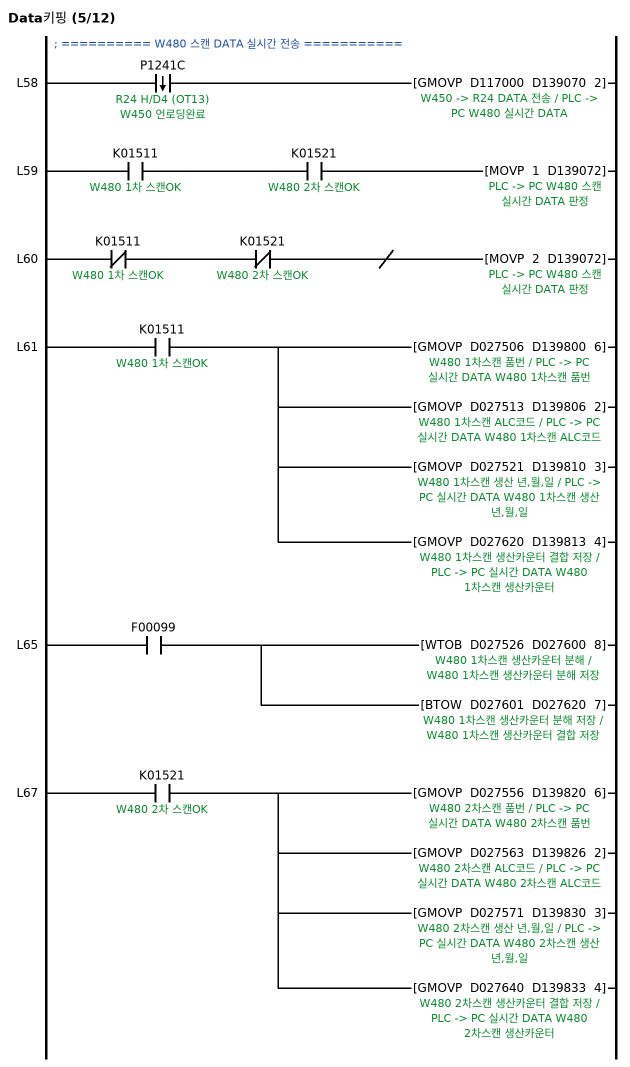
[picture p504: Data키핑 rungs L58-L67]
// ========== W480 스캔 DATA 실시간 전송 ===========
; L58
LOADN     P1241C	// R24 H/D4 (OT13) W450 언로딩완료
GMOVP     D117000 D139070 2	// W450 -> R24 DATA 전송 / PLC -> PC W480 실시간 DATA
; L59
LOAD      K01511	// W480 1차 스캔OK
AND       K01521	// W480 2차 스캔OK
MOVP      1 D139072	// PLC -> PC W480 스캔 실시간 DATA 판정
; L60
LOAD NOT  K01511	// W480 1차 스캔OK
AND NOT   K01521	// W480 2차 스캔OK
NOT
MOVP      2 D139072	// PLC -> PC W480 스캔 실시간 DATA 판정
; L61
LOAD      K01511	// W480 1차 스캔OK
GMOVP     D027506 D139800 6	// W480 1차스캔 품번 / PLC -> PC 실시간 DATA W480 1차스캔 품번
GMOVP     D027513 D139806 2	// W480 1차스캔 ALC코드 / PLC -> PC 실시간 DATA W480 1차스캔 ALC코드
GMOVP     D027521 D139810 3	// W480 1차스캔 생산 년,월,일 / PLC -> PC 실시간 DATA W480 1차스캔 생산 년,월,일
GMOVP     D027620 D139813 4	// W480 1차스캔 생산카운터 결합 저장 / PLC -> PC 실시간 DATA W480 1차스캔 생산카운터
; L65
LOAD      F00099
WTOB      D027526 D027600 8	// W480 1차스캔 생산카운터 분해 / W480 1차스캔 생산카운터 분해 저장
BTOW      D027601 D027620 7	// W480 1차스캔 생산카운터 분해 저장 / W480 1차스캔 생산카운터 결합 저장
; L67
LOAD      K01521	// W480 2차 스캔OK
GMOVP     D027556 D139820 6	// W480 2차스캔 품번 / PLC -> PC 실시간 DATA W480 2차스캔 품번
GMOVP     D027563 D139826 2	// W480 2차스캔 ALC코드 / PLC -> PC 실시간 DATA W480 2차스캔 ALC코드
GMOVP     D027571 D139830 3	// W480 2차스캔 생산 년,월,일 / PLC -> PC 실시간 DATA W480 2차스캔 생산 년,월,일
GMOVP     D027640 D139833 4	// W480 2차스캔 생산카운터 결합 저장 / PLC -> PC 실시간 DATA W480 2차스캔 생산카운터

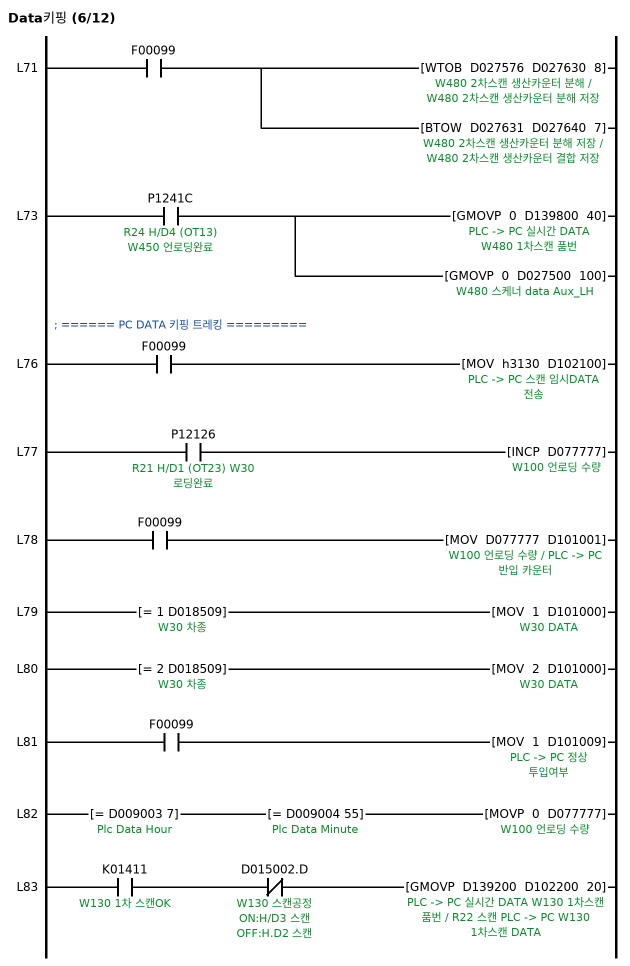
; L71
LOAD      F00099
WTOB      D027576 D027630 8	// W480 2차스캔 생산카운터 분해 / W480 2차스캔 생산카운터 분해 저장
BTOW      D027631 D027640 7	// W480 2차스캔 생산카운터 분해 저장 / W480 2차스캔 생산카운터 결합 저장
; L73
LOAD      P1241C	// R24 H/D4 (OT13) W450 언로딩완료
GMOVP     0 D139800 40	// PLC -> PC 실시간 DATA W480 1차스캔 품번
GMOVP     0 D027500 100	// W480 스케너 data Aux_LH
// ====== PC DATA 키핑 트레킹 =========
; L76
LOAD      F00099
MOV       h3130 D102100	// PLC -> PC 스캔 임시DATA 전송
; L77
LOAD      P12126	// R21 H/D1 (OT23) W30 로딩완료
INCP      D077777	// W100 언로딩 수량
; L78
LOAD      F00099
MOV       D077777 D101001	// W100 언로딩 수량 / PLC -> PC 반입 카운터
; L79
LOAD=     1 D018509	// W30 차종
MOV       1 D101000	// W30 DATA
; L80
LOAD=     2 D018509	// W30 차종
MOV       2 D101000	// W30 DATA
; L81
LOAD      F00099
MOV       1 D101009	// PLC -> PC 정상 투입여부
; L82
LOAD=     D009003 7	// Plc Data Hour
AND=      D009004 55	// Plc Data Minute
MOVP      0 D077777	// W100 언로딩 수량
; L83
LOAD      K01411	// W130 1차 스캔OK
AND NOT   D015002.D	// W130 스캔공정 ON:H/D3 스캔 OFF:H.D2 스캔
GMOVP     D139200 D102200 20	// PLC -> PC 실시간 DATA W130 1차스캔 품번 / R22 스캔 PLC -> PC W130 1차스캔 DATA

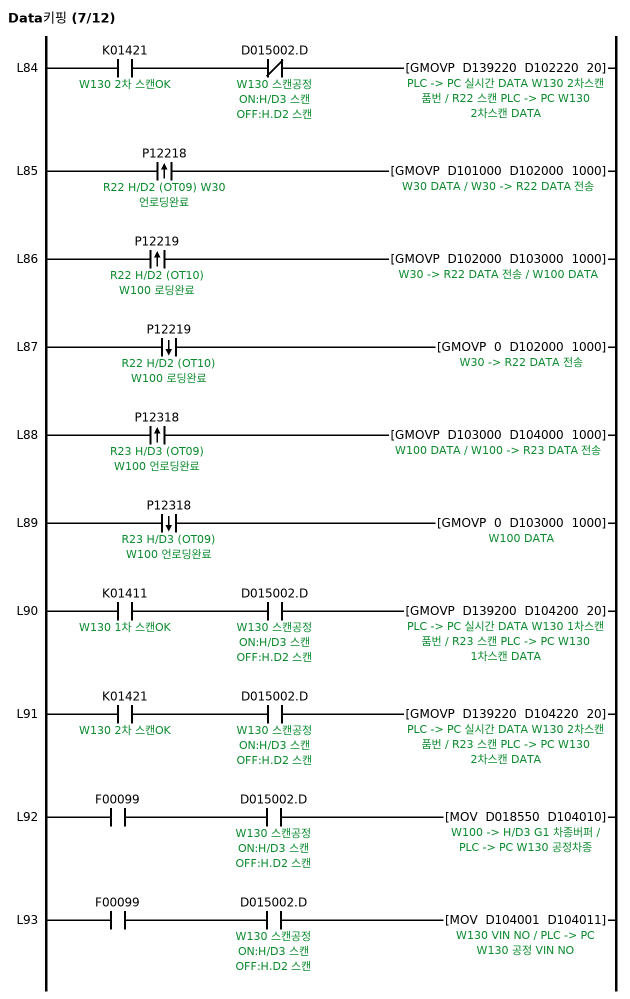
; L84
LOAD      K01421	// W130 2차 스캔OK
AND NOT   D015002.D	// W130 스캔공정 ON:H/D3 스캔 OFF:H.D2 스캔
GMOVP     D139220 D102220 20	// PLC -> PC 실시간 DATA W130 2차스캔 품번 / R22 스캔 PLC -> PC W130 2차스캔 DATA
; L85
LOADP     P12218	// R22 H/D2 (OT09) W30 언로딩완료
GMOVP     D101000 D102000 1000	// W30 DATA / W30 -> R22 DATA 전송
; L86
LOADP     P12219	// R22 H/D2 (OT10) W100 로딩완료
GMOVP     D102000 D103000 1000	// W30 -> R22 DATA 전송 / W100 DATA
; L87
LOADN     P12219	// R22 H/D2 (OT10) W100 로딩완료
GMOVP     0 D102000 1000	// W30 -> R22 DATA 전송
; L88
LOADP     P12318	// R23 H/D3 (OT09) W100 언로딩완료
GMOVP     D103000 D104000 1000	// W100 DATA / W100 -> R23 DATA 전송
; L89
LOADN     P12318	// R23 H/D3 (OT09) W100 언로딩완료
GMOVP     0 D103000 1000	// W100 DATA
; L90
LOAD      K01411	// W130 1차 스캔OK
AND       D015002.D	// W130 스캔공정 ON:H/D3 스캔 OFF:H.D2 스캔
GMOVP     D139200 D104200 20	// PLC -> PC 실시간 DATA W130 1차스캔 품번 / R23 스캔 PLC -> PC W130 1차스캔 DATA
; L91
LOAD      K01421	// W130 2차 스캔OK
AND       D015002.D	// W130 스캔공정 ON:H/D3 스캔 OFF:H.D2 스캔
GMOVP     D139220 D104220 20	// PLC -> PC 실시간 DATA W130 2차스캔 품번 / R23 스캔 PLC -> PC W130 2차스캔 DATA
; L92
LOAD      F00099
AND       D015002.D	// W130 스캔공정 ON:H/D3 스캔 OFF:H.D2 스캔
MOV       D018550 D104010	// W100 -> H/D3 G1 차종버퍼 / PLC -> PC W130 공정차종
; L93
LOAD      F00099
AND       D015002.D	// W130 스캔공정 ON:H/D3 스캔 OFF:H.D2 스캔
MOV       D104001 D104011	// W130 VIN NO / PLC -> PC W130 공정 VIN NO

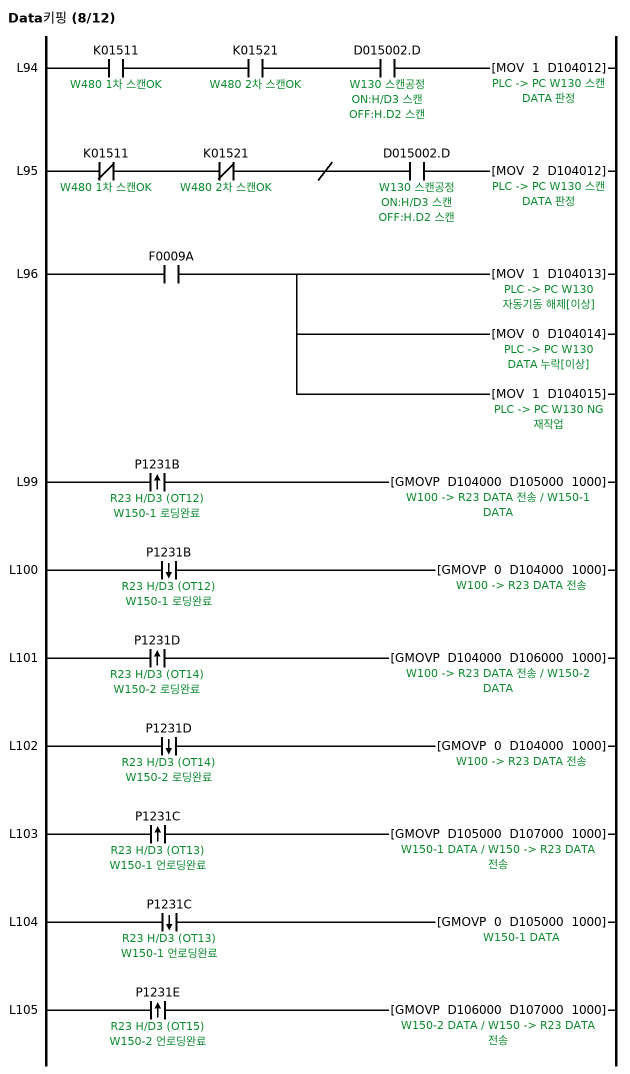
; L94
LOAD      K01511	// W480 1차 스캔OK
AND       K01521	// W480 2차 스캔OK
AND       D015002.D	// W130 스캔공정 ON:H/D3 스캔 OFF:H.D2 스캔
MOV       1 D104012	// PLC -> PC W130 스캔 DATA 판정
; L95
LOAD NOT  K01511	// W480 1차 스캔OK
AND NOT   K01521	// W480 2차 스캔OK
NOT
AND       D015002.D	// W130 스캔공정 ON:H/D3 스캔 OFF:H.D2 스캔
MOV       2 D104012	// PLC -> PC W130 스캔 DATA 판정
; L96
LOAD      F0009A
MOV       1 D104013	// PLC -> PC W130 자동기동 해제[이상]
MOV       0 D104014	// PLC -> PC W130 DATA 누락[이상]
MOV       1 D104015	// PLC -> PC W130 NG 재작업
; L99
LOADP     P1231B	// R23 H/D3 (OT12) W150-1 로딩완료
GMOVP     D104000 D105000 1000	// W100 -> R23 DATA 전송 / W150-1 DATA
; L100
LOADN     P1231B	// R23 H/D3 (OT12) W150-1 로딩완료
GMOVP     0 D104000 1000	// W100 -> R23 DATA 전송
; L101
LOADP     P1231D	// R23 H/D3 (OT14) W150-2 로딩완료
GMOVP     D104000 D106000 1000	// W100 -> R23 DATA 전송 / W150-2 DATA
; L102
LOADN     P1231D	// R23 H/D3 (OT14) W150-2 로딩완료
GMOVP     0 D104000 1000	// W100 -> R23 DATA 전송
; L103
LOADP     P1231C	// R23 H/D3 (OT13) W150-1 언로딩완료
GMOVP     D105000 D107000 1000	// W150-1 DATA / W150 -> R23 DATA 전송
; L104
LOADN     P1231C	// R23 H/D3 (OT13) W150-1 언로딩완료
GMOVP     0 D105000 1000	// W150-1 DATA
; L105
LOADP     P1231E	// R23 H/D3 (OT15) W150-2 언로딩완료
GMOVP     D106000 D107000 1000	// W150-2 DATA / W150 -> R23 DATA 전송

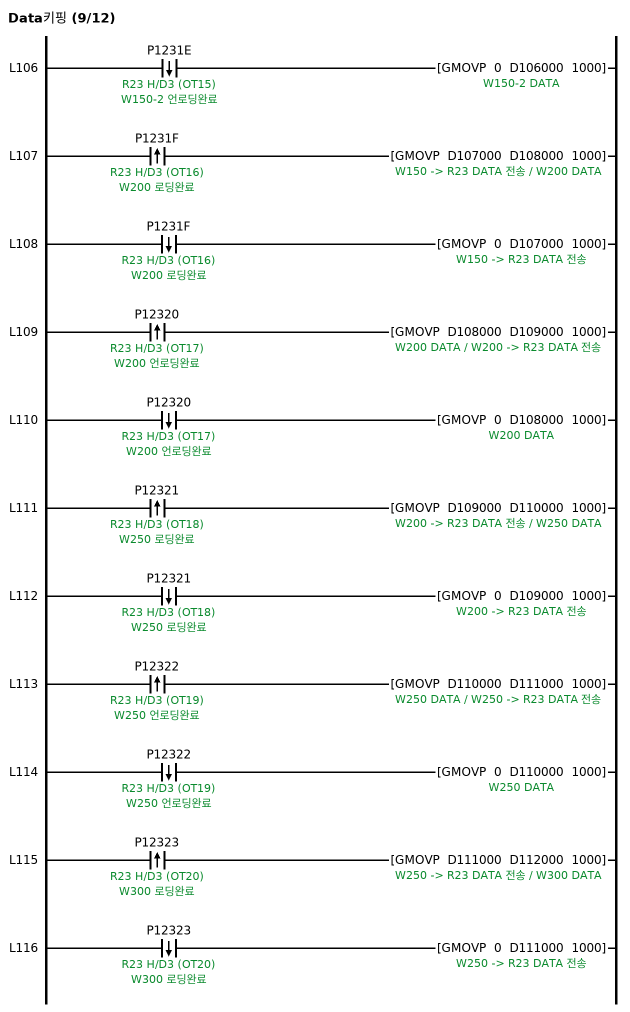
; L106
LOADN     P1231E	// R23 H/D3 (OT15) W150-2 언로딩완료
GMOVP     0 D106000 1000	// W150-2 DATA
; L107
LOADP     P1231F	// R23 H/D3 (OT16) W200 로딩완료
GMOVP     D107000 D108000 1000	// W150 -> R23 DATA 전송 / W200 DATA
; L108
LOADN     P1231F	// R23 H/D3 (OT16) W200 로딩완료
GMOVP     0 D107000 1000	// W150 -> R23 DATA 전송
; L109
LOADP     P12320	// R23 H/D3 (OT17) W200 언로딩완료
GMOVP     D108000 D109000 1000	// W200 DATA / W200 -> R23 DATA 전송
; L110
LOADN     P12320	// R23 H/D3 (OT17) W200 언로딩완료
GMOVP     0 D108000 1000	// W200 DATA
; L111
LOADP     P12321	// R23 H/D3 (OT18) W250 로딩완료
GMOVP     D109000 D110000 1000	// W200 -> R23 DATA 전송 / W250 DATA
; L112
LOADN     P12321	// R23 H/D3 (OT18) W250 로딩완료
GMOVP     0 D109000 1000	// W200 -> R23 DATA 전송
; L113
LOADP     P12322	// R23 H/D3 (OT19) W250 언로딩완료
GMOVP     D110000 D111000 1000	// W250 DATA / W250 -> R23 DATA 전송
; L114
LOADN     P12322	// R23 H/D3 (OT19) W250 언로딩완료
GMOVP     0 D110000 1000	// W250 DATA
; L115
LOADP     P12323	// R23 H/D3 (OT20) W300 로딩완료
GMOVP     D111000 D112000 1000	// W250 -> R23 DATA 전송 / W300 DATA
; L116
LOADN     P12323	// R23 H/D3 (OT20) W300 로딩완료
GMOVP     0 D111000 1000	// W250 -> R23 DATA 전송

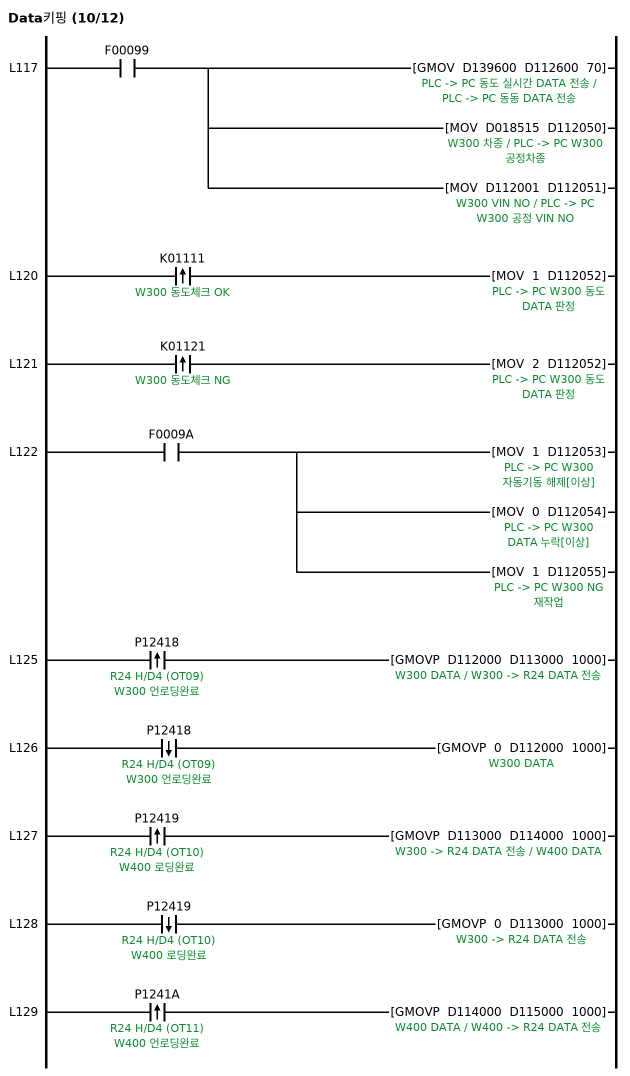
; L117
LOAD      F00099
GMOV      D139600 D112600 70	// PLC -> PC 동도 실시간 DATA 전송 / PLC -> PC 동동 DATA 전송
MOV       D018515 D112050	// W300 차종 / PLC -> PC W300 공정차종
MOV       D112001 D112051	// W300 VIN NO / PLC -> PC W300 공정 VIN NO
; L120
LOADP     K01111	// W300 동도체크 OK
MOV       1 D112052	// PLC -> PC W300 동도 DATA 판정
; L121
LOADP     K01121	// W300 동도체크 NG
MOV       2 D112052	// PLC -> PC W300 동도 DATA 판정
; L122
LOAD      F0009A
MOV       1 D112053	// PLC -> PC W300 자동기동 해제[이상]
MOV       0 D112054	// PLC -> PC W300 DATA 누락[이상]
MOV       1 D112055	// PLC -> PC W300 NG 재작업
; L125
LOADP     P12418	// R24 H/D4 (OT09) W300 언로딩완료
GMOVP     D112000 D113000 1000	// W300 DATA / W300 -> R24 DATA 전송
; L126
LOADN     P12418	// R24 H/D4 (OT09) W300 언로딩완료
GMOVP     0 D112000 1000	// W300 DATA
; L127
LOADP     P12419	// R24 H/D4 (OT10) W400 로딩완료
GMOVP     D113000 D114000 1000	// W300 -> R24 DATA 전송 / W400 DATA
; L128
LOADN     P12419	// R24 H/D4 (OT10) W400 로딩완료
GMOVP     0 D113000 1000	// W300 -> R24 DATA 전송
; L129
LOADP     P1241A	// R24 H/D4 (OT11) W400 언로딩완료
GMOVP     D114000 D115000 1000	// W400 DATA / W400 -> R24 DATA 전송

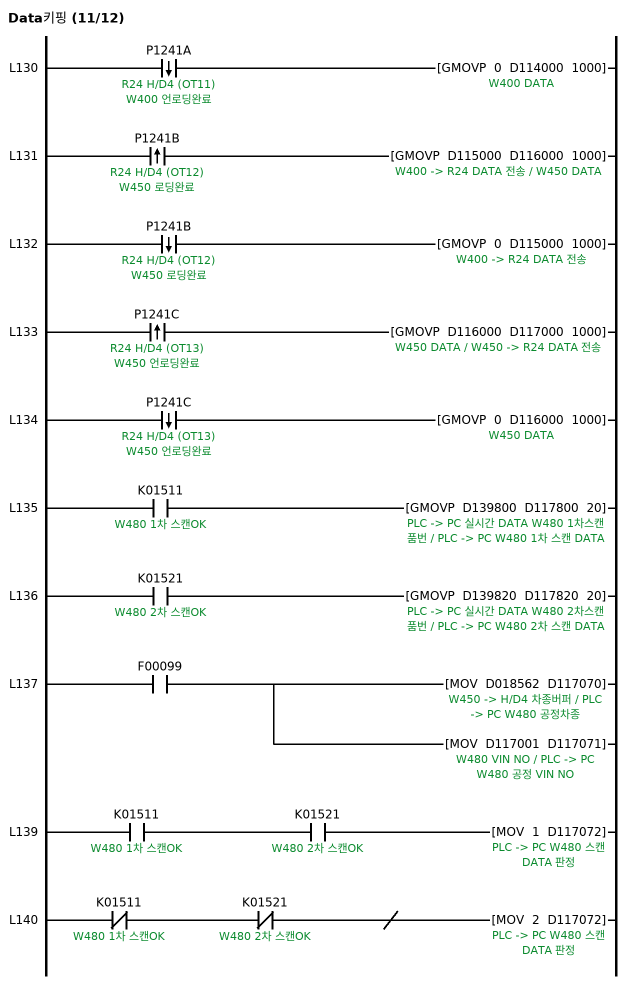
; L130
LOADN     P1241A	// R24 H/D4 (OT11) W400 언로딩완료
GMOVP     0 D114000 1000	// W400 DATA
; L131
LOADP     P1241B	// R24 H/D4 (OT12) W450 로딩완료
GMOVP     D115000 D116000 1000	// W400 -> R24 DATA 전송 / W450 DATA
; L132
LOADN     P1241B	// R24 H/D4 (OT12) W450 로딩완료
GMOVP     0 D115000 1000	// W400 -> R24 DATA 전송
; L133
LOADP     P1241C	// R24 H/D4 (OT13) W450 언로딩완료
GMOVP     D116000 D117000 1000	// W450 DATA / W450 -> R24 DATA 전송
; L134
LOADN     P1241C	// R24 H/D4 (OT13) W450 언로딩완료
GMOVP     0 D116000 1000	// W450 DATA
; L135
LOAD      K01511	// W480 1차 스캔OK
GMOVP     D139800 D117800 20	// PLC -> PC 실시간 DATA W480 1차스캔 품번 / PLC -> PC W480 1차 스캔 DATA
; L136
LOAD      K01521	// W480 2차 스캔OK
GMOVP     D139820 D117820 20	// PLC -> PC 실시간 DATA W480 2차스캔 품번 / PLC -> PC W480 2차 스캔 DATA
; L137
LOAD      F00099
MOV       D018562 D117070	// W450 -> H/D4 차종버퍼 / PLC -> PC W480 공정차종
MOV       D117001 D117071	// W480 VIN NO / PLC -> PC W480 공정 VIN NO
; L139
LOAD      K01511	// W480 1차 스캔OK
AND       K01521	// W480 2차 스캔OK
MOV       1 D117072	// PLC -> PC W480 스캔 DATA 판정
; L140
LOAD NOT  K01511	// W480 1차 스캔OK
AND NOT   K01521	// W480 2차 스캔OK
NOT
MOV       2 D117072	// PLC -> PC W480 스캔 DATA 판정

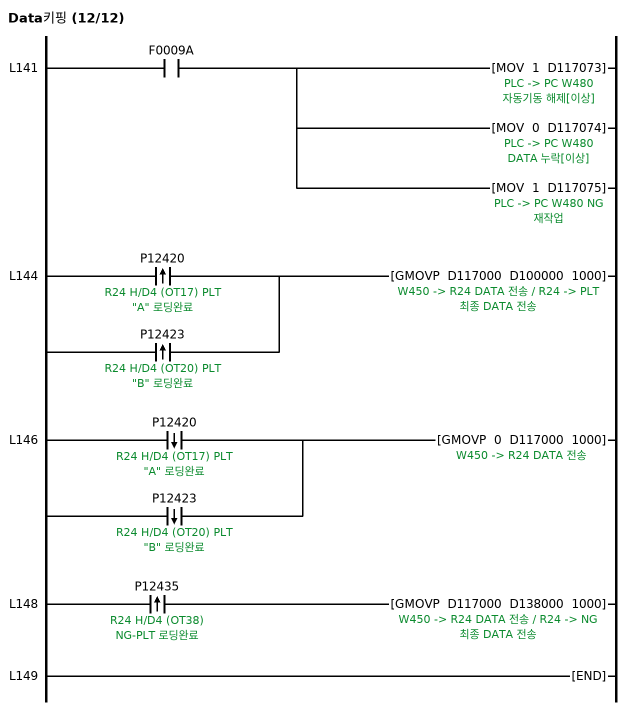
; L141
LOAD      F0009A
MOV       1 D117073	// PLC -> PC W480 자동기동 해제[이상]
MOV       0 D117074	// PLC -> PC W480 DATA 누락[이상]
MOV       1 D117075	// PLC -> PC W480 NG 재작업
; L144
LOADP     P12420	// R24 H/D4 (OT17) PLT "A" 로딩완료
ORP       P12423	// R24 H/D4 (OT20) PLT "B" 로딩완료
GMOVP     D117000 D100000 1000	// W450 -> R24 DATA 전송 / R24 -> PLT 최종 DATA 전송
; L146
LOADN     P12420	// R24 H/D4 (OT17) PLT "A" 로딩완료
ORN       P12423	// R24 H/D4 (OT20) PLT "B" 로딩완료
GMOVP     0 D117000 1000	// W450 -> R24 DATA 전송
; L148
LOADP     P12435	// R24 H/D4 (OT38) NG-PLT 로딩완료
GMOVP     D117000 D138000 1000	// W450 -> R24 DATA 전송 / R24 -> NG 최종 DATA 전송
; L149
END

PROGRAM POP (task: 스캔 프로그램)

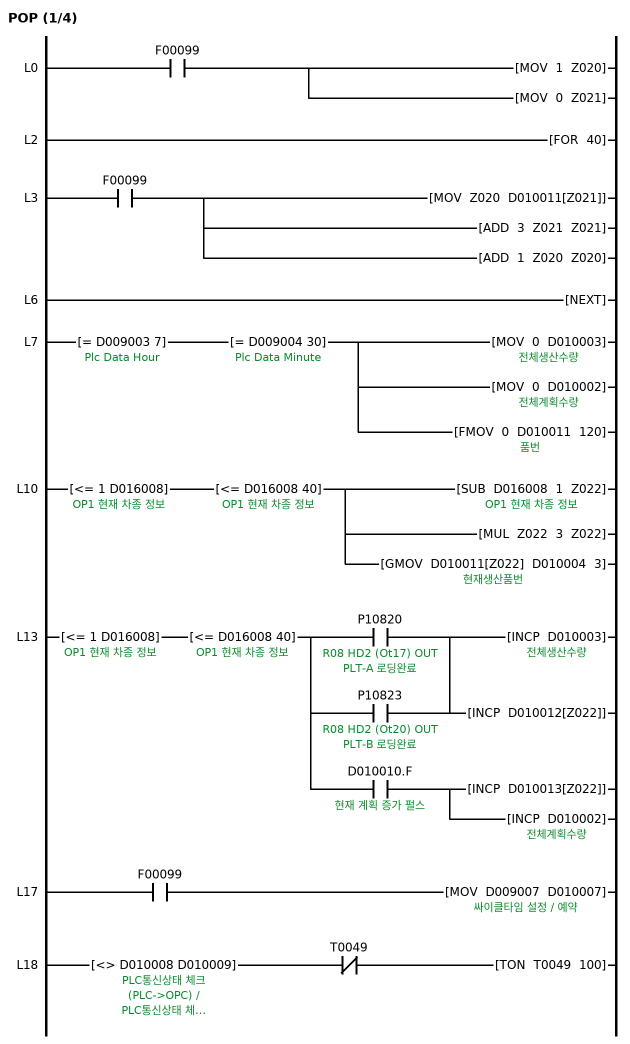
; L0
LOAD      F00099
MOV       1 Z020
MOV       0 Z021
; L2
FOR       40
; L3
LOAD      F00099
MOV       Z020 D010011[Z021]
ADD       3 Z021 Z021
ADD       1 Z020 Z020
; L6
NEXT
; L7
LOAD=     D009003 7	// Plc Data Hour
AND=      D009004 30	// Plc Data Minute
MOV       0 D010003	// 전체생산수량
MOV       0 D010002	// 전체계획수량
FMOV      0 D010011 120	// 품번
; L10
LOAD<=    1 D016008	// OP1 현재 차종 정보
AND<=     D016008 40	// OP1 현재 차종 정보
SUB       D016008 1 Z022	// OP1 현재 차종 정보
MUL       Z022 3 Z022
GMOV      D010011[Z022] D010004 3	// 현재생산품번
; L13
LOAD<=    1 D016008	// OP1 현재 차종 정보
AND<=     D016008 40	// OP1 현재 차종 정보
MPUSH
LOAD      P10820	// R08 HD2 (Ot17) OUT PLT-A 로딩완료
OR        P10823	// R08 HD2 (Ot20) OUT PLT-B 로딩완료
AND LOAD
INCP      D010003	// 전체생산수량
INCP      D010012[Z022]
MPOP
AND       D010010.F	// 현재 계획 증가 펄스
INCP      D010013[Z022]
INCP      D010002	// 전체계획수량
; L17
LOAD      F00099
MOV       D009007 D010007	// 싸이클타임 설정 / 예약
; L18
LOAD<>    D010008 D010009	// PLC통신상태 체크 (PLC->OPC) / PLC통신상태 체크 (OPC->PLC)
AND NOT   T0049
TON       T0049 100

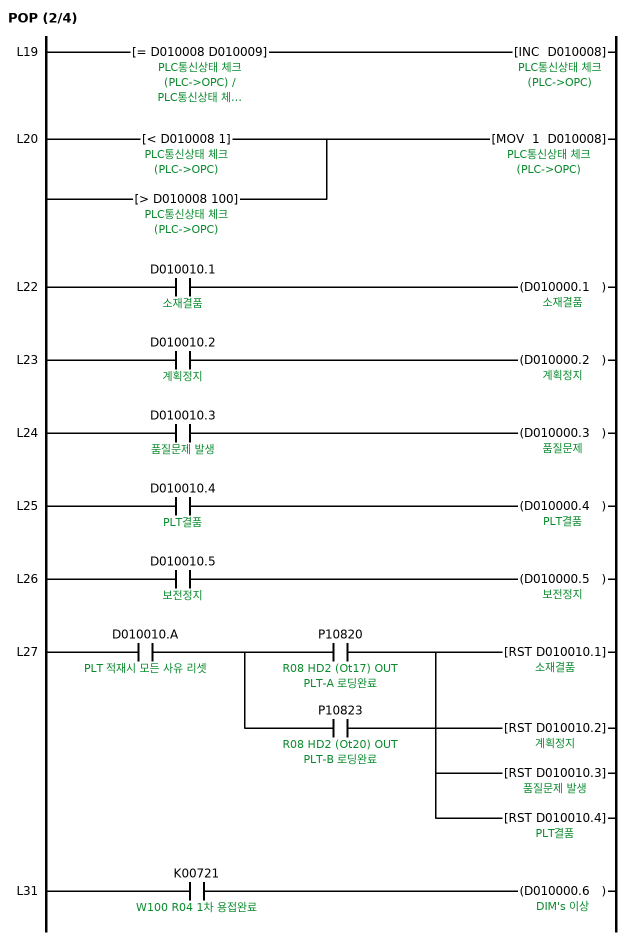
; L19
LOAD=     D010008 D010009	// PLC통신상태 체크 (PLC->OPC) / PLC통신상태 체크 (OPC->PLC)
INC       D010008	// PLC통신상태 체크 (PLC->OPC)
; L20
LOAD<     D010008 1	// PLC통신상태 체크 (PLC->OPC)
OR>       D010008 100	// PLC통신상태 체크 (PLC->OPC)
MOV       1 D010008	// PLC통신상태 체크 (PLC->OPC)
; L22
LOAD      D010010.1	// 소재결품
OUT       D010000.1	// 소재결품
; L23
LOAD      D010010.2	// 계획정지
OUT       D010000.2	// 계획정지
; L24
LOAD      D010010.3	// 품질문제 발생
OUT       D010000.3	// 품질문제
; L25
LOAD      D010010.4	// PLT결품
OUT       D010000.4	// PLT결품
; L26
LOAD      D010010.5	// 보전정지
OUT       D010000.5	// 보전정지
; L27
LOAD      D010010.A	// PLT 적재시 모든 사유 리셋
LOAD      P10820	// R08 HD2 (Ot17) OUT PLT-A 로딩완료
OR        P10823	// R08 HD2 (Ot20) OUT PLT-B 로딩완료
AND LOAD
RST       D010010.1	// 소재결품
RST       D010010.2	// 계획정지
RST       D010010.3	// 품질문제 발생
RST       D010010.4	// PLT결품
; L31
LOAD      K00721	// W100 R04 1차 용접완료
OUT       D010000.6	// DIM's 이상

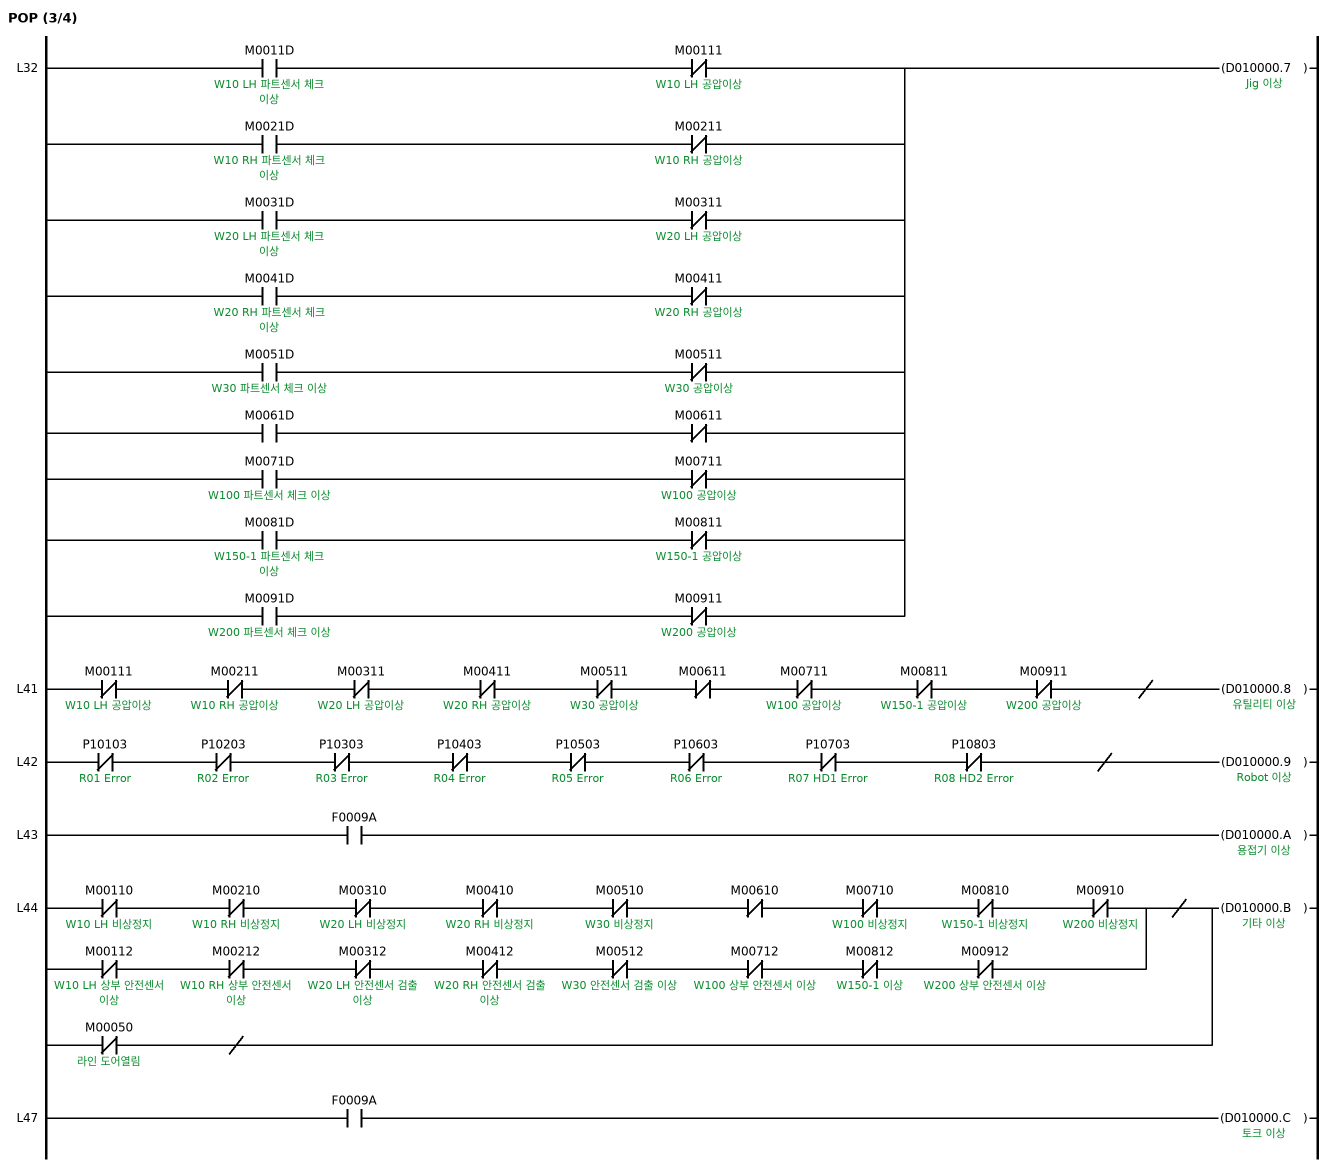
; L32
LOAD      M0011D	// W10 LH 파트센서 체크 이상
AND NOT   M00111	// W10 LH 공압이상
LOAD      M0021D	// W10 RH 파트센서 체크 이상
AND NOT   M00211	// W10 RH 공압이상
OR LOAD
LOAD      M0031D	// W20 LH 파트센서 체크 이상
AND NOT   M00311	// W20 LH 공압이상
OR LOAD
LOAD      M0041D	// W20 RH 파트센서 체크 이상
AND NOT   M00411	// W20 RH 공압이상
OR LOAD
LOAD      M0051D	// W30 파트센서 체크 이상
AND NOT   M00511	// W30 공압이상
OR LOAD
LOAD      M0061D
AND NOT   M00611
OR LOAD
LOAD      M0071D	// W100 파트센서 체크 이상
AND NOT   M00711	// W100 공압이상
OR LOAD
LOAD      M0081D	// W150-1 파트센서 체크 이상
AND NOT   M00811	// W150-1 공압이상
OR LOAD
LOAD      M0091D	// W200 파트센서 체크 이상
AND NOT   M00911	// W200 공압이상
OR LOAD
OUT       D010000.7	// Jig 이상
; L41
LOAD NOT  M00111	// W10 LH 공압이상
AND NOT   M00211	// W10 RH 공압이상
AND NOT   M00311	// W20 LH 공압이상
AND NOT   M00411	// W20 RH 공압이상
AND NOT   M00511	// W30 공압이상
AND NOT   M00611
AND NOT   M00711	// W100 공압이상
AND NOT   M00811	// W150-1 공압이상
AND NOT   M00911	// W200 공압이상
NOT
OUT       D010000.8	// 유틸리티 이상
; L42
LOAD NOT  P10103	// R01 Error
AND NOT   P10203	// R02 Error
AND NOT   P10303	// R03 Error
AND NOT   P10403	// R04 Error
AND NOT   P10503	// R05 Error
AND NOT   P10603	// R06 Error
AND NOT   P10703	// R07 HD1 Error
AND NOT   P10803	// R08 HD2 Error
NOT
OUT       D010000.9	// Robot 이상
; L43
LOAD      F0009A
OUT       D010000.A	// 용접기 이상
; L44
LOAD NOT  M00110	// W10 LH 비상정지
AND NOT   M00210	// W10 RH 비상정지
AND NOT   M00310	// W20 LH 비상정지
AND NOT   M00410	// W20 RH 비상정지
AND NOT   M00510	// W30 비상정지
AND NOT   M00610
AND NOT   M00710	// W100 비상정지
AND NOT   M00810	// W150-1 비상정지
AND NOT   M00910	// W200 비상정지
LOAD NOT  M00112	// W10 LH 상부 안전센서 이상
AND NOT   M00212	// W10 RH 상부 안전센서 이상
AND NOT   M00312	// W20 LH 안전센서 검출 이상
AND NOT   M00412	// W20 RH 안전센서 검출 이상
AND NOT   M00512	// W30 안전센서 검출 이상
AND NOT   M00712	// W100 상부 안전센서 이상
AND NOT   M00812	// W150-1 이상
AND NOT   M00912	// W200 상부 안전센서 이상
OR LOAD
NOT
LOAD NOT  M00050	// 라인 도어열림
NOT
OR LOAD
OUT       D010000.B	// 기타 이상
; L47
LOAD      F0009A
OUT       D010000.C	// 토크 이상

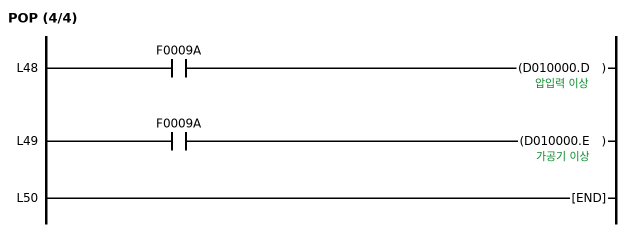
; L48
LOAD      F0009A
OUT       D010000.D	// 압입력 이상
; L49
LOAD      F0009A
OUT       D010000.E	// 가공기 이상
; L50
END

VARIABLES AND COMMENTS (devices not used above)
M02300	BIT	Servo 4  Auto Pb
M02301	BIT	Servo 4  Manual Pb
M02302	BIT	Servo 4 Jog + Pb
M02303	BIT	Servo 4 Jog - Pb
M02305	BIT	Servo 4  Home Pos. Set Pb
M02306	BIT	Servo 4  Position1 Select Pb
M02307	BIT	Servo 4  Position2 Select Pb
M02308	BIT	Servo 4  Position3 Select Pb
M02309	BIT	Servo 4  Position4 Select Pb
M0230A	BIT	Servo 4  Position5 Select Pb
M0230C	BIT	Servo 4  Position7 Select Pb
M0230D	BIT	Servo 4  Position8 Select Pb
M02310	BIT	Servo 4  Auto Lamp
M02311	BIT	Servo 4  Manual Mode Lamp
M02315	BIT	Servo 4  Home Pos Set Comple
M02316	BIT	Servo 4  Position1 Select Comple
M02317	BIT	Servo 4  Position2 Select Comple
M02318	BIT	Servo 4  Position3 Select Comple
M02319	BIT	Servo 4  Position4 Select Comple
M0231A	BIT	Servo 4  Position5 Select Comple
M02321	BIT	Servo 4 POS 1 (Home)
M02322	BIT	Servo 4 Pos 2 (Worker)
M02331	BIT	Servo 4  Position 1 Select'g
M02332	BIT	Servo 4  Position2 Select'g
M02333	BIT	Servo 4  Position3 Select'g
M02334	BIT	Servo 4  Position4 Select'g
M02335	BIT	Servo 4  Position5 Select'g
M02341	BIT	Servo 4  Pos 1 Move
M02342	BIT	Servo 4  Pos2 Move
M02343	BIT	Servo 4  Pos3 Move
M02344	BIT	Servo 4  Pos4 Move
M02345	BIT	Servo 4  Pos5 Move
M02350	BIT	Servo 4  Auto Location Possible
M02354	BIT	Servo 4 Power ON Check
M02361	BIT	Servo 4  Position 1 (Home) Move Commend
M02362	BIT	Servo 4  Position2 (Worker) Move Commend
M02363	BIT	Servo 4  Position3 (1st Weld) Move Commend
M02364	BIT	Servo 4  Position4 (2nd Weld) Move Commend
M02365	BIT	Servo 4  Position5 (3rd Weld) Move Commend
D02600	WORD	서보 4 현재 위치 데이타 Low
D02614	WORD	서보 4 Table 1 위치 데이타 Low
D02636	WORD	서보 4 이상 코드 Low
D02638	WORD	서보 4 통신 하트 비트 리턴 Low
D02640	WORD	서보 4 Mode (0=자동, 1=수동)
D02641	WORD	서보 4 통신 체크용 스캔 카운터
D02650	WORD	서보 4 등록 포지션 1번 Low
D02652	WORD	서보 4 등록 포지션 2번 Low
D02654	WORD	서보 4 등록 포지션 3번 Low
D02656	WORD	서보 4 등록 포지션 4번 Low
D02658	WORD	서보 4 등록 포지션 5번 Low
D02670	WORD	서보 4 등록 포지션 1번 Low Band Low
D02672	WORD	서보 4 등록 포지션 2번 Low Band Low
D02674	WORD	서보 4 등록 포지션 3번 Low Band Low
D02676	WORD	서보 4 등록 포지션 4번 Low Band Low
D02678	WORD	서보 4 등록 포지션 5번 Low Band Low
D02680	WORD	서보 4 등록 포지션 1번 High Band Low
D02682	WORD	서보 4 등록 포지션 2번 High Band Low
D02684	WORD	서보 4 등록 포지션 3번 High Band Low
D02686	WORD	서보 4 등록 포지션 4번 High Band Low
D02688	WORD	서보 4 등록 포지션 5번 High Band Low
D02702	WORD	서보 4 Table 1 위치 데이타 Low
D02704	WORD	서보 4 Table 1 위치 결정 속도 Low
D02738	WORD	서보 4 통신 하트 비트 Low
D02608.6	BIT	서보 4 리셋 (RES) 리턴
D02609.1	BIT	서보 4 자동/수동 선택 (MD0) 리턴
D02609.3	BIT	서보 4 포인트 테이블 No. 선택1 (DI0) 리턴
D02609.4	BIT	서보 4 포인트 테이블 No. 선택2 (DI1) 리턴
D02609.5	BIT	서보 4 포인트 테이블 No. 선택3 (DI2) 리턴
D02609.6	BIT	서보 4 포인트 테이블 No. 선택4 (DI3) 리턴
D02609.D	BIT	서보 4 포인트 테이블 No. 선택5 (DI4) 리턴
D02610.0	BIT	서보 4 준비완료 (RD)
D02610.8	BIT	서보 4 고장 (ALM)
D02611.1	BIT	서보 4 원점복귀완료 (ZP)
D02611.C	BIT	서보 4 이동완료 (MEND)
D02700.0	BIT	서보 4 서보 ON (SON)
D02700.1	BIT	서보 4 정전스트로크엔드 (LSP)
D02700.2	BIT	서보 4 역전스트로크엔드 (LSN)
D02700.6	BIT	서보 4 리셋 (RES)
D02700.B	BIT	서보 4 정전 시동 (ST1)
D02700.C	BIT	서보 4 역전 시동 (ST2)
D02701.1	BIT	서보 4 자동/수동 선택 (MD0)
D02701.3	BIT	서보 4 포인트 테이블 No. 선택1 (DI0)
D02701.4	BIT	서보 4 포인트 테이블 No. 선택2 (DI1)
D02701.5	BIT	서보 4 포인트 테이블 No. 선택3 (DI2)
D02701.6	BIT	서보 4 포인트 테이블 No. 선택4 (DI3)
D02701.D	BIT	서보 4 포인트 테이블 No. 선택5 (DI4)
D03411.1	BIT	서보 7 원점복귀완료 (ZP)
D03500.0	BIT	서보 7 서보 ON (SON)
D03500.1	BIT	서보 7 정전스트로크엔드 (LSP)
D03500.2	BIT	서보 7 역전스트로크엔드 (LSN)
D03500.6	BIT	서보 7 리셋 (RES)
D03500.B	BIT	서보 7 정전 시동 (ST1)
D03500.C	BIT	서보 7 역전 시동 (ST2)
D03501.3	BIT	서보 7 포인트 테이블 No. 선택1 (DI0)
D03501.4	BIT	서보 7 포인트 테이블 No. 선택2 (DI1)
D03501.5	BIT	서보 7 포인트 테이블 No. 선택3 (DI2)
D03501.6	BIT	서보 7 포인트 테이블 No. 선택4 (DI3)
D03501.D	BIT	서보 7 포인트 테이블 No. 선택5 (DI4)
M1022F	BIT	R02 (IN32)
M1022E	BIT	R02 (IN31)
M1032F	BIT	R03 (IN32)
M1032E	BIT	R03 (IN31)
M1012E	BIT	R01 (IN31)
M1012F	BIT	R01 (IN32)
M1042E	BIT	R04 (IN31)
M1042F	BIT	R04 (IN32)
M1052E	BIT	R05 (IN31)
M1052F	BIT	R05 (IN32)
M0230B	BIT	Servo 4  Position6 Select Pb
M0231B	BIT	Servo 4  Position6 Select Comple
M0231C	BIT	Servo 4  Position7 Select Comple
M0231D	BIT	Servo 4  Position8 Select Comple
M02326	BIT	Servo 4 POS 6 ()
M0232C	BIT	Servo 4  Move Pb
M0232D	BIT	Servo 4 Copy From CV
M0232E	BIT	Servo 4 Copy from PV
M02336	BIT	Servo 4  Position6 Select'g
M02337	BIT	Servo 4  Position7 Select'g
M02338	BIT	Servo 4  Position8 Select'g
M02346	BIT	Servo 4  Pos6 Move
M02347	BIT	Servo 4  Pos7 Move
M02348	BIT	Servo 4  Pos8 Move
M02366	BIT	Servo 4  Position6()Move Commend
M02367	BIT	Servo 4  Position7 (Load'g) Move Commend
M02368	BIT	Servo 4  Position8 (Unload'g) Move Commend
D03410.8	BIT	서보 7 고장 (ALM)
D03408.6	BIT	서보 7 리셋 (RES) 리턴
D03411.C	BIT	서보 7 이동완료 (MEND)
D15001.8	BIT	OP1 STN08 Select Pb
D15001.9	BIT	OP1 STN09 IDLE Select Pb
D15001.A	BIT	OP1 STN10 Select Pb
D15001.B	BIT	OP1 STN11 Select Pb
D15001.C	BIT	OP1 STN12 Select Pb
K07211	BIT	R02+W100 서보1 간섭 이상
K07212	BIT	R--+W100 서보1 간섭 이상
K07221	BIT	R03+W700-2 서보2 간섭 이상
K07222	BIT	R--+W700-2 서보2 간섭 이상
K07231	BIT	R04+W40 서보3 간섭 이상
K07232	BIT	R--+W40 서보3 간섭 이상
K07240	BIT	W400 서보4 로봇 간섭이상
K07241	BIT	R05+W400 서보4 간섭 이상
K07242	BIT	R06+W400 서보4 간섭 이상
K07243	BIT	R--+W400 서보4 간섭 이상
K07252	BIT	R07+W70 서보5 간섭 이상
K07261	BIT	R07+W80 서보6 간섭 이상
M0030B	BIT	W20 LH 상부 안전센서 정상
M00332	BIT	W20 LH 기동 Pulse
M00342	BIT	W20-3 LH 로보트 간섭무
M00343	BIT	W20 LH Work 로보트 간섭무
M00370	BIT	W20 LH 기동준비
M00371	BIT	W20 LH 1차 기동
M00372	BIT	W20 LH 2차 기동
M00373	BIT	W20 LH 3차 기동
M00506	BIT	W30 서보 동작가능
M0050B	BIT	W30 상부 안전센서 정상
M0050C	BIT	W30 하부 안전세서 정상
M0050D	BIT	W30 안전매트 정상
M00560	BIT	W30 원위치복귀 Pb (XP)
M00574	BIT	W30 4차 기동
M00584	BIT	W30 4차 기동완료
M00070	BIT	OP1 Robot Error
M00073	BIT	OP2 Robot Error
D00005	WORD	OP2 Touch Display Change 비밀번호
M02323	BIT	Servo 4 Pos 3 (1st Weld'g)
M02324	BIT	Servo 4 POS 4 (2nd Weld'g)
M02325	BIT	Servo 4 POS 5 (3rd Weld'g)
M02328	BIT	Servo 4 POS 8 (Unload'g)
M02327	BIT	Servo 4 POS 7 (Load'g)
K07210	BIT	W100 서보1 로봇 간섭이상
K07250	BIT	W70 서보5 로봇 간섭이상
K07260	BIT	W80 서보6 로봇 간섭이상
K07251	BIT	R--+W70 서보5 간섭 이상
K07270	BIT	OP1 Total 서보 로봇 간섭이상
D18002	WORD	R01 표준시간 최소 용접시간
D18012	WORD	R02 표준시간 최소 용접시간
D18022	WORD	R03 표준시간 최소 용접시간
D18032	WORD	R04 표준시간 최소 용접시간
P10529	BIT	R05 (OT26)
M1062F	BIT	R06 (IN32)
M10027	BIT	R-- 원점 요구 Pb
M10037	BIT	R-- 원점 확인 요구
D18066.1	BIT	W200 R05 용접구간 카운터
M16285	BIT	OP1 R05 Seleted
M16286	BIT	OP1 R06 Seleted
M16265	BIT	OP1 R05 Select Pb
M16266	BIT	OP1 R06 Select Pb
D18076.1	BIT	W200 R06 용접구간 카운터
M00035	BIT	OP3 Emergency Stop
P0030F	BIT	W10 LH 1차 클램프 풀림2
M16328	BIT	OP2 R-- Seleted
M16308	BIT	OP2 R-- Select Pb
M16580	BIT	OP1 R16 Power On Lamp
M03780	BIT	R-- 주간 초품 원점 체크 지령
M03781	BIT	R-- 주간 중품 원점 체크 지령
M03782	BIT	R-- 야간 초품 원점 체크 지령
M03783	BIT	R-- 야간 중품 원점 체크 지령
M03788	BIT	R-- 전체 카운터 클리어 Pb
M03789	BIT	R-- OK 카운터 클리어 Pb
M0378A	BIT	R-- NG 카운터 클리어 Pb
D04880	WORD	R-- 원점 주간 초품 OK/NG 정보
D04881	WORD	R-- 원점 주간 중품 OK/NG 정보
D04882	WORD	R-- 원점 야간 초품 OK/NG 정보
D04883	WORD	R-- 원점 야간 중품 OK/NG 정보
D04884	WORD	R-- 원점 확인 전체 카운터
D04885	WORD	R-- 원점 OK 카운터
D04886	WORD	R-- 원점 NG 카운터
D04911	WORD	R-- 원점 주간 중품 OK/NG 정보
D04921	WORD	R-- 원점 주간 중품 OK/NG 정보
K07271	BIT	OP2 Total 서보 로봇 간섭이상
D18086.1	BIT	W300 R05 용접구간 카운터
D18096.1	BIT	W300 R06 용접구간 카운터
D18106.1	BIT	W600 R-- 용접구간 카운터
D18116.1	BIT	W600 R-- 용접구간 카운터
D18126.1	BIT	W700 R-- 용접구간 카운터
D18136.1	BIT	W700 R07 용접구간 카운터
M00091	BIT	OP2 토탈 공정 선택
M00060	BIT	OP2 Robot Emergency Stop
M16500	BIT	Line 강제배출 Mode On Pb
M16501	BIT	Line 강제배출 Mode Off Pb
T0018	BIT/WORD	Line 강제배출 Mode Off Delay Tmr
T0008	BIT/WORD	Line 강제배출 Mode On Delay Tmr
D00023	WORD	OP2 Touch Display Change 비밀번호
T0116	BIT/WORD	W10 LH 파트이상 (누락)지연
P0050F	BIT	W10 RH 1차 클램프 풀림2
D00117	WORD	W50 파트램프 상태7
M00306	BIT	W20 LH 서보 동작가능
M0030C	BIT	W20 LH 하부 안전세서 정상
M0030D	BIT	W20 LH 안전매트 정상
M00374	BIT	W20 LH 4차 기동
M00381	BIT	W20 LH 1차 기동완료
M00382	BIT	W20 LH 2차 기동완료
M00383	BIT	W20 LH 3차 기동완료
M00384	BIT	W20 LH 4차 기동완료
M00406	BIT	W20 RH 서보 동작가능
M0040C	BIT	W20 RH 하부 안전세서 정상
M0040B	BIT	W20 RH 상부 안전센서 정상
M0040D	BIT	W20 RH 안전매트 정상
M00432	BIT	W20 RH 기동 Pulse
M00472	BIT	W20 RH 2차 기동
M00473	BIT	W20 RH 3차 기동
M00441	BIT	W20-2 RH 로보트 간섭무
M00442	BIT	W20-3 RH 로보트 간섭무
M00443	BIT	W20 RH Work 로보트 간섭무
M00470	BIT	W20 RH 기동준비
M00471	BIT	W20 RH 1차 기동
M00474	BIT	W20 RH 4차 기동
M00481	BIT	W20 RH 1차 기동완료
M00482	BIT	W20 RH 2차 기동완료
M00483	BIT	W20 RH 3차 기동완료
M00484	BIT	W20 RH 4차 기동완료
T0403	BIT/WORD	W20 RH Air Blow On TMR
M02351	BIT	Servo 4 수동선택
M02352	BIT	Servo 4 자동선택
M02353	BIT	Servo 4 이상해제
M02340	BIT	Servo 4 원점복귀 명령
D02660	WORD	서보 4 사용자 입력 위치 데이타1 Low
D02662	WORD	서보 4 사용자 입력 위치 데이타2 Low
D02664	WORD	서보 4 사용자 입력 위치 데이타3 Low
D02706	WORD	서보 4 예약
D02708	WORD	서보 4 예약
D03409.1	BIT	서보 7 자동/수동 선택 (MD0) 리턴
D03501.1	BIT	서보 7 자동/수동 선택 (MD0)
D03409.3	BIT	서보 7 포인트 테이블 No. 선택1 (DI0) 리턴
D03409.4	BIT	서보 7 포인트 테이블 No. 선택2 (DI1) 리턴
D03409.5	BIT	서보 7 포인트 테이블 No. 선택3 (DI2) 리턴
D03409.6	BIT	서보 7 포인트 테이블 No. 선택4 (DI3) 리턴
D03409.D	BIT	서보 7 포인트 테이블 No. 선택5 (DI4) 리턴
D00006	WORD	OP3 Touch Display Change 비밀번호
P0030D	BIT	W10 LH 1차 클램프 풀림1
P0030C	BIT	W10 LH 1차 클램프 잠김1
D04701.0	BIT	OP2 로보트 용접 카운트 전체 리셋PB
M10028	BIT	R-- 원점 요구 Pb
M10038	BIT	R-- 원점 확인 요구
M03790	BIT	R-- 주간 초품 원점 체크 지령
M03791	BIT	R-- 주간 중품 원점 체크 지령
M03792	BIT	R-- 야간 초품 원점 체크 지령
M03793	BIT	R-- 야간 중품 원점 체크 지령
M10039	BIT	R-- 원점 확인 요구
M03798	BIT	R-- 전체 카운터 클리어 Pb
M03799	BIT	R-- OK 카운터 클리어 Pb
M0379A	BIT	R-- NG 카운터 클리어 Pb
M03820	BIT	R-- 주간 초품 원점 체크 지령
M03821	BIT	R-- 주간 중품 원점 체크 지령
M03822	BIT	R-- 야간 초품 원점 체크 지령
M03823	BIT	R-- 야간 중품 원점 체크 지령
M03828	BIT	R-- 전체 카운터 클리어 Pb
M03829	BIT	R-- OK 카운터 클리어 Pb
M0382A	BIT	R-- NG 카운터 클리어 Pb
M03830	BIT	R-- 주간 초품 원점 체크 지령
M03831	BIT	R-- 주간 중품 원점 체크 지령
M03832	BIT	R-- 야간 초품 원점 체크 지령
M03833	BIT	R-- 야간 중품 원점 체크 지령
M03838	BIT	R-- 전체 카운터 클리어 Pb
M03839	BIT	R-- OK 카운터 클리어 Pb
M0383A	BIT	R-- NG 카운터 클리어 Pb
M03840	BIT	R-- 주간 초품 원점 체크 지령
M03841	BIT	R-- 주간 중품 원점 체크 지령
M03842	BIT	R-- 야간 초품 원점 체크 지령
M03843	BIT	R-- 야간 중품 원점 체크 지령
M03848	BIT	R-- 전체 카운터 클리어 Pb
M03849	BIT	R-- OK 카운터 클리어 Pb
M0384A	BIT	R-- NG 카운터 클리어 Pb
M03850	BIT	R12 주간 초품 원점 체크 지령
M03851	BIT	R12 주간 중품 원점 체크 지령
M03852	BIT	R12 야간 초품 원점 체크 지령
M03853	BIT	R12 야간 중품 원점 체크 지령
M03858	BIT	R12 전체 카운터 클리어 Pb
M03859	BIT	R12 OK 카운터 클리어 Pb
M0385A	BIT	R12 NG 카운터 클리어 Pb
M03860	BIT	R13 주간 초품 원점 체크 지령
M03861	BIT	R13 주간 중품 원점 체크 지령
M03862	BIT	R13 야간 초품 원점 체크 지령
M03863	BIT	R13 야간 중품 원점 체크 지령
M03868	BIT	R13 전체 카운터 클리어 Pb
M03869	BIT	R13 OK 카운터 클리어 Pb
M0386A	BIT	R13 NG 카운터 클리어 Pb
M03870	BIT	R14 주간 초품 원점 체크 지령
M03871	BIT	R14 주간 중품 원점 체크 지령
M03872	BIT	R14 야간 초품 원점 체크 지령
M03873	BIT	R14 야간 중품 원점 체크 지령
M03878	BIT	R14 전체 카운터 클리어 Pb
M03879	BIT	R14 OK 카운터 클리어 Pb
M0387A	BIT	R14 NG 카운터 클리어 Pb
M10029	BIT	R-- 원점 요구 Pb
D04890	WORD	R-- 원점 주간 초품 OK/NG 정보
D04900	WORD	R-- 원점 주간 초품 OK/NG 정보
D04920	WORD	R-- 원점 주간 초품 OK/NG 정보
D04891	WORD	R-- 원점 주간 중품 OK/NG 정보
D04892	WORD	R-- 원점 야간 초품 OK/NG 정보
D04893	WORD	R-- 원점 야간 중품 OK/NG 정보
D04894	WORD	R-- 원점 확인 전체 카운터
D04895	WORD	R-- 원점 OK 카운터
D04896	WORD	R-- 원점 NG 카운터
D04901	WORD	R-- 원점 주간 중품 OK/NG 정보
D04902	WORD	R-- 원점 야간 초품 OK/NG 정보
D04903	WORD	R-- 원점 야간 중품 OK/NG 정보
D04904	WORD	R-- 원점 확인 전체 카운터
D04905	WORD	R-- 원점 OK 카운터
D04906	WORD	R-- 원점 NG 카운터
D04912	WORD	R-- 원점 야간 초품 OK/NG 정보
D04913	WORD	R-- 원점 야간 중품 OK/NG 정보
D04914	WORD	R-- 원점 확인 전체 카운터
D04915	WORD	R-- 원점 OK 카운터
D04916	WORD	R-- 원점 NG 카운터
D04922	WORD	R-- 원점 야간 초품 OK/NG 정보
D04923	WORD	R-- 원점 야간 중품 OK/NG 정보
D04924	WORD	R-- 원점 확인 전체 카운터
D04925	WORD	R-- 원점 OK 카운터
D04926	WORD	R-- 원점 NG 카운터
T0303	BIT/WORD	W20 LH Air Blow On TMR
D00001.1	BIT	Main 62405-S1000 2WD-가솔린 LHD 비방청
D00001.2	BIT	Main 62405-S1250 2WD-가솔린 LHD 방청
D00001.3	BIT	Main 62405-S1100 2WD-디젤 LHD 비방청
D00001.4	BIT	Main 62405-S1350 2WD-디젤 LHD 방청
D00001.5	BIT	Main 62405-S1400 4WD-가솔린 LHD 비방청
D00001.6	BIT	Main 62405-S1650 4WD-가솔린 LHD 방청
D00001.7	BIT	Main 62405-S1500 4WD-디젤 LHD 비방청
D00001.8	BIT	Main 62405-S1750 4WD-디젤 LHD 방청
D00001.9	BIT	Main 62405-S1850 2WD-디젤 LHD 방청
D00001.A	BIT	Main 62405-S1950 4WD-디젤 LHD 방청
D00001.B	BIT	Main 62405-S1010 2WD-가솔린 RHD 비방청
D00001.C	BIT	Main 62405-S1110 2WD-디젤 RHD 비방청
D00001.D	BIT	Main 62405-S1410 4WD-가솔린 RHD 비방청
D00001.E	BIT	Main 62405-S1660 4WD-가솔린 RHD 방청
D00002.0	BIT	Main 62405-S1860 2WD-디젤 RHD 방청
D00002.1	BIT	Main 62405-S1960 4WD-디젤 RHD 방청
P0050D	BIT	W10 RH 1차 클램프 풀림1
D08810.0	BIT	OP2 노즐청소 카운터 전체리셋  PB
T0117	BIT/WORD	W10 LH 사양감지 체크완료 지연
D00014.0	BIT	Line JIG All No Part[Main]
D00014.1	BIT	Robot All No Part/ All Home[main]
D00011.3	BIT	All Jig No Work Completed MAIN
D00014.3	BIT	All Jig No Work Completed MAIN
D00010	WORD	Exhaust Mode 1:Running 0:Cancel
D00013	WORD	Exhaust Mode[op3_라인2] 1:Running 0:Cancel
M10041	BIT	OP2 원점체크 NG 리셋PB
P10240	BIT	R02 (OT49)
P10340	BIT	R03 (OT49)
P10440	BIT	R04 (OT49)
P10540	BIT	R05 (OT49)
P10640	BIT	R06 (OT49)
M10067	BIT	R-- 원점체크 요구 On
M10068	BIT	R-- 원점체크 요구 On
M10069	BIT	R-- 원점체크 요구 On
T2517	BIT/WORD	R-- 원점체크 요구/완료 해제지연
T2518	BIT/WORD	R-- 원점체크 요구/완료 해제지연
T2519	BIT/WORD	R-- 원점체크 요구/완료 해제지연
D07000.7	BIT	SR01 용접팁교환 요구 PB
D07000.8	BIT	SR02 용접팁교환 요구 PB
D07002.7	BIT	SR01 용접팁교환 완료 PB
D07002.8	BIT	SR02 용접팁교환 완료 PB
D07003.1	BIT	R-- 용접팁교환 요구 PB
D07003.2	BIT	R-- 용접팁교환 요구 PB
D07003.3	BIT	R-- 용접팁교환 요구 PB
D07003.4	BIT	R07 용접팁교환 요구 PB
D07003.5	BIT	R08 용접팁교환 요구 PB
D07003.6	BIT	R12 용접팁교환 요구 PB
D20000	WORD	스캐너 Data
D17539.0	BIT	W100/W50-1 지그사용 마킹기 데이터
D17539.1	BIT	W150/W50-1 지그사용 마킹기 데이터
T0503	BIT/WORD	W30 Air Blow On TMR
R00700	WORD	R-- 원점체크 최종점검 일자 년
R00800	WORD	R-- 원점체크 최종점검 일자 년
R00900	WORD	R-- 원점체크 최종점검 일자 년
R01000	WORD	R07 원점체크 최종점검 일자 년
R01100	WORD	R08 원점체크 최종점검 일자 년
R01200	WORD	R12 원점체크 최종점검 일자 년
R01300	WORD	R13 원점체크 최종점검 일자 년
R01400	WORD	R14 원점체크 최종점검 일자 년
D18204	WORD	W50 R01 용접구간 카운터
R10001	WORD	Arc_R01 용접구간 저장 시작워드
P1023F	BIT	R02 (OT48)
R10101	WORD	Arc_R02 용접구간 저장 시작워드
P1033F	BIT	R03 (OT48)
D18224	WORD	W100 R03 용접구간 카운터
R10201	WORD	Arc_R03 용접구간 저장 시작워드
P1043F	BIT	R04 (OT48)
R10301	WORD	Arc_R04 용접구간 저장 시작워드
P1053F	BIT	R05 (OT48)
P1063F	BIT	R06 (OT48)
R10501	WORD	Arc_R04 용접구간 저장 시작워드
T2106	BIT/WORD	W200 R05 용접시간 현재값
R10600	WORD	W700-3 R05 용접시간 저장 시작워드
R10601	WORD	Arc_R05 용접구간 저장 시작워드
T2107	BIT/WORD	W200 R06 용접시간 현재값
R10700	WORD	W200 R06 용접시간 저장 시작워드
R10701	WORD	Arc_R06 용접구간 저장 시작워드
T2108	BIT/WORD	W300 R05 용접시간 현재값
D15014.1	BIT	R-- Weld Count By_Pass On
R10800	WORD	W300 R05 용접시간 저장 시작워드
R10801	WORD	Arc_R05 용접구간 저장 시작워드
T2109	BIT/WORD	W300 R06 용접시간 현재값
D15014.2	BIT	R-- Weld Count By_Pass On
R10900	WORD	W300 R06 용접시간 저장 시작워드
R10901	WORD	Arc_R06 용접구간 저장 시작워드
T2110	BIT/WORD	W600 R-- 용접시간 현재값
D15014.3	BIT	R-- Weld Count By_Pass On
R11001	WORD	Arc_R-- 용접구간 저장 시작워드
T2111	BIT/WORD	W600 R-- 용접시간 현재값
D15014.4	BIT	R07 Weld Count By_Pass On
R11100	WORD	W600 R-- 용접시간 저장 시작워드
R11101	WORD	Arc_R-- 용접구간 저장 시작워드
T2112	BIT/WORD	W700 R-- 용접시간 현재값
D15014.5	BIT	R08 Weld Count By_Pass On
R11200	WORD	W700 R-- 용접시간 저장 시작워드
R11201	WORD	Arc_R079 용접구간 저장 시작워드
T2113	BIT/WORD	W700 R-- 용접시간 현재값
R11300	WORD	W700 R07 용접시간 저장 시작워드
R11301	WORD	Arc_R07 용접구간 저장 시작워드
D15014.6	BIT	R12 Weld Count By_Pass On
D15016.6	BIT	스캐너 By_Pass On
D15016.5	BIT	타각정보 수동입력
M00055	BIT	메인라인 도어열림
D00032	WORD	라인1 누설가스 설정시간
T2201	BIT/WORD	R01 누설가스 검출이상
M03901	BIT	R01 누설가스 검출이상
M03903	BIT	R02 누설가스 검출이상
M03905	BIT	R03 누설가스 검출이상
M03907	BIT	R04 누설가스 검출이상
M03909	BIT	R05 누설가스 검출이상
T2203	BIT/WORD	R02 누설가스 검출이상
T2205	BIT/WORD	R03 누설가스 검출이상
T2207	BIT/WORD	R04 누설가스 검출이상
T2209	BIT/WORD	R05 누설가스 검출이상
D00040	WORD	라인2 가스체크 설정시간
D00042	WORD	라인2 누설가스 설정시간
D00021	WORD	OP1 Touch Display Change 비밀번호
D25000	WORD	NG 버퍼
D25002	WORD	NG 슈트 버퍼
D18003	WORD	R01 표준시간 최대 용접시간
D18013	WORD	R02 표준시간 최대 용접시간
D18023	WORD	R03 표준시간 최대 용접시간
D18024	WORD	W100 R03 용접구간 카운터설정
D18033	WORD	R04 표준시간 최대 용접시간
D18004	WORD	W50 R01 용접구간 카운터설정
D15021.3	BIT	OP3 W70 Select Pb
D17541.0	BIT	W70 타각기 차종
D15016.1	BIT	W45 브러쉬 시프트 바이 패스
T0032	BIT/WORD	라인3 배기팬 Off Delay Tmr
D00092	WORD	라인3 배기팬 전원 상태
T2240	BIT/WORD	R01 Gas On 검출이상
T2241	BIT/WORD	R02 Gas On 검출이상
T2242	BIT/WORD	R03 Gas On 검출이상
T2243	BIT/WORD	R04 Gas On 검출이상
T2244	BIT/WORD	R05 Gas On 검출이상
T2245	BIT/WORD	R06 Gas On 검출이상
T2246	BIT/WORD	R-- Gas On 검출이상
T2247	BIT/WORD	R-- Gas On 검출이상
T2248	BIT/WORD	R-- Gas On 검출이상
D07001.7	BIT	SR01 용접팁교환 요구 LAMP
D07001.8	BIT	SR02 용접팁교환 요구 LAMP
D07004.1	BIT	R-- 용접팁교환 요구 LAMP
D07004.2	BIT	R-- 용접팁교환 요구 LAMP
D07004.3	BIT	R-- 용접팁교환 요구 LAMP
D07004.4	BIT	R07 용접팁교환 요구 LAMP
D07004.5	BIT	R08 용접팁교환 요구 LAMP
D07004.6	BIT	R12 용접팁교환 요구 LAMP
D06060	WORD	W200 R05 용접누락 판정결과
D06070	WORD	W200 R06 용접누락 판정결과
D06080	WORD	W300 R05 용접누락 판정결과
D06090	WORD	W300 R06 용접누락 판정결과
D06100	WORD	W600 R-- 용접누락 판정결과
D06110	WORD	W600 R-- 용접누락 판정결과
D06120	WORD	W700 R-- 용접누락 판정결과
D06130	WORD	W700 R-- 용접누락 판정결과
D01871	WORD	W500 G1 측정 1:OK 2:NG (W600)
D01872	WORD	W500 G2 측정 1:OK 2:NG (W600)
D01873	WORD	W500 G3 측정 1:OK 2:NG (W600)
D15007.D	BIT	로보트서보 Off lamp
M00036	BIT	Line Emergency Stop
D00001.F	BIT	Main 62405-S1510 4WD-디젤 RHD 비방청
M09970	BIT	R01 원점 확인 NG
M09960	BIT	R01 원점 확인 OK
M09961	BIT	R02 원점 확인 OK
M09971	BIT	R02 원점 확인 NG
M09962	BIT	R03 원점 확인 OK
M09972	BIT	R03 원점 확인 NG
M09963	BIT	R04 원점 확인 OK
M09973	BIT	R04 원점 확인 NG
M09964	BIT	R05 원점 확인 OK
M09974	BIT	R05 원점 확인 NG
M09965	BIT	R06 원점 확인 OK
M09975	BIT	R06 원점 확인 NG
M09966	BIT	R-- 원점 확인 OK
M09976	BIT	R-- 원점 확인 NG
M09967	BIT	R-- 원점 확인 OK
M09977	BIT	R-- 원점 확인 NG
D05706	WORD	R-- 전압 진행상태
D05716	WORD	R-- 전류 진행상태
D00070	WORD	NG 마스타 파트램프 상태1
D00071	WORD	NG 마스타 파트램프 상태2
D00072	WORD	NG 마스타 파트램프 상태3
D00073	WORD	NG 마스타 파트램프 상태4
D00074	WORD	NG 마스타 파트램프 상태5
D00075	WORD	NG 마스타 파트램프 상태6
D00076	WORD	NG 마스타 파트램프 상태7
D00077	WORD	NG 마스타 파트램프 상태8
D00078	WORD	NG 마스타 파트램프 상태9
D00079	WORD	NG 마스타 파트램프 상태10
D00080	WORD	NG 마스타 파트램프 상태11
D00081	WORD	NG 마스타 파트램프 상태12
D00082	WORD	NG 마스타 파트램프 상태13
R01900.2	BIT	R01 용접시간 NG
R01900.3	BIT	R01 용접구간 NG
R01900.4	BIT	R01 용접 시간/구간 NG
R01901.2	BIT	R02 용접시간 NG
R01901.3	BIT	R02 용접구간 NG
R01901.4	BIT	R02 용접 시간/구간 NG
R01902.2	BIT	R03 용접시간 NG
R01902.3	BIT	R03 용접구간 NG
R01902.4	BIT	R03 용접 시간/구간 NG
R01903.2	BIT	R04 용접시간 NG
R01903.3	BIT	R04 용접구간 NG
R01903.4	BIT	R04 용접 시간/구간 NG
R01904.2	BIT	R05 용접시간 NG
R01904.3	BIT	R05 용접구간 NG
R01904.4	BIT	R05 용접 시간/구간 NG
R01905.2	BIT	R06 용접시간 NG
R01905.3	BIT	R06 용접구간 NG
R01905.4	BIT	R06 용접 시간/구간 NG
R01906.2	BIT	R-- 용접시간 NG
R01906.3	BIT	R-- 용접구간 NG
R01906.4	BIT	R-- 용접 시간/구간 NG
R01907.2	BIT	R-- 용접시간 NG
R01907.3	BIT	R-- 용접구간 NG
R01907.4	BIT	R-- 용접 시간/구간 NG
R01908.2	BIT	R-- 용접시간 NG
R01908.3	BIT	R-- 용접구간 NG
R01908.4	BIT	R-- 용접 시간/구간 NG
R01909.2	BIT	R07 용접시간 NG
R01909.3	BIT	R07 용접구간 NG
R01909.4	BIT	R07 용접 시간/구간 NG
R01910.2	BIT	R08 용접시간 NG
R01910.3	BIT	R08 용접구간 NG
R01910.4	BIT	R08 용접 시간/구간 NG
R01911.2	BIT	R12 용접시간 NG
R01911.3	BIT	R12 용접구간 NG
R01911.4	BIT	R12 용접 시간/구간 NG
R01912.2	BIT	R13 용접시간 NG
R01912.3	BIT	R13 용접구간 NG
R01912.4	BIT	R13 용접 시간/구간 NG
R01913.2	BIT	R14 용접시간 NG
R01913.3	BIT	R14 용접구간 NG
R01913.4	BIT	R14 용접 시간/구간 NG
D15016.8	BIT	라인1 안전문 안전매트 By_Pass On
M0005F	BIT	라인 안전문 안전매트 이상
T0059	BIT/WORD	라인1 안전문3 안전매트 횟수RST 지연
T0041	BIT/WORD	라인1 안전문2 안전매트 검출유지 RST지연
D08500	WORD	R-- 표준시간 최소 용접시간 설정
D08540	WORD	R-- 표준시간 최소 용접시간 설정
D08580	WORD	R-- 표준시간 최소 용접시간 설정
D08620	WORD	R13 표준시간 최소 용접시간 설정
D08660	WORD	R15 표준시간 최소 용접시간 설정
D03410.0	BIT	서보 7 준비완료 (RD)
D00095	WORD	라인1 안전매트1 터치횟수
D00097	WORD	라인1 안전매트2 터치횟수
D00099	WORD	라인1 안전매트3 터치횟수
D00002.4	BIT	LX 프로젝트 차종 LHD 방청
D00002.2	BIT	TMC-S1000 2WD LHD 비방청
D00002.3	BIT	TMC-S1400 4WD LHD 비방청
M10076	BIT	R-- 노즐체크 NG
M10077	BIT	R-- 노즐체크 NG
M10078	BIT	R-- 노즐체크 NG
D00118	WORD	W50 파트램프 상태8
D00119	WORD	W50 파트램프 상태9
D00120	WORD	W50 파트램프 상태10
D00121	WORD	W50 파트램프 상태11
D00417	WORD	W200 파트램프 상태7
D00418	WORD	W200 파트램프 상태8
D00419	WORD	W200 파트램프 상태9
D15017.6	BIT	R06 원점체크 By_Pass On
D15017.7	BIT	SR01 원점체크 By_Pass On
D15017.8	BIT	SR02 원점체크 By_Pass On
D15018.1	BIT	R-- 원점체크 By_Pass On
D15018.2	BIT	R-- 원점체크 By_Pass On
D15018.3	BIT	R-- 원점체크 By_Pass On
D15018.4	BIT	R07 원점체크 By_Pass On
D15018.5	BIT	R08 원점체크 By_Pass On
D15018.6	BIT	R12 원점체크 By_Pass On
M1013C	BIT	R01 (IN45)
M1023C	BIT	R02 (IN45)
M1033C	BIT	R03 (IN45)
M1043C	BIT	R04 (IN45)
M1053C	BIT	R05 (IN45)
M1063C	BIT	R06 (IN45)
M0397A	BIT	NG마스타 주간 초품 체크 지령
M0397B	BIT	NG마스타 주간 중품 체크 지령
M0397C	BIT	NG마스타 야간 초품 체크 지령
M0397D	BIT	NG마스타 야간 중품 체크 지령
D15016.B	BIT	댐퍼미사용 By_Pass On
D18538	WORD	W700-> 파렛트적재 R-- HD2 버퍼
D18543	WORD	NG슈트 차종
D18566	WORD	W150-1  JIG변경 차종
D18567	WORD	W150-2  JIG변경 차종
D18501.0	BIT	W50 차종
D18503.0	BIT	W100 차종
D18505.0	BIT	W700-2 차종
D18513.0	BIT	W40 차종
D18521.0	BIT	W500 차종
D18523.0	BIT	W200 차종
D18527.0	BIT	W300 차종
D18529.0	BIT	W400 차종
M0501E	BIT	5라인 Display 표시창
M0501F	BIT	6라인 Display 표시창
D19740	WORD	5라인 잔여수량 Display 표시 
D19750	WORD	6라인 잔여수량 Display 표시 
K00115	BIT	W50 LWR 사양감지 체크완료
D00171	WORD	W50 LWR CHK Data.2 1:OK 2:NG
D00172	WORD	W50 UPR CHK Data.1 1:OK 2:NG
D00173	WORD	W50 UPR CHK Data.1 1:OK 2:NG
M05020	BIT	W50공정 작업수량 도달 차종교환 메세지
M10140	BIT	R01 (IN49)
M10240	BIT	R02 (IN49) 
M10340	BIT	R03 (IN49) 
M10440	BIT	R04 (IN49) 
M10540	BIT	R05 (IN49) 
M10640	BIT	R06 (IN49) 
D15016.2	BIT	W95 브러쉬 시프트 바이 패스
D15016.3	BIT	W250 브러쉬 시프트 바이 패스
D00122	WORD	W50 파트램프 상태12
M1636D	BIT	OP1 R13 Power ON Pb
M1636E	BIT	OP1 R14 Power ON Pb
M1657D	BIT	OP1 R13 Power On Lamp
M1657E	BIT	OP1 R14 Power On Lamp
M1657F	BIT	OP1 R15 Power On Lamp
M16581	BIT	OP1 R17 Power On Lamp
M16582	BIT	OP1 R18 Power On Lamp
M16583	BIT	OP1 R19 Power On Lamp
M16584	BIT	OP1 R20 Power On Lamp
M16585	BIT	OP1 R17 HD1 Power On Lamp
M16586	BIT	OP1 R18 HD2 Power On Lamp
M16587	BIT	OP1 R19 HD3 Power On Lamp
M16588	BIT	OP1 R20 HD4 Power On Lamp
M16589	BIT	OP1 R25 Power On Lamp
M1658E	BIT	OP1 R30 Power On Lamp
M16769	BIT	OP1 R-- 용접기 Power On Pb
M1676A	BIT	OP1 R07 용접기 Power On Pb
M1676B	BIT	OP1 R08 용접기 Power On Pb
M1676C	BIT	OP1 R12 용접기 Power On Pb
M1676D	BIT	OP1 R13 용접기 Power On Pb
M1676E	BIT	OP1 R14 용접기 Power On Pb
M16771	BIT	OP1 R20 HD4 용접기 Power On Pb
M16772	BIT	OP1 R18 용접기 Power On Pb
M16773	BIT	OP1 R19 용접기 Power On Pb
M16775	BIT	OP1 R17 HD1 용접기 Power On Pb
M16776	BIT	OP1 R18 HD2 용접기 Power On Pb
M16777	BIT	OP1 R19 HD3 용접기 Power On Pb
M16778	BIT	OP1 R20 HD4 용접기 Power On Pb
M16779	BIT	OP1 R25 용접기 Power On Pb
M1677A	BIT	OP1 R26 용접기 Power On Pb
M1677B	BIT	OP1 R27 용접기 Power On Pb
M1677C	BIT	OP1 R28 용접기 Power On Pb
M1677D	BIT	OP1 R29 용접기 Power On Pb
M1677E	BIT	OP1 R30 용접기 Power On Pb
M16979	BIT	OP1 R-- 용접기 Power On Lamp
M1697A	BIT	OP1 R07 용접기 Power On Lamp
M1697B	BIT	OP1 R08 용접기 Power On Lamp
M1697C	BIT	OP1 R12 용접기 Power On Lamp
M1697D	BIT	OP1 R13 용접기 Power On Lamp
M1697E	BIT	OP1 R14 용접기 Power On Lamp
M16981	BIT	OP1 R20 HD4 용접기 Power On Lamp
M16982	BIT	OP1 R18 용접기 Power On Lamp
M16983	BIT	OP1 R19 용접기 Power On Lamp
M16986	BIT	OP1 R18 HD2 용접기 Power On Lamp
M16987	BIT	OP1 R19 HD3 용접기 Power On Lamp
M16988	BIT	OP1 R20 HD4 용접기 Power On Lamp
M16989	BIT	OP1 R25 용접기 Power On Lamp
M1698A	BIT	OP1 R26 용접기 Power On Lamp
M1698B	BIT	OP1 R27 용접기 Power On Lamp
M1698C	BIT	OP1 R28 용접기 Power On Lamp
M1698D	BIT	OP1 R29 용접기 Power On Lamp
M1698E	BIT	OP1 R30 용접기 Power On Lamp
M1646D	BIT	OP1 R13 Power OFF Pb
M1646E	BIT	OP1 R14 Power OFF Pb
M16472	BIT	OP1 R18 Power OFF Pb
M16473	BIT	OP1 R19 Power OFF Pb
M16474	BIT	OP1 R20 Power OFF Pb
M16475	BIT	OP1 R17 HD1 Power OFF Pb
M16476	BIT	OP1 R18 HD2 Power OFF Pb
M16477	BIT	OP1 R19 HD3 Power OFF Pb
M16478	BIT	OP1 R20 HD4 Power OFF Pb
M16479	BIT	OP1 R25 Power OFF Pb
M1647E	BIT	OP1 R30 Power OFF Pb
M16869	BIT	OP1 R-- 용접기 Power OFF Pb
M1686A	BIT	OP1 R07 용접기 Power OFF Pb
M1686B	BIT	OP1 R08 용접기 Power OFF Pb
M1686C	BIT	OP1 R12 용접기 Power OFF Pb
M1686D	BIT	OP1 R13 용접기 Power OFF Pb
M1686E	BIT	OP1 R14 용접기 Power OFF Pb
M16871	BIT	OP1 R20 HD4 용접기 Power OFF Pb
M16872	BIT	OP1 R18 용접기 Power OFF Pb
M16873	BIT	OP1 R19 용접기 Power OFF Pb
M16875	BIT	OP1 R17 HD1 용접기 Power OFF Pb
M16876	BIT	OP1 R18 HD2 용접기 Power OFF Pb
M16877	BIT	OP1 R19 HD3 용접기 Power OFF Pb
M16878	BIT	OP1 R20 HD4 용접기 Power OFF Pb
M16879	BIT	OP1 R25 용접기 Power OFF Pb
M1687A	BIT	OP1 R26 용접기 Power OFF Pb
M1687B	BIT	OP1 R27 용접기 Power OFF Pb
M1687C	BIT	OP1 R28 용접기 Power OFF Pb
M1687D	BIT	OP1 R29 용접기 Power OFF Pb
M1687E	BIT	OP1 R30 용접기 Power OFF Pb
M03000	BIT	Servo 5  Auto Pb
M03001	BIT	Servo 5  Manual Pb
M03002	BIT	Servo 5 Jog + Pb
M03003	BIT	Servo 5 Jog - Pb
M03005	BIT	Servo 5  Home Pos. Set Pb
M03006	BIT	Servo 5  Position1 Select Pb
M03007	BIT	Servo 5  Position2 Select Pb
M03008	BIT	Servo 5  Position3 Select Pb
M03009	BIT	Servo 5  Position4 Select Pb
M0300A	BIT	Servo 5  Position5 Select Pb
M0300B	BIT	Servo 5  Position6 Select Pb
M0300C	BIT	Servo 5  Position7 Select Pb
M0300D	BIT	Servo 5  Position8 Select Pb
M03010	BIT	Servo 5  Auto Lamp
M03011	BIT	Servo 5  Manual Mode Lamp
M03015	BIT	Servo 5  Home Pos Set Comple
M03016	BIT	Servo 5  Position1 Select Comple
M03017	BIT	Servo 5  Position2 Select Comple
M03018	BIT	Servo 5  Position3 Select Comple
M03019	BIT	Servo 5  Position4 Select Comple
M0301A	BIT	Servo 5  Position5 Select Comple
M0301B	BIT	Servo 5  Position6 Select Comple
M0301C	BIT	Servo 5  Position7 Select Comple
M0301D	BIT	Servo 5  Position8 Select Comple
M03021	BIT	Servo 5 POS 1 (Home)
M03022	BIT	Servo 5 Pos 2 (Worker)
M03023	BIT	Servo 5 Pos 3 (1st Weld)
M03024	BIT	Servo 5 POS 4 (2nd Weld)
M03025	BIT	Servo 5 POS 5 (3rd Weld) 
M03026	BIT	Servo 5 POS 6 ()
M03027	BIT	Servo 5 POS 7 (Load'g)
M03028	BIT	Servo 5 POS 8 (Unload'g)
M0302C	BIT	Servo 5  Move Pb
M0302D	BIT	Servo 5 Copy From CV
M0302E	BIT	Servo 5 Copy from PV
M03031	BIT	Servo 5  Position 1 Select'g
M03032	BIT	Servo 5  Position2 Select'g
M03033	BIT	Servo 5  Position3 Select'g
M03034	BIT	Servo 5  Position4 Select'g
M03035	BIT	Servo 5  Position5 Select'g
M03036	BIT	Servo 5  Position6 Select'g
M03037	BIT	Servo 5  Position7 Select'g
M03038	BIT	Servo 5  Position8 Select'g
M03040	BIT	Servo 5 원점복귀 명령
M03041	BIT	Servo 5  Pos 1 Move
M03042	BIT	Servo 5  Pos2 Move
M03043	BIT	Servo 5  Pos3 Move
M03044	BIT	Servo 5  Pos4 Move
M03045	BIT	Servo 5  Pos5 Move
M03046	BIT	Servo 5  Pos6 Move
M03047	BIT	Servo 5  Pos7 Move
M03048	BIT	Servo 5  Pos8 Move
M03050	BIT	Servo 5  Auto Location Possible
M03051	BIT	Servo 5 수동선택
M03052	BIT	Servo 5 자동선택
M03053	BIT	Servo 5 이상해제
M03054	BIT	Servo 5 Power ON Check
M03061	BIT	Servo 5  Position 1 (Home) Move Commend
M03062	BIT	Servo 5  Position2 (Worker) Move Commend
M03063	BIT	Servo 5  Position3 (1st Weld) Move Commend
M03064	BIT	Servo 5  Position4 (2nd Weld) Move Commend
M03065	BIT	Servo 5  Position5 (3rd Weld) Move Commend
M03066	BIT	Servo 5  Position6()Move Commend
M03067	BIT	Servo 5  Position7 (Load'g) Move Commend
M03068	BIT	Servo 5  Position8 (Unload'g) Move Commend
M03100	BIT	Servo 6  Auto Pb
M03101	BIT	Servo 6  Manual Pb
M03102	BIT	Servo 6 Jog + Pb
M03103	BIT	Servo 6 Jog - Pb
M03105	BIT	Servo 6  Home Pos. Set Pb
M03106	BIT	Servo 6  Position1 Select Pb
M03107	BIT	Servo 6  Position2 Select Pb
M03108	BIT	Servo 6  Position3 Select Pb
M03109	BIT	Servo 6  Position4 Select Pb
M0310A	BIT	Servo 6  Position5 Select Pb
M0310B	BIT	Servo 6  Position6 Select Pb
M0310C	BIT	Servo 6  Position7 Select Pb
M0310D	BIT	Servo 6  Position8 Select Pb
M03110	BIT	Servo 6  Auto Lamp
M03111	BIT	Servo 6  Manual Mode Lamp
M03115	BIT	Servo 6  Home Pos Set Comple
M03116	BIT	Servo 6  Position1 Select Comple
M03117	BIT	Servo 6  Position2 Select Comple
M03118	BIT	Servo 6  Position3 Select Comple
M03119	BIT	Servo 6  Position4 Select Comple
M0311A	BIT	Servo 6  Position5 Select Comple
M0311B	BIT	Servo 6  Position6 Select Comple
M0311C	BIT	Servo 6  Position7 Select Comple
M0311D	BIT	Servo 6  Position8 Select Comple
M03121	BIT	Servo 6 POS 1 (Home)
M03122	BIT	Servo 6 Pos 2 (Worker)
M03123	BIT	Servo 6 Pos 3 (1st Weld'g)
M03124	BIT	Servo 6 POS 4 (2nd Weld'g) 
M03125	BIT	Servo 6 POS 5 (3rd Weld'g)
M03126	BIT	Servo 6 POS 6 ()
M03127	BIT	Servo 6 POS 7 (Load'g)
M03128	BIT	Servo 6 POS 8 (Unload'g)
M0312C	BIT	Servo 6  Move Pb
M0312D	BIT	Servo 6 Copy From CV
M0312E	BIT	Servo 6 Copy from PV
M03131	BIT	Servo 6  Position 1 Select'g
M03132	BIT	Servo 6  Position2 Select'g
M03133	BIT	Servo 6  Position3 Select'g
M03134	BIT	Servo 6  Position4 Select'g
M03135	BIT	Servo 6  Position5 Select'g
M03136	BIT	Servo 6  Position6 Select'g
M03137	BIT	Servo 6  Position7 Select'g
M03138	BIT	Servo 6  Position8 Select'g
M03140	BIT	Servo 6 원점복귀 명령
M03141	BIT	Servo 6  Pos 1 Move
M03142	BIT	Servo 6  Pos2 Move
M03143	BIT	Servo 6  Pos3 Move
M03144	BIT	Servo 6  Pos4 Move
M03145	BIT	Servo 6  Pos5 Move
M03146	BIT	Servo 6  Pos6 Move
M03147	BIT	Servo 6  Pos7 Move
M03148	BIT	Servo 6  Pos8 Move
M03150	BIT	Servo 6  Auto Location Possible
M03151	BIT	Servo 6 수동선택
M03152	BIT	Servo 6 자동선택
M03153	BIT	Servo 6 이상해제
M03154	BIT	Servo 6 Power ON Check
M03161	BIT	Servo 6  Position 1 (Home) Move Commend
M03162	BIT	Servo 6  Position2 (Worer) Move Commend
M03163	BIT	Servo 6  Position3 (1st Weld) Move Commend
M03164	BIT	Servo 6  Position4 (2nd Weld) Move Commend
M03165	BIT	Servo 6  Position5 (3rd Weld) Move Commend
M03166	BIT	Servo 6  Position6()Move Commend
M03167	BIT	Servo 6  Position7 (Load'g) Move Commend
M03168	BIT	Servo 6  Position8 (Unload) Move Commend
M03200	BIT	Servo 7  Auto Pb
M03201	BIT	Servo 7  Manual Pb
M03202	BIT	Servo 7 Jog + Pb
M03203	BIT	Servo 7 Jog - Pb
M03205	BIT	Servo 7  Home Pos. Set Pb
M03206	BIT	Servo 7  Position1 Select Pb
M03207	BIT	Servo 7  Position2 Select Pb
M03208	BIT	Servo 7  Position3 Select Pb
M03209	BIT	Servo 7  Position4 Select Pb
M0320A	BIT	Servo 7  Position5 Select Pb
M0320B	BIT	Servo 7  Position6 Select Pb
M0320C	BIT	Servo 7  Position7 Select Pb
M0320D	BIT	Servo 7  Position8 Select Pb
M03210	BIT	Servo 7  Auto Lamp
M03211	BIT	Servo 7  Manual Mode Lamp
M03215	BIT	Servo 7  Home Pos Set Comple
M03216	BIT	Servo 7  Position1 Select Comple
M03217	BIT	Servo 7  Position2 Select Comple
M03218	BIT	Servo 7  Position3 Select Comple
M03219	BIT	Servo 7  Position4 Select Comple
M0321A	BIT	Servo 7  Position5 Select Comple
M0321B	BIT	Servo 7  Position6 Select Comple
M0321C	BIT	Servo 7  Position7 Select Comple
M0321D	BIT	Servo 7  Position8 Select Comple
M03221	BIT	Servo 7 POS 1 (Home)
M03222	BIT	Servo 7 Pos 2 (Worker)
M03223	BIT	Servo 7 Pos 3 (1st Weld)
M03224	BIT	Servo 7 POS 4 (2nd Weld)
M03225	BIT	Servo 7 POS 5 (3rd Weld)
M03226	BIT	Servo 7 POS 6 ()
M03227	BIT	Servo 7 POS 7 (Load'g)
M03228	BIT	Servo 7 POS 8 (Unload'g)
M0322C	BIT	Servo 7  Move Pb
M0322D	BIT	Servo 7 Copy From CV
M0322E	BIT	Servo 7 Copy from PV
M03231	BIT	Servo 7  Position 1 Select'g
M03232	BIT	Servo 7  Position2 Select'g
M03233	BIT	Servo 7  Position3 Select'g
M03234	BIT	Servo 7  Position4 Select'g
M03235	BIT	Servo 7  Position5 Select'g
M03236	BIT	Servo 7  Position6 Select'g
M03237	BIT	Servo 7  Position7 Select'g
M03238	BIT	Servo 7  Position8 Select'g
M03240	BIT	Servo 7 원점복귀 명령
M03241	BIT	Servo 7  Pos 1 Move
M03242	BIT	Servo 7  Pos2 Move
M03243	BIT	Servo 7  Pos3 Move
M03244	BIT	Servo 7  Pos4 Move
M03245	BIT	Servo 7  Pos5 Move
M03246	BIT	Servo 7  Pos6 Move
M03247	BIT	Servo 7  Pos7 Move
M03248	BIT	Servo 7  Pos8 Move
M03250	BIT	Servo 7  Auto Location Possible
M03251	BIT	Servo 7 수동선택
M03252	BIT	Servo 7 자동선택
M03253	BIT	Servo 7 이상해제
M03254	BIT	Servo 7 Power ON Check
M03261	BIT	Servo 7  Position 1 (Home) Move Commend
M03262	BIT	Servo 7  Position2 (Worker) Move Commend
M03263	BIT	Servo 7  Position3 (1st Weld) Move Commend
M03264	BIT	Servo 7  Position4 (2nd Weld) Move Commend
M03265	BIT	Servo 7  Position5 (3rd Weld) Move Commend
M03266	BIT	Servo 7  Position6()Move Commend
M03267	BIT	Servo 7  Position7 (Load'g) Move Commend
M03268	BIT	Servo 7  Position8 (Unload'g) Move Commend
D03000	WORD	서보 5 현재 위치 데이타 Low
D03014	WORD	서보 5 Table 1 위치 데이타 Low
D03036	WORD	서보 5 이상 코드 Low
D03038	WORD	서보 5 통신 하트 비트 리턴 Low
D03040	WORD	서보 5 Mode (0=자동, 1=수동)
D03041	WORD	서보 5 통신 체크용 스캔 카운터
D03050	WORD	서보 5 등록 포지션 1번 Low
D03052	WORD	서보 5 등록 포지션 2번 Low
D03054	WORD	서보 5 등록 포지션 3번 Low
D03056	WORD	서보 5 등록 포지션 4번 Low
D03058	WORD	서보 5 등록 포지션 5번 Low
D03060	WORD	서보 5 사용자 입력 위치 데이타1 Low
D03062	WORD	서보 5 사용자 입력 위치 데이타2 Low
D03064	WORD	서보 5 사용자 입력 위치 데이타3 Low
D03070	WORD	서보 5 등록 포지션 1번 Low Band Low
D03072	WORD	서보 5 등록 포지션 2번 Low Band Low
D03074	WORD	서보 5 등록 포지션 3번 Low Band Low
D03076	WORD	서보 5 등록 포지션 4번 Low Band Low
D03078	WORD	서보 5 등록 포지션 5번 Low Band Low
D03080	WORD	서보 5 등록 포지션 1번 High Band Low
D03082	WORD	서보 5 등록 포지션 2번 High Band Low
D03084	WORD	서보 5 등록 포지션 3번 High Band Low
D03086	WORD	서보 5 등록 포지션 4번 High Band Low
D03088	WORD	서보 5 등록 포지션 5번 High Band Low
D03102	WORD	서보 5 Table 1 위치 데이타 Low
D03104	WORD	서보 5 Table 1 위치 결정 속도 Low
D03106	WORD	서보 5 예약
D03108	WORD	서보 5 예약
D03138	WORD	서보 5 통신 하트 비트 Low
D03200	WORD	서보 6 현재 위치 데이타 Low
D03214	WORD	서보 6 Table 1 위치 데이타 Low
D03236	WORD	서보 6 이상 코드 Low
D03238	WORD	서보 6 통신 하트 비트 리턴 Low
D03240	WORD	서보 6 Mode (0=자동, 1=수동)
D03241	WORD	서보 6 통신 체크용 스캔 카운터
D03250	WORD	서보 6 등록 포지션 1번 Low
D03252	WORD	서보 6 등록 포지션 2번 Low
D03254	WORD	서보 6 등록 포지션 3번 Low
D03256	WORD	서보 6 등록 포지션 4번 Low
D03258	WORD	서보 6 등록 포지션 5번 Low
D03260	WORD	서보 6 사용자 입력 위치 데이타 Low
D03262	WORD	서보 6 등록 포지션 7번 Low
D03264	WORD	서보 6 등록 포지션 8번 Low
D03270	WORD	서보 6 등록 포지션 1번 Low Band Low
D03272	WORD	서보 6 등록 포지션 2번 Low Band Low
D03274	WORD	서보 6 등록 포지션 3번 Low Band Low
D03276	WORD	서보 6 등록 포지션 4번 Low Band Low
D03278	WORD	서보 6 등록 포지션 5번 Low Band Low
D03280	WORD	서보 6 등록 포지션 1번 High Band Low
D03282	WORD	서보 6 등록 포지션 2번 High Band Low
D03284	WORD	서보 6 등록 포지션 3번 High Band Low
D03286	WORD	서보 6 등록 포지션 4번 High Band Low
D03288	WORD	서보 6 등록 포지션 5번 High Band Low
D03302	WORD	서보 6 Table 1 위치 데이타 Low
D03304	WORD	서보 6 Table 1 위치 결정 속도 Low
D03306	WORD	서보 6 예약
D03308	WORD	서보 6 예약
D03008.6	BIT	서보 5 리셋 (RES) 리턴
D03009.1	BIT	서보 5 자동/수동 선택 (MD0) 리턴
D03009.3	BIT	서보 5 포인트 테이블 No. 선택1 (DI0) 리턴
D03009.4	BIT	서보 5 포인트 테이블 No. 선택2 (DI1) 리턴
D03009.5	BIT	서보 5 포인트 테이블 No. 선택3 (DI2) 리턴
D03009.6	BIT	서보 5 포인트 테이블 No. 선택4 (DI3) 리턴
D03009.D	BIT	서보 5 포인트 테이블 No. 선택5 (DI4) 리턴
D03010.0	BIT	서보 5 준비완료 (RD)
D03010.8	BIT	서보 5 고장 (ALM)
D03011.1	BIT	서보 5 원점복귀완료 (ZP)
D03011.C	BIT	서보 5 이동완료 (MEND)
D03100.0	BIT	서보 5 서보 ON (SON)
D03100.1	BIT	서보 5 정전스트로크엔드 (LSP)
D03100.2	BIT	서보 5 역전스트로크엔드 (LSN)
D03100.6	BIT	서보 5 리셋 (RES)
D03100.B	BIT	서보 5 정전 시동 (ST1)
D03100.C	BIT	서보 5 역전 시동 (ST2)
D03101.1	BIT	서보 5 자동/수동 선택 (MD0)
D03101.3	BIT	서보 5 포인트 테이블 No. 선택1 (DI0)
D03101.4	BIT	서보 5 포인트 테이블 No. 선택2 (DI1)
D03101.5	BIT	서보 5 포인트 테이블 No. 선택3 (DI2)
D03101.6	BIT	서보 5 포인트 테이블 No. 선택4 (DI3)
D03101.D	BIT	서보 5 포인트 테이블 No. 선택5 (DI4)
D03208.6	BIT	서보 6 리셋 (RES) 리턴
D03209.1	BIT	서보 6 자동/수동 선택 (MD0) 리턴
D03209.3	BIT	서보 6 포인트 테이블 No. 선택1 (DI0) 리턴
D03209.4	BIT	서보 6 포인트 테이블 No. 선택2 (DI1) 리턴
D03209.5	BIT	서보 6 포인트 테이블 No. 선택3 (DI2) 리턴
D03209.6	BIT	서보 6 포인트 테이블 No. 선택4 (DI3) 리턴
D03209.D	BIT	서보 6 포인트 테이블 No. 선택5 (DI4) 리턴
D03210.0	BIT	서보 6 준비완료 (RD)
D03210.8	BIT	서보 6 고장 (ALM)
D03211.1	BIT	서보 6 원점복귀완료 (ZP)
D03211.C	BIT	서보 6 이동완료 (MEND)
D03300.0	BIT	서보 6 서보 ON (SON)
D03300.1	BIT	서보 6 정전스트로크엔드 (LSP)
D03300.2	BIT	서보 6 역전스트로크엔드 (LSN)
D03300.6	BIT	서보 6 리셋 (RES)
D03300.B	BIT	서보 6 정전 시동 (ST1)
D03300.C	BIT	서보 6 역전 시동 (ST2)
D03301.1	BIT	서보 6 자동/수동 선택 (MD0)
D03301.3	BIT	서보 6 포인트 테이블 No. 선택1 (DI0)
D03301.4	BIT	서보 6 포인트 테이블 No. 선택2 (DI1)
D03301.5	BIT	서보 6 포인트 테이블 No. 선택3 (DI2)
D03301.6	BIT	서보 6 포인트 테이블 No. 선택4 (DI3)
D03301.D	BIT	서보 6 포인트 테이블 No. 선택5 (DI4)
D04020	WORD	T1500 라벨보관함 파트램프
D04021	WORD	S1250 라벨보관함 파트램프
D04022	WORD	S1100 라벨보관함 파트램프
D04023	WORD	S1350 라벨보관함 파트램프
D04024	WORD	S1400 라벨보관함 파트램프
D04025	WORD	S1650 라벨보관함 파트램프
D04026	WORD	S1500 라벨보관함 파트램프
D04027	WORD	S1750 라벨보관함 파트램프
D04028	WORD	S1850 라벨보관함 파트램프
D04029	WORD	S1950 라벨보관함 파트램프
D04030	WORD	S1010 라벨보관함 파트램프
D04031	WORD	S1110 라벨보관함 파트램프
D04032	WORD	S1360 라벨보관함 파트램프
D04033	WORD	S1410 라벨보관함 파트램프
D04034	WORD	S1660 라벨보관함 파트램프
D04035	WORD	S1510 라벨보관함 파트램프
D04036	WORD	S1760 라벨보관함 파트램프
D04037	WORD	S1860 라벨보관함 파트램프
D04038	WORD	S1960 라벨보관함 파트램프
T0601	BIT/WORD	W400 수동 Mode Tmr
T0602	BIT/WORD	W400 자동 Mode Tmr
T0611	BIT/WORD	W400 공압이상 지연 타이머
T0612	BIT/WORD	W400 로보트 간섭무지연
T0622	BIT/WORD	W400 MBR 2번 파트없음 지연
T0623	BIT/WORD	W400 MBR 2번 파트 OK지연
T0624	BIT/WORD	W400 MBR 3번 파트없음 지연
T0625	BIT/WORD	W400 MBR 3번 파트 OK지연
T0631	BIT/WORD	W400-1 냉각동작 시간
T0632	BIT/WORD	W400-2 냉각동작 시간
T0633	BIT/WORD	W400-3 냉각동작 시간
D00600	WORD	W400 공정표시
D00611	WORD	W400 파트램프 상태1
D00612	WORD	W400 파트램프 상태2
D00613	WORD	W400 파트램프 상태3
D00614	WORD	W400 파트램프 상태4
D00615	WORD	W400 파트램프 상태5
D00616	WORD	W400 파트램프 상태6
P03001	BIT	OP1 수동 선택
P03005	BIT	OP1 부저 정지
P03009	BIT	OP1 CAM S/W 선택 BIT2
P0300A	BIT	OP1 CAM S/W 선택 BIT4
P0300B	BIT	OP1 CAM S/W 선택 BIT8
P03021	BIT	OP2 수동 선택
P03025	BIT	OP2 부저 정지
P03029	BIT	OP2 CAM S/W 선택 BIT2
P0302A	BIT	OP2 CAM S/W 선택 BIT4
P0302B	BIT	OP2 CAM S/W 선택 BIT8
P0030E	BIT	W10 LH 1차 클램프 잠김2
P00317	BIT	W10 LH 3차 클램프 풀림1
P00318	BIT	W10 LH 3차 클램프 잠김2
P00319	BIT	W10 LH 3차 클램프 풀림2
P02300	BIT	W65 클램프 전진1
P02301	BIT	W65 클램프 후진1
P02302	BIT	W65 클램프 전진2
P02303	BIT	W65 클램프 후진2
P02304	BIT	W65 제품확인1 UPR
P02307	BIT	W65 공기압력
P0230A	BIT	W60 브러쉬1 BLDC - 이상
P0230B	BIT	W60 브러쉬2 BLDC - 이상
P02320	BIT	W65 클램프 전진 Sol
P02321	BIT	W65 클램프 후진 Sol
P02326	BIT	W60 브러쉬1 BLDC - 역회전
P0232A	BIT	W60 브러쉬2 BLDC - 역회전
P0232D	BIT	W65 에어 분사 Sol
P0232F	BIT	W65 잔압배기 Sol
P0240E	BIT	타각기 작업완료
P0240F	BIT	타각기 이상
P02416	BIT	W70 제품확인7 PIPE
P0242D	BIT	타각기 이상해제
P02500	BIT	W80-1 클램프 전진1
P02501	BIT	W80-1 클램프 후진1
P02509	BIT	W80-1 제품확인1 SIDE MBR
P02510	BIT	W80-1 턴포인트 1
P02511	BIT	W80-1 턴포인트 2
P02512	BIT	W80-1 턴포인트 3
P02513	BIT	W80-1 턴포인트 4
P02517	BIT	W80-1 공기압력
P02518	BIT	W80-1 발판스위치 Jog+
P02519	BIT	W80-1 발판스위치 Jog-
P0251A	BIT	W80-1 광 안전장치1
P0251B	BIT	W80-1 광 안전장치2
P0251C	BIT	W80-1 기동-L
P0251D	BIT	W80-1 기동-R
P0251E	BIT	W80-1 원점복귀
P0251F	BIT	W80-1 비상정지
P02520	BIT	W80-1 클램프 전진 Sol
P02521	BIT	W80-1 클램프 후진 Sol
P0252D	BIT	W80-1 에어 분사 Sol
P0252F	BIT	W80-1 잔압배기 Sol
P02600	BIT	W80-2 클램프 전진1
P02601	BIT	W80-2 클램프 후진1
P02609	BIT	W80-2 제품확인1 SIDE MBR
P02610	BIT	W80-2 턴포인트 1
P02611	BIT	W80-2 턴포인트 2
P02612	BIT	W80-2 턴포인트 3
P02613	BIT	W80-2 턴포인트 4
P02617	BIT	W80-2 공기압력
P02618	BIT	W80-2 발판스위치 Jog+
P02619	BIT	W80-2 발판스위치 Jog-
P0261A	BIT	W80-2 광 안전장치1
P0261B	BIT	W80-2 광 안전장치2
P0261C	BIT	W80-2 기동-L
P0261D	BIT	W80-2 기동-R
P0261E	BIT	W80-2 원점복귀
P0261F	BIT	W80-2 비상정지
P02620	BIT	W80-2 클램프 전진 Sol
P02621	BIT	W80-2 클램프 후진 Sol
P0262D	BIT	W80-2 에어 분사 Sol
P0262F	BIT	W80-2 잔압배기 Sol
P02700	BIT	파렛트-A 클램프 잠김
P02701	BIT	파렛트-A 클램프 풀림
P02702	BIT	파렛트-A 배출 전진
P02703	BIT	파렛트-A 배출 후진
P02704	BIT	파렛트-A 배출 전진
P02705	BIT	파렛트-A 배출 후진
P02706	BIT	파렛트-A 안전 플러그
P02707	BIT	파렛트-A 광 안전장치
P02708	BIT	파렛트-A 배출 기동
P02709	BIT	파렛트-A 파렛트 감지_1
P0270A	BIT	파렛트-A 파렛트 감지_2
P0270B	BIT	파렛트-A 자동/수동
P0270C	BIT	파렛트-A 기동
P0270D	BIT	파렛트-A 클램프 잠김
P0270E	BIT	파렛트-A 클램프 풀림
P0270F	BIT	파렛트-A 비상정지
P02710	BIT	파렛트-B 클램프 잠김
P02711	BIT	파렛트-B 클램프 풀림
P02712	BIT	파렛트-B 배출 전진
P02713	BIT	파렛트-B 배출 후진
P02714	BIT	파렛트-B 배출 전진
P02715	BIT	파렛트-B 배출 후진
P02716	BIT	파렛트-B 안전 플러그
P02717	BIT	파렛트-B 광 안전장치
P02718	BIT	파렛트-B 배출 기동
P02719	BIT	파렛트-B 파렛트 감지_1
P0271A	BIT	파렛트-B 파렛트 감지_2
P0271B	BIT	파렛트-B 자동/수동
P0271C	BIT	파렛트-B 기동
P0271D	BIT	파렛트-B 클램프 잠김
P0271E	BIT	파렛트-B 클램프 풀림
P0271F	BIT	파렛트-B 비상정지
P02720	BIT	불량DIE 클램프 잠김
P02721	BIT	불량DIE 클램프 풀림
P0272C	BIT	불량DIE 기동
P02740	BIT	파렛트-A 클램프 잠김 Sol
P02741	BIT	파렛트-A 클램프 풀림 Sol
P02742	BIT	파렛트-A 배출 전진 Sol
P02743	BIT	파렛트-A 배출 후진 Sol
P02748	BIT	파렛트-A 기동
P02749	BIT	파렛트-A Tower Lamp_R
P0274A	BIT	파렛트-A Tower Lamp_Y
P0274B	BIT	파렛트-A Tower Lamp_G
P0274C	BIT	파렛트-A Tower Lamp_B
P0274E	BIT	불량DIE 클램프 잠김 Sol
P0274F	BIT	불량DIE 클램프 풀림 Sol
P02760	BIT	파렛트-B 클램프 잠김 Sol
P02761	BIT	파렛트-B 클램프 풀림 Sol
P02762	BIT	파렛트-B 배출 전진 Sol
P02763	BIT	파렛트-B 배출 후진 Sol
P02768	BIT	파렛트-B 기동
P02769	BIT	파렛트-B Tower Lamp_R
P0276A	BIT	파렛트-B Tower Lamp_Y
P0276B	BIT	파렛트-B Tower Lamp_G
P0276C	BIT	파렛트-B Tower Lamp_B
P1012F	BIT	R01 (OT32)
P1032F	BIT	R03 (OT32)
P1042F	BIT	R04 (OT32)
P1052F	BIT	R05 (OT32)
P1062F	BIT	R06 (OT32)
M1697F	BIT	OP1 R15 용접기 Power On Lamp
M16980	BIT	OP1 R16 용접기 Power On Lamp
D15001.6	BIT	OP1 STN06 Select Pb
D15001.7	BIT	OP1 STN07 Select Pb
T0354	BIT/WORD	W20 LH 에어블로우 ON
T0374	BIT/WORD	W20 LH 에어블로우 OFF
T0454	BIT/WORD	W20 RH 에어블로우 ON
T0474	BIT/WORD	W20 RH 에어블로우 OFF
M0027A	BIT	W10 RH 2차 작업준비
P1031C	BIT	R03 (OT13)
P1031D	BIT	R03 (OT14)
P1041D	BIT	R04 (OT14)
T0634	BIT/WORD	W400-4 냉각동작 시간
T0626	BIT/WORD	W400 MBR 4번 파트없음 지연
T0627	BIT/WORD	W400 MBR 4번 파트 OK지연
T0716	BIT/WORD	W100 파트이상 (누락)지연
T0717	BIT/WORD	W100 사양감지 체크완료 지연
M0017A	BIT	W10 LH 2차 작업준비
M00826	BIT	W150-1 파트체크 정상
M00827	BIT	W150-1 차종감지 파트정상
M00832	BIT	W150-1 기동 Pulse
M00842	BIT	W150-1 언로딩 로보트 간섭무
M00843	BIT	W150-1 Work Robot 간섭무
M00870	BIT	W150-1 기동준비
M00871	BIT	W150-1 1차 기동
M00872	BIT	W150-1 2차 기동
M00873	BIT	W150-1 3차 기동
M00874	BIT	W150-1 4차 기동
M00879	BIT	W150-1 1차 작업준비
M0087A	BIT	W150-1 2차 작업준비
M00881	BIT	W150-1 1차 기동 End
M00882	BIT	W150-1 2차 기동 End
M00883	BIT	W150-1 3차 기동 End
T0803	BIT/WORD	W150-1 Air Blow On TMR
T0812	BIT/WORD	W150-1 로보트 간섭무지연
T0816	BIT/WORD	W150-1 파트이상 (누락)지연
T0830	BIT/WORD	W150-1 양수기동 이상지연
M00830	BIT	W150-1 양수기동 이상
M00831	BIT	W150-1 Anti-Repeat
M0082F	BIT	W150-1 차광막 하강/상승
M00927	BIT	W200 차종감지 파트정상
M0092F	BIT	W200 차광막 하강/상승
M00930	BIT	W200 양수기동 이상
M00931	BIT	W200 Anti-Repeat
M00974	BIT	W200 4차 기동
K00915	BIT	W700 LWR 사양감지 체크완료
K00916	BIT	W700 UPR 사양감지 체크완료
T0916	BIT/WORD	W200 파트이상 (누락)지연
T0917	BIT/WORD	W200 사양감지 체크완료 지연
T0930	BIT/WORD	W200 양수기동 이상지연
D15021.1	BIT	OP3 W60 Select Pb
M03159	BIT	Foot S/W 사용함
M03156	BIT	Servo 6 Foot S/W + Aux
M03157	BIT	Servo 6 Foot S/W - Aux
M03259	BIT	Foot S/W 사용함
M03258	BIT	Servo 7 Foot S/W Control Mode
M03158	BIT	Servo 6 Foot S/W Control Mode
M03256	BIT	Servo 7 Foot S/W + Aux
M03257	BIT	Servo 7 Foot S/W - Aux
M1646F	BIT	OP1 R15 Power OFF Pb
M16470	BIT	OP1 R16 Power OFF Pb
M1636F	BIT	OP1 R15 Power ON Pb
M16471	BIT	OP1 R17 Power OFF Pb
M1686F	BIT	OP1 R15 용접기 Power OFF Pb
M1676F	BIT	OP1 R15 용접기 Power On Pb
M16770	BIT	OP1 R16 용접기 Power On Pb
M16870	BIT	OP1 R16 용접기 Power OFF Pb
M1626A	BIT	OP1 R07 Select Pb
M1626B	BIT	OP1 R08 Select Pb
M1626C	BIT	OP1 R12 Select Pb
M1626D	BIT	OP1 R13 Select Pb
M1626E	BIT	OP1 R14 Select Pb
M1626F	BIT	OP1 R15 Select Pb
M1628A	BIT	OP1 R07 Seleted
M1628B	BIT	OP1 R08 Seleted
M1628C	BIT	OP1 R12 Seleted
M1628D	BIT	OP1 R13 Seleted
M1628E	BIT	OP1 R14 Seleted
M1628F	BIT	OP1 R15 Seleted
M16309	BIT	OP2 R-- Select Pb
M1630A	BIT	OP2 R-- Select Pb
M1630B	BIT	OP2 R-- Select Pb
M1630C	BIT	OP2 R-- Select Pb
M16329	BIT	OP2 R-- Seleted
M1632A	BIT	OP2 R-- Seleted
M1632B	BIT	OP2 R-- Seleted
M1632C	BIT	OP2 R-- Seleted
M16344	BIT	OP3 R04 Select Pb
M16345	BIT	OP3 R05 Select Pb
M16346	BIT	OP3 R06 Select Pb
M16347	BIT	OP3 R-- Select Pb
M16348	BIT	OP3 R-- Select Pb
M16349	BIT	OP3 R-- Select Pb
M1634A	BIT	OP3 R07 Select Pb
M1634B	BIT	OP3 R08 Select Pb
M1634C	BIT	OP3 R12 Select Pb
M1634D	BIT	OP3 R13 Select Pb
M1634E	BIT	OP3 R14 Select Pb
M1634F	BIT	OP3 R15 Select Pb
P10429	BIT	R04 (OT26)
M0057A	BIT	W30 2차 작업준비
P10629	BIT	R06 (OT26)
M16040	BIT	OP3 Robot SERVO_ON PB/XP
M16041	BIT	OP3 Robot REMOTE PB/XP
M16042	BIT	OP3 Robot PLAY PB/XP
M16043	BIT	OP3 Robot RUN /XP
M16044	BIT	OP3 Robot WELD PB/XP
M16045	BIT	OP3 Robot ERROR RESET PB/XP
M16046	BIT	OP3 Robot LOCAL PB/XP
M16047	BIT	OP3 Robot TEACH PB/XP
M16048	BIT	OP3 Robot PAUSE PB/XP
M16049	BIT	OP3 Robot Power On PB/XP
P10330	BIT	R03 (OT33)
P1052A	BIT	R05 (OT27)
P1062A	BIT	R06 (OT27)
P0276D	BIT	불량DIE Tower Lamp_R
P0276E	BIT	불량DIE Tower Lamp_G
K04295	BIT	NG 슈트 로딩 완료
K04296	BIT	NG 슈트 로딩완료 해제
P0276F	BIT	불량DIE Tower Lamp_B
P0272D	BIT	불량DIE 클램프 잠김 SPB
P0272E	BIT	불량DIE 클램프 풀림 SPB
P02725	BIT	불량DIE 확인    1
P02726	BIT	불량DIE 확인    2
P02724	BIT	불량DIE 제품 안착확인 1
T4249	BIT/WORD	NG 슈트 락킹 잠김완료
T4269	BIT/WORD	NG 슈트 락킹 풀림 완료
D15016.4	BIT	타각기 By_Pass On
D00198	WORD	메인3 안전문 안전매트 터치 횟수
T0062	BIT/WORD	라인1 안전문3 안전매트 이상지연
T0063	BIT/WORD	라인1 안전문3 안전매트 횟수RST 지연
D15021.4	BIT	OP3 80-1 Select Pb
D15021.5	BIT	OP3 80-2 Select Pb
D15021.6	BIT	OP3 STN6 Select Pb
D15021.7	BIT	OP3 Pallet Select Pb
M04727	BIT	-
P02418	BIT	W70 제품확인09 PIPE (LH ONLY)
P02419	BIT	W70 제품확인 MAIN LS
M16985	BIT	OP1 수동 용접기2 Power On Lamp
M02356	BIT	Servo 4 Foot S/W + Aux
M02357	BIT	Servo 4 Foot S/W - Aux
M02358	BIT	Servo 4 Foot S/W Control Mode
M02359	BIT	Foot S/W 사용함
D15016.9	BIT	라인 안전문2 안전매트 By_Pass On
D15016.A	BIT	라인 안전문3 안전매트 By_Pass On
T0050	BIT/WORD	라인 안전문1 안전매트 이상지연 (W50)
T0052	BIT/WORD	라인 안전문3 안전매트 이상지연
D00096	WORD	라인1 안전문2 안전매트 터치 횟수
M0003B	BIT	라인1 안전문2 안전매트 검출
M0003E	BIT	라인1 안전문2 안전매트 검출유지
M0003A	BIT	라인1 안전문1 안전매트 검출
M0003D	BIT	라인1 안전문1 안전매트 검출유지
T0040	BIT/WORD	라인1 안전문1 안전매트 검출유지 RST지연
D00094	WORD	라인1 안전문1 안전매트 터치 횟수
P0260C	BIT	라인2 안전문2 안전매트
D00098	WORD	라인1 안전문3 안전매트 터치 횟수
M0003C	BIT	라인1 안전문3 안전매트 검출
M0003F	BIT	라인1 안전문3 안전매트 검출유지
T0042	BIT/WORD	라인1 안전문3 안전매트 검출유지 RST지연
P0260D	BIT	안전문2. 플러그 1 외부
P0260E	BIT	안전문2. 플러그 2 개방
P0260F	BIT	안전문2. 플러그 내부
T0057	BIT/WORD	라인2 메인에어 압력 이상
T0058	BIT/WORD	라인2 메인가스 압력저하 이상
D08810.3	BIT	R-- 노즐청소 카운터 리셋PB
D08810.4	BIT	R07 노즐청소 카운터 리셋PB
D08810.5	BIT	R08 노즐청소 카운터 리셋PB
D08810.6	BIT	R12 노즐청소 카운터 리셋PB
D08810.7	BIT	R13 노즐청소 카운터 리셋PB
D08810.8	BIT	R14 노즐청소 카운터 리셋PB
D08810.1	BIT	R-- 노즐청소 카운터 리셋PB
D08810.2	BIT	R-- 노즐청소 카운터 리셋PB
D08810.9	BIT	R15 노즐청소 카운터 리셋PB
D08810.A	BIT	R16 노즐청소 카운터 리셋PB
D08830	WORD	R-- 노즐청소 설정
D08810.F	BIT	OP2 노즐청소 카운터 전체리셋  PB
D07003.7	BIT	R13 용접팁교환 요구 PB
D07003.8	BIT	R14 용접팁교환 요구 PB
D07003.9	BIT	R15 용접팁교환 요구 PB
D07003.A	BIT	R16 용접팁교환 요구 PB
D07004.7	BIT	R13 용접팁교환 요구 LAMP
D07004.8	BIT	R14 용접팁교환 요구 LAMP
D07004.9	BIT	R15 용접팁교환 요구 LAMP
D07004.A	BIT	R16 용접팁교환 요구 LAMP
D08822	WORD	R-- 노즐청소 설정
D08824	WORD	R-- 노즐청소 설정
M08807	BIT	R-- 노즐청소 진입중
M08808	BIT	R-- 노즐청소 진입중
M08817	BIT	R-- 노즐청소 요구
M08818	BIT	R-- 노즐청소 요구
D08800.7	BIT	SR01 노즐청소 카운터 리셋PB
D08800.8	BIT	SR02 노즐청소 카운터 리셋PB
R01500	WORD	R15 원점체크 최종점검 일자 년
R01600	WORD	R16 원점체크 최종점검 일자 년
R01700	WORD	SR01 원점체크 최종점검 일자 년
R01800	WORD	SR02 원점체크 최종점검 일자 년
M03880	BIT	R15 주간 초품 원점 체크 지령
M03881	BIT	R15 주간 중품 원점 체크 지령
M03882	BIT	R15 야간 초품 원점 체크 지령
M03883	BIT	R15 야간 중품 원점 체크 지령
M03888	BIT	R15 전체 카운터 클리어 Pb
M03889	BIT	R15 OK 카운터 클리어 Pb
M0388A	BIT	R15 NG 카운터 클리어 Pb
M03890	BIT	R16 주간 초품 원점 체크 지령
M03891	BIT	R16 주간 중품 원점 체크 지령
M03892	BIT	R16 야간 초품 원점 체크 지령
M03893	BIT	R16 야간 중품 원점 체크 지령
M03898	BIT	R16 전체 카운터 클리어 Pb
M03899	BIT	R16 OK 카운터 클리어 Pb
M0389A	BIT	R16 NG 카운터 클리어 Pb
M03680	BIT	SR01 주간 초품 원점 체크 지령
M03681	BIT	SR01 주간 중품 원점 체크 지령
M03682	BIT	SR01 야간 초품 원점 체크 지령
M03683	BIT	SR01 야간 중품 원점 체크 지령
M03688	BIT	SR01전체 카운터 클리어 Pb
M03689	BIT	SR01 OK 카운터 클리어 Pb
M0368A	BIT	SR01 NG 카운터 클리어 Pb
M03690	BIT	SR02 주간 초품 원점 체크 지령
M03691	BIT	SR02 주간 중품 원점 체크 지령
M03692	BIT	SR02 야간 초품 원점 체크 지령
M03693	BIT	SR02 야간 중품 원점 체크 지령
M03698	BIT	SR02전체 카운터 클리어 Pb
M03699	BIT	SR02 OK 카운터 클리어 Pb
M0369A	BIT	SR02 NG 카운터 클리어 Pb
D15018.7	BIT	R13 원점체크 By_Pass On
D15018.8	BIT	R14 원점체크 By_Pass On
D15018.9	BIT	R15 원점체크 By_Pass On
D15018.A	BIT	R16 원점체크 By_Pass On
D18146.1	BIT	W40 R08 용접구간 카운터
D18156.1	BIT	W40 R12 용접구간 카운터
D07003.0	BIT	OP2 전체 용접팁교환 요구 PB
D07007.0	BIT	OP2 전체 용접팁교환 완료 PB
D07007.1	BIT	R-- 용접팁교환 완료 PB
D07007.2	BIT	R-- 용접팁교환 완료 PB
D07007.3	BIT	R-- 용접팁교환 완료 PB
D07007.4	BIT	R07 용접팁교환 완료 PB
D07007.5	BIT	R08 용접팁교환 완료 PB
D07007.6	BIT	R12 용접팁교환 완료 PB
D07007.7	BIT	R13 용접팁교환 완료 PB
D07007.8	BIT	R14 용접팁교환 완료 PB
D07007.9	BIT	R15 용접팁교환 완료 PB
D07007.A	BIT	R16 용접팁교환 완료 PB
D12010	WORD	R01 용접 가스 유량
D12014	WORD	R01 가스 하한
D12016	WORD	R01 용접중 가스 유량
D12018	WORD	R01 가스 상한
D12020	WORD	R02 용접 가스 유량
D12024	WORD	R02 가스 하한
D12026	WORD	R02 용접중 가스 유량
D12028	WORD	R02 가스 상한
D12030	WORD	R03 용접 가스 유량
D12034	WORD	R03 가스 하한
D12036	WORD	R03 용접중 가스 유량
D12038	WORD	R03 가스 상한
D12040	WORD	R04 용접 가스 유량
D12044	WORD	R04 가스 하한
D12046	WORD	R04 용접중 가스 유량
D12048	WORD	R04 가스 상한
D12050	WORD	R05 용접 가스 유량
D12054	WORD	R05 가스 하한
D12056	WORD	R05 용접중 가스 유량
D12058	WORD	R05 가스 상한
D12000	WORD	라인1 공기 압력 
D12002	WORD	라인1 공기 압력 
D12004	WORD	라인1 용접 가스 유량
D12006	WORD	라인1 용접 가스 유량
D12110	WORD	R-- 용접 가스 유량
D12114	WORD	R-- 가스 하한
D12116	WORD	R-- 용접중 가스 유량
D12118	WORD	R-- 가스 상한
D15015.3	BIT	R-- GAS Check By_Pass On
D15015.4	BIT	R07 GAS Check By_Pass On
D15015.5	BIT	R08 GAS Check By_Pass On
D15015.6	BIT	R12 GAS Check By_Pass On
D15015.7	BIT	R13 GAS Check By_Pass On
D15015.8	BIT	R14 GAS Check By_Pass On
D15015.9	BIT	R15 GAS Check By_Pass On
D15015.A	BIT	R16 GAS Check By_Pass On
D15014.7	BIT	R13 Weld Count By_Pass On
D15014.8	BIT	R14 Weld Count By_Pass On
R01914.2	BIT	R15 용접시간 NG
R01914.3	BIT	R15 용접구간 NG
R01914.4	BIT	R15 용접 시간/구간 NG
R01915.2	BIT	R16 용접시간 NG
R01915.3	BIT	R16 용접구간 NG
R01915.4	BIT	R16 용접 시간/구간 NG
K04261	BIT	Main 62410-T1500
K04262	BIT	Main 62410-SP2
K04263	BIT	Main 62410-SP3
K04264	BIT	Main 62410-SP4
K04265	BIT	Main 62410-SP5
K04266	BIT	Main 62410-SP6
K04267	BIT	Main 62410-SP7
K04268	BIT	Main 62410-SP8
K04269	BIT	Main 62410-SP9
K0426A	BIT	Main 62410-SP10
K0426B	BIT	Main 62410-SP11
K0426C	BIT	Main 62410-SP12
K0426D	BIT	Main 62410-SP13
K0426E	BIT	Main 62410-SP14
K0426F	BIT	Main 62410-SP15
K04270	BIT	Main 62410-SP16
K04271	BIT	Main 62410-SP17
K04272	BIT	Main 62410-SP18
K04273	BIT	Main 62410-SP19
K04274	BIT	Main 62410-SP20
D19082	WORD	R18 HD2 G1 Spare3 라인내 잔여수량 카운터
D19083	WORD	R18 HD2 G2 Spare3 라인내 잔여수량 카운터
D19084	WORD	R19 HD3 G1 Spare3 라인내 잔여수량 카운터
D19085	WORD	R19 HD3 G2 Spare3 라인내 잔여수량 카운터
D19086	WORD	R20 HD4 G1 Spare3 라인내 잔여수량 카운터
D19087	WORD	R20 HD4 G2 Spare3 라인내 잔여수량 카운터
D19112	WORD	R18 HD2 G1 Spare4 라인내 잔여수량 카운터
D19113	WORD	R18 HD2 G2 Spare4 라인내 잔여수량 카운터
D19114	WORD	R19 HD3 G1 Spare4 라인내 잔여수량 카운터
D19115	WORD	R19 HD3 G2 Spare4 라인내 잔여수량 카운터
D19116	WORD	R20 HD4 G1 Spare4 라인내 잔여수량 카운터
D19117	WORD	R20 HD4 G2 Spare4 라인내 잔여수량 카운터
D19142	WORD	R18 HD2 G1 Spare5 라인내 잔여수량 카운터
D19143	WORD	R18 HD2 G2 Spare5 라인내 잔여수량 카운터
D19144	WORD	R19 HD3 G1 Spare5 라인내 잔여수량 카운터
D19145	WORD	R19 HD3 G2 Spare5 라인내 잔여수량 카운터
D19146	WORD	R20 HD4 G1 Spare5 라인내 잔여수량 카운터
D19147	WORD	R20 HD4 G2 Spare5 라인내 잔여수량 카운터
D19172	WORD	R18 HD2 G1 Spare6 라인내 잔여수량 카운터
D19173	WORD	R18 HD2 G2 Spare6 라인내 잔여수량 카운터
D19174	WORD	R19 HD3 G1 Spare6 라인내 잔여수량 카운터
D19175	WORD	R19 HD3 G2 Spare6 라인내 잔여수량 카운터
D19176	WORD	R20 HD4 G1 Spare6 라인내 잔여수량 카운터
D19177	WORD	R20 HD4 G2 Spare6 라인내 잔여수량 카운터
D19202	WORD	R18 HD2 G1 Spare7 라인내 잔여수량 카운터
D19203	WORD	R18 HD2 G2 Spare7 라인내 잔여수량 카운터
D19204	WORD	R19 HD3 G1 Spare7 라인내 잔여수량 카운터
D19205	WORD	R19 HD3 G2 Spare7 라인내 잔여수량 카운터
D19206	WORD	R20 HD4 G1 Spare7 라인내 잔여수량 카운터
D19207	WORD	R20 HD4 G2 Spare7 라인내 잔여수량 카운터
D19232	WORD	R18 HD2 G1 Spare8 라인내 잔여수량 카운터
D19233	WORD	R18 HD2 G2 Spare8 라인내 잔여수량 카운터
D19234	WORD	R19 HD3 G1 Spare8 라인내 잔여수량 카운터
D19235	WORD	R19 HD3 G2 Spare8 라인내 잔여수량 카운터
D19236	WORD	R20 HD4 G1 Spare8 라인내 잔여수량 카운터
D19237	WORD	R20 HD4 G2 Spare8 라인내 잔여수량 카운터
M00037	BIT	라인1 안전문4 안전매트 검출
M00038	BIT	라인1 안전문4 안전매트 검출유지
D00088	WORD	라인1 안전문4 안전매트 터치 횟수
D00089	WORD	라인1 안전매트4 터치횟수
D15016.C	BIT	라인 안전문4 안전매트 By_Pass On
D18186.1	BIT	W50-2 R15 용접구간 카운터
D18196.1	BIT	W50-2 R16 용접구간 카운터
D18206.1	BIT	S01 SR01 용접구간 카운터
D18216.1	BIT	S01 SR02 용접구간 카운터
R10699	WORD	W200 R05 용접시간 저장 시작워드
R10799	WORD	W200 R06 용접시간 저장 시작워드
R10899	WORD	W300 R05 용접시간 저장 시작워드
R10999	WORD	W300 R06 용접시간 저장 시작워드
R11199	WORD	W600 R-- 용접시간 저장 시작워드
R11299	WORD	W700 R-- 용접시간 저장 시작워드
R11399	WORD	W700 R07 용접시간 저장 시작워드
R11400	WORD	W40 R08 용접시간 저장 시작워드
R11401	WORD	Arc_R08 용접구간 저장 시작워드
R11499	WORD	W40 R08 용접시간 저장 시작워드
R11500	WORD	W40 R12 용접시간 저장 시작워드
R11501	WORD	Arc_R12 용접구간 저장 시작워드
R11599	WORD	W40 R12 용접시간 저장 시작워드
R11600	WORD	W50-1 R13 용접시간 저장 시작워드
R11601	WORD	Arc_R13 용접구간 저장 시작워드
R11699	WORD	W50-1 R13 용접시간 저장 시작워드
R11700	WORD	W50-1 R14 용접시간 저장 시작워드
R11701	WORD	Arc_R14 용접구간 저장 시작워드
R11799	WORD	W50-1 R14 용접시간 저장 시작워드
R11800	WORD	W50-2 R15 용접시간 저장 시작워드
R11801	WORD	Arc_R15 용접구간 저장 시작워드
R11899	WORD	W50-2 R15 용접시간 저장 시작워드
R11900	WORD	W50-2 R16 용접시간 저장 시작워드
R11901	WORD	Arc_R16 용접구간 저장 시작워드
R11999	WORD	W50-2 R16 용접시간 저장 시작워드
D08420	WORD	R05 표준시간 최소 용접시간 설정
D08440	WORD	R06 표준시간 최소 용접시간 설정
D08460	WORD	R05 표준시간 최소 용접시간 설정
D08480	WORD	R06 표준시간 최소 용접시간 설정
D08520	WORD	R-- 표준시간 최소 용접시간 설정
D08560	WORD	R-- 표준시간 최소 용접시간 설정
D08600	WORD	R12 표준시간 최소 용접시간 설정
D08640	WORD	R14 표준시간 최소 용접시간 설정
D08680	WORD	R16 표준시간 최소 용접시간 설정
D15014.A	BIT	R16 Weld Count By_Pass On
D15012.7	BIT	SR01 Weld Count By_Pass On
D15013.7	BIT	SR01 GAS Check By_Pass On
D15013.8	BIT	SR02 GAS Check By_Pass On
D17539.2	BIT	W200/W50-1 지그사용 마킹기 데이터
D17539.3	BIT	W300/W50-1 지그사용 마킹기 데이터
D17539.4	BIT	W100/W50-2 지그사용 마킹기 데이터
D17539.5	BIT	W150/W50-2 지그사용 마킹기 데이터
D17539.6	BIT	W200/W50-2 지그사용 마킹기 데이터
D17539.7	BIT	W300/W50-2 지그사용 마킹기 데이터
M16353	BIT	OP3 R03 Seleted
M16354	BIT	OP3 R04 Seleted
M16355	BIT	OP3 R05 Seleted
M16356	BIT	OP3 R06 Seleted
M16357	BIT	OP3 R-- Seleted
M16358	BIT	OP3 R-- Seleted
M16359	BIT	OP3 R-- Seleted
M1635A	BIT	OP3 R07 Seleted
M1635B	BIT	OP3 R08 Seleted
M1635C	BIT	OP3 R12 Seleted
M1635D	BIT	OP3 R13 Seleted
M1635E	BIT	OP3 R14 Seleted
M1635F	BIT	OP3 R15 Seleted
M16370	BIT	OP1 R16 Power ON Pb
M16371	BIT	OP1 R17 Power ON Pb
M16372	BIT	OP1 R18 Power ON Pb
M16373	BIT	OP1 R19 Power ON Pb
M16374	BIT	OP1 R20 Power ON Pb
M16375	BIT	OP1 R17 HD1 Power ON Pb
M16376	BIT	OP1 R18 HD2 Power ON Pb
M16377	BIT	OP1 R19 HD3 Power ON Pb
M16378	BIT	OP1 R20 HD4 Power ON Pb
M16379	BIT	OP1 R25 Power ON Pb
M1637E	BIT	OP1 R30 Power ON Pb
P0252C	BIT	W80-1 제품확인(PL)
P0262C	BIT	W80-2 제품확인(PL)
P0260A	BIT	W80-2 작업자 NG 취출기동 SW
P0262A	BIT	W80-2 제품 NG Lamp [부져차단]
P02629	BIT	W80-2 제품 NG Lamp [녹색]
P02628	BIT	W80-2 제품 NG Lamp [적색]
P02727	BIT	마스터 DIE 제품 안착확인 LS
D00508	WORD	W300 Air Blow Setting Time
D00408	WORD	W200 Air Blow Set'g Time
D15006.C	BIT	라인 전체 배기팬 전원 ON Pb
D15007.C	BIT	라인 전체 배기팬 전원 ON LAMP
D24998	WORD	W600 NG 버퍼
P0250A	BIT	W80-1 작업자 NG 취출기동 SW
P02528	BIT	W80-1 제품 NG Lamp [적색]
P02529	BIT	W80-1 제품 NG Lamp [녹색]
P0252A	BIT	W80-1 제품 NG Lamp [부져차단]
D15021.8	BIT	OP3 STN8 Select Pb
P02415	BIT	W70 제품확인6 PIPE ON:이상 OFF;정상
K00250	BIT	W100.2 선두 신호
K00251	BIT	W200.4 선두 신호
P1052B	BIT	R05 (OT28)
P1062B	BIT	R06 (OT28)
M0012E	BIT	W10 LH 작업수량 도달 차종교환 메세지
M05103	BIT	R03 지그 작업중
M05104	BIT	R04 지그 작업중
M05105	BIT	R05 지그 작업중
M05107	BIT	R-- 지그 작업중
M05108	BIT	R-- 지그 작업중
M05109	BIT	R-- 지그 작업중
M05110	BIT	R07 HD1 지그 작업중
M05111	BIT	R08 HD2 지그 작업중
M05201	BIT	R01 로보트 팬던트 감지 이상
M05202	BIT	R02 로보트 팬던트 감지 이상
M05203	BIT	R03 로보트 팬던트 감지 이상
M05204	BIT	R04 로보트 팬던트 감지 이상
M05205	BIT	R05 로보트 팬던트 감지 이상
M05206	BIT	R06 로보트 팬던트 감지 이상
M05207	BIT	R-- 로보트 팬던트 감지 이상
M05208	BIT	R-- 로보트 팬던트 감지 이상
M05209	BIT	R-- 로보트 팬던트 감지 이상
M05210	BIT	R07 HD1 로보트 팬던트 감지 이상
M05211	BIT	R08 HD2 로보트 팬던트 감지 이상
T5210	BIT/WORD	R07 로보트 팬던트 감지 이상
T5211	BIT/WORD	R08 로보트 팬던트 감지 이상
T5212	BIT/WORD	R12 로보트 팬던트 감지 이상
T5213	BIT/WORD	R13 로보트 팬던트 감지 이상
T5214	BIT/WORD	R14 로보트 팬던트 감지 이상
T5215	BIT/WORD	R15 로보트 팬던트 감지 이상
T5216	BIT/WORD	R16 로보트 팬던트 감지 이상
T5217	BIT/WORD	R17(H/D-1) 로보트 팬던트 감지 이상
T5218	BIT/WORD	R18(H/D-2) 로보트 팬던트 감지 이상
T5219	BIT/WORD	R19(H/D-3) 로보트 팬던트 감지 이상
T5201	BIT/WORD	R01 로보트 팬던트 감지 이상
T5202	BIT/WORD	R02 로보트 팬던트 감지 이상
T5203	BIT/WORD	R03 로보트 팬던트 감지 이상
T5204	BIT/WORD	R04 로보트 팬던트 감지 이상
T5205	BIT/WORD	R05 로보트 팬던트 감지 이상
T5206	BIT/WORD	R06 로보트 팬던트 감지 이상
T5207	BIT/WORD	R-- 로보트 팬던트 감지 이상
T5208	BIT/WORD	R-- 로보트 팬던트 감지 이상
T5209	BIT/WORD	R-- 로보트 팬던트 감지 이상
T5220	BIT/WORD	R20(H/D-4) 로보트 팬던트 감지 이상
T0124	BIT/WORD	W10 LH 차종감지 이상 지연
T0681	BIT/WORD	W400 클램프 이상
T0685	BIT/WORD	W400 베이스 슬라이드 이상
M03978	BIT	W600 체크 OK LAMP _ W600
P0005B	BIT	라인1 조명등 전원 ON
P0005C	BIT	라인2 조명등 전원 ON
P0005D	BIT	라인1 배기팬 전원 ON
M16577	BIT	OP1 R-- Power On Lamp
M16578	BIT	OP1 R-- Power On Lamp
M16467	BIT	OP1 R-- Power OFF Pb
M16468	BIT	OP1 R-- Power OFF Pb
M16367	BIT	OP1 R-- Power ON Pb
M16368	BIT	OP1 R-- Power ON Pb
M16978	BIT	OP1 R-- 용접기 Power On Lamp
M16867	BIT	OP1 R-- 용접기 Power OFF Pb
M16868	BIT	OP1 R-- 용접기 Power OFF Pb
M16768	BIT	OP1 R-- 용접기 Power On Pb
M16767	BIT	OP1 R-- 용접기 Power On Pb
M0390A	BIT	R-- Gas On 검출이상
M0390B	BIT	R-- 누설가스 검출이상
M0390C	BIT	R-- Gas On 검출이상
M0390E	BIT	R-- Gas On 검출이상
M0390D	BIT	R-- 누설가스 검출이상
M0390F	BIT	R-- 누설가스 검출이상
M04717	BIT	R-- 팁 교환요구
M04718	BIT	R-- 팁 교환요구
K07220	BIT	W200 서보2 로봇 간섭이상
K07230	BIT	W300 서보3 로봇 간섭이상
D00401	WORD	W200 상부 안전센서 상태
D00402	WORD	W200 하부 안전센서 상태
D00501	WORD	W300 상부 안전센서 상태
D00502	WORD	W300 하부 안전센서 상태
M0020F	BIT	W10 RH 지그동작 서보위치
P10311	BIT	R03 (OT02)
K0011A	BIT	W50 너트감지 OK
K0011B	BIT	W50 너트감지 NG
D00170	WORD	W50 너트감지 Data.1 1:OK 2:NG
D00123	WORD	W50 파트램프 상태13
D00124	WORD	W50 파트램프 상태14
D00125	WORD	W50 파트램프 상태15
M10248	BIT	R02 (IN57)
P10348	BIT	R03 (OT57)
P10248	BIT	R02 (OT57)
M10348	BIT	R03 (IN57)
P1032A	BIT	R03 (OT27)
M10448	BIT	R04 (IN57)
P10548	BIT	R05 (OT57)
P10411	BIT	R04 (OT02)
P1042B	BIT	R04 (OT28)
M10548	BIT	R05 (IN57)
P10448	BIT	R04 (OT57)
P1052C	BIT	R05 (OT29)
P1062D	BIT	R06 (OT30)
M16288	BIT	OP1 R08 HD2 Seleted
T0620	BIT/WORD	W400 파트없음 지연
T0621	BIT/WORD	W400 파트 OK지연
M00341	BIT	W20-2 LH 로보트 간섭무
T0313	BIT/WORD	W20-2 LH 로보트 간섭무지연
T0666	BIT/WORD	W400 베이스 록킹 후진완료
T0646	BIT/WORD	W400 베이스 록킹 전진완료
K00221	BIT	W100 R03 1차 용접완료
K00222	BIT	W100 R03 2차 용접완료
T0665	BIT/WORD	W400 베이스 슬라이드 후진완료
T0645	BIT/WORD	W400 베이스 슬라이드 전진완료
T0641	BIT/WORD	W400 클램프 잠김완료
T0518	BIT/WORD	W30 서보 위치이상 지연
T0519	BIT/WORD	W30 서보 근접센서 위치이상 Tmr
T0686	BIT/WORD	W400 베이스 록킹 이상
D15016.7	BIT	W500 파트체크 By_Pass On
D00760	WORD	W500 동도 측정 1:OK 2:NG
D00771	WORD	W500 G1 측정 1:OK 2:NG
D00767	WORD	W500 RH 홀 체크 결과
D00768	WORD	W500 LH 홀 체크 결과
D00772	WORD	W500 G2 측정 1:OK 2:NG
D00773	WORD	W500 G3 측정 1:OK 2:NG
D00774	WORD	W500 G4 측정 1:OK 2:NG
D00775	WORD	W500 G5 측정 1:OK 2:NG
D00776	WORD	W500 G6 측정 1:OK 2:NG
D00777	WORD	W500 G7 측정 1:OK 2:NG
D24012	WORD	W500 Unload'g G1:P1-P2 REAL Data
D24014	WORD	W600 Load'g G1:P1-P2 REAL Data
D24022	WORD	W500 Unload'g G2:P3-P4 REAL Data
D24024	WORD	W600 Load'g G2:P3-P4 REAL Data
D24032	WORD	W500 Unload'g G3:(Avg) REAL Data
D24034	WORD	W600 Load'g G3:(Avg) REAL Data
D24042	WORD	W500 Unload'g G4:P5-P6 REAL Data
D24044	WORD	W600 Load'g G4:P5-P6 REAL Data
D24052	WORD	W500 Unload'g G5:P7-P8 REAL Data
D24054	WORD	W600 Load'g G5:P7-P8 REAL Data
D24062	WORD	W500 Unload'g G6:(Avg) REAL Data
D24064	WORD	W600 Load'g G6:(Avg) REAL Data
D24072	WORD	W500 Unload'g G7:G3+G6 REAL Data
D24074	WORD	W600 Load'g G7:G3+G6 REAL Data
D03912	WORD	OK_NG Master 파트램프 상태2
M03979	BIT	W600 체크 NG LAMP - W500
P1041C	BIT	R04 (OT13)
D08823	WORD	R-- Arc Weld Count
D08825	WORD	R-- Arc Weld Count
D08831	WORD	R-- Arc Weld Count
D08826	WORD	R-- 노즐청소 설정
D08827	WORD	R-- Arc Weld Count
D08828	WORD	R-- 노즐청소 설정
D08829	WORD	R-- Arc Weld Count
M04719	BIT	R-- 팁 교환요구
D04700.7	BIT	R-- 로보트 용접 카운트 리셋PB
D04700.8	BIT	R-- 로보트 용접 카운트 리셋PB
D04701.1	BIT	R-- 로보트 용접 카운트 리셋PB
T2007	BIT/WORD	R-- 노즐청소 요구지연
T2008	BIT/WORD	R-- 노즐청소 요구지연
T2010	BIT/WORD	R-- 노즐청소 요구지연
M08809	BIT	R-- 노즐청소 진입중
M08819	BIT	R-- 노즐청소 요구
M09968	BIT	R-- 원점 확인 OK
M09978	BIT	R-- 원점 확인 NG
D18214	WORD	W100 R02 용접구간 카운터
D18014	WORD	W100 R02 용접구간 카운터설정
D18234	WORD	W200 R04 용접구간 카운터
D18034	WORD	W200 R04 용접구간 카운터설정
D18244	WORD	W200 R05 용접구간 카운터
D18042	WORD	R05 표준시간 최소 용접시간
D18043	WORD	R05 표준시간 최대 용접시간
D18044	WORD	W200 R05 용접구간 카운터설정
R10401	WORD	Arc_R05 용접구간 저장 시작워드
T0054	BIT/WORD	라인1 안전문1 안전매트 횟수RST 지연(W300)
T0053	BIT/WORD	라인1 안전문1 안전매트 횟수RST 지연(W50)
M0004B	BIT	OP2 R08 HD2 Emergency Stop
T2216	BIT/WORD	R-- Gas On 검출이상
T2217	BIT/WORD	R-- 누설가스 검출이상
T0661	BIT/WORD	W400 클램프 풀림완료
D12060	WORD	R-- 용접 가스 유량
D12070	WORD	R-- 용접 가스 유량
D12076	WORD	R-- 용접중 가스 유량
D12080	WORD	R-- 용접 가스 유량
D12086	WORD	R-- 용접중 가스 유량
D15015.1	BIT	R-- GAS Check By_Pass On
T2212	BIT/WORD	R-- Gas On 검출이상
D12074	WORD	R-- 가스 하한
D12078	WORD	R-- 가스 상한
T2213	BIT/WORD	R-- 누설가스 검출이상
T2214	BIT/WORD	R-- Gas On 검출이상
D15015.2	BIT	R-- GAS Check By_Pass On
D12084	WORD	R-- 가스 하한
D12088	WORD	R-- 가스 상한
T2215	BIT/WORD	R-- 누설가스 검출이상
D00778	WORD	W500 G8 측정 1:OK 2:NG
D00779	WORD	W500 G9 측정 1:OK 2:NG
D00780	WORD	W500 G10 측정 1:OK 2:NG
D00781	WORD	W500 G11 측정 1:OK 2:NG
D00782	WORD	W500 G12 측정 1:OK 2:NG
D00783	WORD	W500 G13 측정 1:OK 2:NG
M16287	BIT	OP1 R07 HD1 Seleted
D00570	WORD	W300 3D 비젼 측정 1:OK 2:NG
D00571	WORD	W300 3D비젼 P1 측정 1:OK 2:NG
D00572	WORD	W300 3D비젼 P2 측정 1:OK 2:NG
D00573	WORD	W300 3D비젼 P3 측정 1:OK 2:NG
D00574	WORD	W300 3D비젼 P4 측정 1:OK 2:NG
D00575	WORD	W300 3D비젼 P5 측정 1:OK 2:NG
D00576	WORD	W300 3D비젼 P6 측정 1:OK 2:NG
D00577	WORD	W300 3D비젼 P7 측정 1:OK 2:NG
D00578	WORD	W300 3D비젼 P8 측정 1:OK 2:NG
D00579	WORD	W300 3D비젼 P9 측정 1:OK 2:NG
D00580	WORD	W300 3D비젼 P10 측정 1:OK 2:NG
D00581	WORD	W300 3D비젼 P11 측정 1:OK 2:NG
D00582	WORD	W300 3D비젼 P12 측정 1:OK 2:NG
D00583	WORD	W300 3D비젼 P13 측정 1:OK 2:NG
D00584	WORD	W300 3D비젼 P14 측정 1:OK 2:NG
D00585	WORD	W300 3D비젼 P15 측정 1:OK 2:NG
D15002.2	BIT	W300 3D비젼체크 바이패스 ON
M03977	BIT	W600 3D비젼 체크 NG LAMP_W300
M03976	BIT	W600 3D비젼 체크 OK LAMP_W300
D24999	WORD	W600 3D비젼 NG 버퍼
D00586	WORD	W300 3D비젼 P16 측정 1:OK 2:NG
D00571.0	BIT	W300 3D비젼 P1 측정 OK
D00572.0	BIT	W300 3D비젼 P2 측정 OK
D00573.0	BIT	W300 3D비젼 P3 측정 OK
D00574.0	BIT	W300 3D비젼 P4 측정 OK
D00575.0	BIT	W300 3D비젼 P5 측정 OK
D00576.0	BIT	W300 3D비젼 P6 측정 OK
D00577.0	BIT	W300 3D비젼 P7 측정 OK
D00578.0	BIT	W300 3D비젼 P8 측정 OK
D00579.0	BIT	W300 3D비젼 P9 측정 OK
D00580.0	BIT	W300 3D비젼 P10 측정 OK
D00581.0	BIT	W300 3D비젼 P11 측정 OK
D00582.0	BIT	W300 3D비젼 P12 측정 OK
D00583.0	BIT	W300 3D비젼 P13 측정 OK
D00584.0	BIT	W300 3D비젼 P14 측정 OK
D00585.0	BIT	W300 3D비젼 P15 측정 OK
D00586.0	BIT	W300 3D비젼 P16 측정 OK
D00571.1	BIT	W300 3D비젼 P1 측정 NG
D00572.1	BIT	W300 3D비젼 P2 측정 NG
D00573.1	BIT	W300 3D비젼 P3 측정 NG
D00574.1	BIT	W300 3D비젼 P4 측정 NG
D00575.1	BIT	W300 3D비젼 P5 측정 NG
D00576.1	BIT	W300 3D비젼 P6 측정 NG
D00577.1	BIT	W300 3D비젼 P7 측정 NG
D00578.1	BIT	W300 3D비젼 P8 측정 NG
D00579.1	BIT	W300 3D비젼 P9 측정 NG
D00580.1	BIT	W300 3D비젼 P10 측정 NG
D00581.1	BIT	W300 3D비젼 P11 측정 NG
D00582.1	BIT	W300 3D비젼 P12 측정 NG
D00583.1	BIT	W300 3D비젼 P13 측정 NG
D00584.1	BIT	W300 3D비젼 P14 측정 NG
D00585.1	BIT	W300 3D비젼 P15 측정 NG
D00586.1	BIT	W300 3D비젼 P16 측정 NG
T4026	BIT/WORD	W600 작업자 NG 취출기동 
D01874	WORD	W500 G4 측정 1:OK 2:NG (W600)
D01875	WORD	W500 G5 측정 1:OK 2:NG (W600)
D01876	WORD	W500 G6 측정 1:OK 2:NG (W600)
D01877	WORD	W500 G7 측정 1:OK 2:NG (W600)
D01878	WORD	W500 G8 측정 1:OK 2:NG (W600)
D01879	WORD	W500 G9 측정 1:OK 2:NG (W600)
D01880	WORD	W500 G10 측정 1:OK 2:NG (W600)
D01881	WORD	W500 G11 측정 1:OK 2:NG (W600)
D01882	WORD	W500 G12 측정 1:OK 2:NG (W600)
D01883	WORD	W500 G13 측정 1:OK 2:NG (W600)
M16268	BIT	OP1 R08 HD2 Select Pb
M16267	BIT	OP1 R07 HD1 Select Pb
P0031A	BIT	W10 LH 3차 클램프 잠김3
M10560	BIT	R05 (ln81) Wire 커터진진
M10561	BIT	R05 (ln82) Wire 커터후진
M10562	BIT	R05 (ln83) Wire Home
M10563	BIT	R05 (ln84) 노즐확인
M10565	BIT	R05 (ln86) Wire Cut
M10566	BIT	R05 (ln87) Motor On
M17000	BIT	R07 HD1 In Line Part Empty
M17001	BIT	R08 HD2 In Line Part Empty
D21012	WORD	G3:FRT LH "L" ASCII Data
D21017	WORD	G4:FRT LH "H" ASCII Data
D21021	WORD	G5:FRT RH "T" ASCII Data
D21026	WORD	G6:FRT RH "L" ASCII Data
D21030	WORD	G7:FRT RH "H" ASCII Data
D21035	WORD	G8:RR LH "T" ASCII Data
D21039	WORD	G9:RR LH "L" ASCII Data
D21044	WORD	G10:RR LH "H" ASCII Data
D21057	WORD	G13:RR RH "H" ASCII Data
T0074	BIT/WORD	서보모타4 전원 OFF 지연
D14100.0	BIT	PC Ready
D14102.0	BIT	PLC Ready
D14102.1	BIT	Car Type-1
D14102.2	BIT	Car Type-2
D14102.3	BIT	Car Type-4
D14102.4	BIT	Car Type-8
D14100.8	BIT	W500 Check OK
D14100.9	BIT	W500 Check NG
D14102.8	BIT	W500 Check Req
D14102.F	BIT	Master Check Mode
D14103.0	BIT	W500 Check Bypass
D14103.8	BIT	W300 Loading
D15100.A	BIT	PC Data Keeping Bypass ON
D14103.A	BIT	W600 Loading
D14200	WORD	PC W500 동도 측정 Data
D24410	WORD	W600 G1:CTR "L" REAL Data
D24420	WORD	W600 G2:FRT LH "T" REAL Data
D24430	WORD	W600 G3:FRT LH "L" REAL Data
D24440	WORD	W600 G4:FRT LH "H" REAL Data
D24450	WORD	W600 G5:FRT RH "T" REAL Data
D24460	WORD	W600 G6:FRT RH "L" REAL Data
D24470	WORD	W600 G7:FRT RH "H" REAL Data
D24480	WORD	W600 G8:RR LH "T" REAL Data
D24490	WORD	W600 G9:RR LH "L" REAL Data
D24510	WORD	W600 G11:RR RH "T" REAL Data
D24520	WORD	W600 G12:RR RH "L" REAL Data
D24530	WORD	W600 G13:RR RH "H" REAL Data
D26250	WORD	W600 G1:CTR "L" REAL Data 차이 <RG3>
D26255	WORD	W600 G2:FRT LH "T" REAL Data 차이 <RG3>
D26260	WORD	W600 G3:FRT LH "L" REAL Data 차이 <RG3>
D26265	WORD	W600 G4:FRT LH "H" REAL Data 차이 <RG3>
D26270	WORD	W600 G5:FRT RH "T" REAL Data 차이 <RG3>
D26275	WORD	W600 G6:FRT RH "L" REAL Data 차이 <RG3>
D26280	WORD	W600 G7:FRT RH "H" REAL Data 차이 <RG3>
D26285	WORD	W600 G8:RR LH "T" REAL Data 차이 <RG3>
D26290	WORD	W600 G9:RR LH "L" REAL Data 차이 <RG3>
D26295	WORD	W600 G10:RR LH "H" REAL Data 차이 <RG3>
D26300	WORD	W600 G11:RR RH "T" REAL Data 차이 <RG3>
D26305	WORD	W600 G12:RR RH "L" REAL Data 차이 <RG3>
D26310	WORD	W600 G13:RR RH "H" REAL Data 차이 <RG3>
D26152	WORD	OK/NG마스타 G1:CTR "L" REAL Data 차이 <RG3>
D26157	WORD	OK/NG마스타 G2:FRT LH "T" REAL Data 차이 <RG3>
D26162	WORD	OK/NG마스타 G3:FRT LH "L" REAL Data 차이 <RG3>
D26167	WORD	OK/NG마스타 G4:FRT LH "H" REAL Data 차이 <RG3>
D26172	WORD	OK/NG마스타 G5:FRT RH "T" REAL Data 차이 <RG3>
D26177	WORD	OK/NG마스타 G6:FRT RH "L" REAL Data 차이 <RG3>
D26182	WORD	OK/NG마스타 G7:FRT RH "H" REAL Data 차이 <RG3>
D26187	WORD	OK/NG마스타 G8:RR LH "T" REAL Data 차이 <RG3>
D26192	WORD	OK/NG마스타 G9:RR LH "L" REAL Data 차이 <RG3>
D26197	WORD	OK/NG마스타 G10:RR LH "H" REAL Data 차이 <RG3>
D26202	WORD	OK/NG마스타 G11:RR RH "T" REAL Data 차이 <RG3>
D26207	WORD	OK/NG마스타 G12:RR RH "L" REAL Data 차이 <RG3>
D26212	WORD	OK/NG마스타 G13:RR RH "H" REAL Data 차이 <RG3>
D14110	WORD	VIN AUX
D14111	WORD	VIN AUX W300
D14112	WORD	VIN AUX H/D.1
D14113	WORD	VIN AUX W400
D14114	WORD	VIN AUX H/D.2
D14115	WORD	VIN AUX W500
D14116	WORD	VIN AUX H/D.2
D14117	WORD	VIN AUX W600
D31000	WORD	PLC->PC 3D비젼 체크 Data
D31050	WORD	PLC->PC W600 스케너 Data_LH
D31100	WORD	PLC->PC W600 스케너 Data_RH
D31200	WORD	PLC->PC W600 동도 측정 Data
D14118	WORD	VIN AUX W700
D14103.1	BIT	W600 NG
D14103.9	BIT	W500 Loading
D14103.C	BIT	W700 Loading
D14103.B	BIT	W600 Unloading
D14102.E	BIT	W300 Scan RH Check Req
D14102.D	BIT	W300 Scan LH Check Req
D14100.D	BIT	W300 Scan LH Check'd
D14100.E	BIT	W300 Scan RH Check'd
D14101.C	BIT	W700 Loading Check
D00761	WORD	W500 F/PROOF 파트램프 상태1
D00762	WORD	W500 F/PROOF 파트램프 상태2
D00763	WORD	W500 F/PROOF 파트램프 상태3
D00764	WORD	W500 F/PROOF 파트램프 상태4
D15002.4	BIT	W350 스케너 체크 바이패스
P00316	BIT	W10 LH 3차 클램프 잠김1
P1051B	BIT	R05 (OT12)
P1041B	BIT	R04 (OT12)
R01800.2	BIT	R01 용접시간 NG
R01800.3	BIT	R01 용접구간 NG
R01800.4	BIT	R01 용접 시간/구간 NG
R01801.2	BIT	R02 용접시간 NG
R01801.3	BIT	R02 용접구간 NG
R01801.4	BIT	R02 용접 시간/구간 NG
R01802.2	BIT	R03 용접시간 NG W02-1
R01802.3	BIT	R03 용접구간 NG W02-1
R01802.4	BIT	R03 용접 시간/구간 NG W02-1
R01803.2	BIT	R04 용접시간 NG W02-1
R01803.3	BIT	R04 용접구간 NG W02-1
R01803.4	BIT	R04 용접 시간/구간 NG W02-1
R01804.2	BIT	R05 용접시간 NG
R01804.3	BIT	R05 용접구간 NG
R01804.4	BIT	R05 용접 시간/구간 NG
R01805.2	BIT	R06 용접시간 NG
R01805.3	BIT	R06 용접구간 NG
R01805.4	BIT	R06 용접 시간/구간 NG
D28152	WORD	G1: CTR "L" 3차원 측정값
D28157	WORD	G2:FRT LH "T" 3차원 측정값
D28162	WORD	G3:FRT LH "L" 3차원 측정값
D28167	WORD	G4:FRT LH "H" 3차원 측정값
D28172	WORD	G5:FRT RH "T" 3차원 측정값
D28177	WORD	G6:FRT RH "L" 3차원 측정값
D28182	WORD	G7:FRT RH "H" 3차원 측정값
D28187	WORD	G8:RR LH "T" 3차원 측정값
D28192	WORD	G9:RR LH "L" 3차원 측정값
D28197	WORD	G10:RR LH "H" 3차원 측정값
D28202	WORD	G11:RR RH "T" 3차원 측정값
D28207	WORD	G12:RR RH "L" 3차원 측정값
D28212	WORD	G13:RR RH "H" 3차원 측정값
M00076	BIT	OP2 Robot08 Gripper-2 Error
M00077	BIT	OP2 Robot08 Gripper Part Error
M00033	BIT	OP3 Emergency Stop
M10700	BIT	R07 HD1 External RUN
M10701	BIT	R07 HD1 Servo_ON
M10703	BIT	R07 HD1 Error Reset
M10705	BIT	R07 HD1 REMInE Selet
M10706	BIT	R07 HD1 PLAY Select
M10707	BIT	R07 HD1 TEACH Select
M1070A	BIT	OP1 RobIn WELD ON
M1071C	BIT	R07 HD1 (In13) W150-2 로딩가능 _RG3
M1071D	BIT	R07 HD1 (In14) W150-2 언로딩가능 _RG3
M1071E	BIT	R07 HD1 (In15) W200 로딩가능 _RG3
M1071F	BIT	R07 HD1 (In16) W200 언로딩가능 _RG3
M10720	BIT	R07 HD1 (In17) W300 로딩가능 _RG3
M10721	BIT	R07 HD1 (In18) W300 언로딩가능 _RG3
M10722	BIT	R07 HD1 (In19) W400 로딩가능 _RG3
M10723	BIT	R07 HD1 (In20) W150 파트 FULL
M10724	BIT	R07 HD1 (In21)
M1072E	BIT	R07 HD1 (In31) 외부 비상정지
M1072F	BIT	R07 HD1 (In32) 외부 일시정지
M1071B	BIT	R07 HD1 (In12) W150-1 언로딩가능 _RG3
M1071A	BIT	R07 HD1 (In11) W150-1 로딩 가능 _RG3
M10738	BIT	R07 HD1 (In41) 그리퍼1 파트감지
M10737	BIT	R07 HD1 (In40)
M10736	BIT	R07 HD1 (In39)
M1073C	BIT	R07 HD1 (In45) 그리퍼1 핀 후진
M10740	BIT	R07 HD1 (In49) 그리퍼2 핀 전진
M10718	BIT	R07 HD1 (In09) W100 언로딩 가능 _RG3
M10719	BIT	R07 HD1 (In10)
M10729	BIT	R07 HD1 (In26) R07 HD1<-R2 인터록
M10730	BIT	R07 HD1 (In33) W100 핀 다운 완료
M10731	BIT	R07 HD1 (In34) W150-1 핀 다운 완료
M10732	BIT	R07 HD1 (In35) W150-2 핀 다운 완료
M10733	BIT	R07 HD1 (In36) W200 핀 다운 완료
M10734	BIT	R07 HD1 (In37) W300 핀 다운 완료
M10739	BIT	R07 HD1 (In42) 그리퍼1 클램프 잠김
M1073A	BIT	R07 HD1 (In43) 그리퍼1 클램프 풀림
M1073B	BIT	R07 HD1 (In44) 그리퍼1 핀 전진
M1073E	BIT	R07 HD1 (In47) 그리퍼2 클램프 잠김
M1073F	BIT	R07 HD1 (In48) 그리퍼2 클램프 풀림
M10741	BIT	R07 HD1 (In50) 그리퍼2 핀 후진
M10770	BIT	R07 HD1 그리퍼2 핀 전진 SOL
M10771	BIT	R07 HD1 그리퍼2 핀 후진 SOL
M10772	BIT	R07 HD1 그리퍼2 클램프 잠김 SOL
M10773	BIT	R07 HD1 그리퍼2 클램프 풀림 SOL
M10774	BIT	R07 HD1 그리퍼1 핀 전진 Sol
M10775	BIT	R07 HD1 그리퍼1 핀 후진 Sol
M10776	BIT	R07 HD1 그리퍼1 클램프 잠김 Sol
M10777	BIT	R07 HD1 그리퍼1 클램프 풀림 Sol
M10790	BIT	R07 HD1 그리퍼 파트감지 없음
M1072D	BIT	R07 HD1 (In30) R07 HD1<-R6 인터록
M1072C	BIT	R07 HD1 (In29) R07 HD1<-R5 인터록
M1072B	BIT	R07 HD1 (In28) R07 HD1<-R4 인터록
M1072A	BIT	R07 HD1 (In27) R07 HD1<-R3 인터록
M10744	BIT	R07 HD1 (In53)
M10743	BIT	R07 HD1 (In52)
M10742	BIT	R07 HD1 (In51)
M10727	BIT	R07 HD1 (In24) Line 강제배출 Mode On
M10735	BIT	R07 HD1 (In38) 비젼마스타 W400 언로딩완료
M10725	BIT	R07 HD1 (In22) 스케너 완료
P10700	BIT	R07 HD1 Running
P10701	BIT	R07 HD1 Servo_ON
P10705	BIT	R07 HD1 REMOTE Mode
P10706	BIT	R07 HD1 PLAY Mode
P10707	BIT	R07 HD1 TEACH 모드
P10739	BIT	R07 HD1 (Ot42) 그리퍼1 클램프 잠김요구
P10728	BIT	R07 HD1 (Ot25) R07 HD1->R1 인터록
P10740	BIT	R07 HD1 (Ot49) 그리퍼2 핀 전진요구
P10736	BIT	R07 HD1 (Ot37)
P10737	BIT	R07 HD1 (Ot37)
P1073F	BIT	R07 HD1 (Ot48) 그리퍼2 클램프 풀림요구
P1073B	BIT	R07 HD1 (Ot44) 그리퍼1 핀 전진요구
P1072F	BIT	R07 HD1 (Ot32) 비상정지
P1070A	BIT	R07 HD1 HOME Position
P10715	BIT	R07 HD1 (Ot06) W400 간섭무
P10716	BIT	R07 HD1 (Ot07) W04 간섭무
P1071E	BIT	R07 HD1 (Ot15) W200 로딩 완료 _RG3
P1071F	BIT	R07 HD1 (Ot16) W200 언로딩 완료 _RG3
P10722	BIT	R07 HD1 (Ot19) W400 로딩 완료 _RG3
P10730	BIT	R07 HD1 (Ot33) W100 핀 다운 요구
P10731	BIT	R07 HD1 (Ot34) W150-1 핀 다운 요구
P10732	BIT	R07 HD1 (Ot35) W150-2 핀 다운 요구
P10733	BIT	R07 HD1 (Ot36) W200 핀 다운 요구
P10734	BIT	R07 HD1 (Ot37) W300 핀 다운 요구
P1073A	BIT	R07 HD1 (Ot43) 그리퍼1 클램프 풀림요구
P1073C	BIT	R07 HD1 (Ot45) 그리퍼1 핀 후진요구
P1073E	BIT	R07 HD1 (Ot47) 그리퍼2 클램프 잠김요구
P10741	BIT	R07 HD1 (Ot50) 그리퍼2 핀 후진요구
P1077C	BIT	R07 HD1 그리퍼1 클램프 풀림1
P1077D	BIT	R07 HD1 그리퍼1 클램프 잠김2
P10720	BIT	R07 HD1 (Ot17) W300 로딩 완료 _RG3
P10721	BIT	R07 HD1 (Ot18) W300 언로딩 완료 _RG3
P1071A	BIT	R07 HD1 (Ot11) W150-1 로딩 완료 _RG3
P1071C	BIT	R07 HD1 (Ot13) W150-2 로딩 완료 _RG3
P1071B	BIT	R07 HD1 (Ot12) W150-1 언로딩 완료 _RG3
P1071D	BIT	R07 HD1 (Ot14) W150-2 언로딩 완료 _RG3
P10718	BIT	R07 HD1 (Ot09) W100 언로딩 완료 _RG3
P10770	BIT	R07 HD1 그리퍼 파트감지.1
P10771	BIT	R07 HD1 그리퍼 파트감지.2
P10776	BIT	R07 HD1 그리퍼 클램프 잠김1
P10778	BIT	R07 HD1 그리퍼 클램프 잠김2
P1077A	BIT	R07 HD1 그리퍼 클램프 잠김3
P10777	BIT	R07 HD1 그리퍼 클램프 풀림1
P10779	BIT	R07 HD1 그리퍼 클램프 풀림2
P1077B	BIT	R07 HD1 그리퍼 클램프 풀림3
P10772	BIT	R07 HD1 그리퍼 핀 전진1
P10774	BIT	R07 HD1 그리퍼 핀 전진2
P10773	BIT	R07 HD1 그리퍼 핀 후진1
P10775	BIT	R07 HD1 그리퍼 핀 후진2
P1078E	BIT	HD-1 H/D Robot Air Press S/W
P10729	BIT	R07 HD1 (Ot26) HD1->R2 인터록
P1072A	BIT	R07 HD1 (Ot27) HD1->R3 인터록
P1072B	BIT	R07 HD1 (Ot28) HD1->R4 인터록
P1072C	BIT	R07 HD1 (Ot29) HD1->R5 인터록
P1072D	BIT	R07 HD1 (Ot30) HD1->R6 인터록
P10710	BIT	R07 HD1 (Ot01) W100 간섭무
P10711	BIT	R07 HD1 (Ot02) W150-1 간섭무
P10712	BIT	R07 HD1 (Ot03) W150-2 간섭무
P10713	BIT	R07 HD1 (Ot04) W200 간섭무
P10714	BIT	R07 HD1 (Ot05) W300 간섭무
P1072E	BIT	R07 HD1 (Ot31) HD1->HD2 인터록
P10735	BIT	R07 HD1 (Ot38) 비젼마스타 W400 언로딩완료
P10725	BIT	R07 HD1 (Ot22) 스케너 스타트
P10723	BIT	R07 HD1 (Ot20) LH 스캐너 선택
P10724	BIT	R07 HD1 (Ot21) RH 스캐너 선택
P10800	BIT	R08 HD2 Running
P10801	BIT	R08 HD2 Servo_ON
P10805	BIT	R08 HD2 REMOTE Mode
P10806	BIT	R08 HD2 PLAY Mode
P10807	BIT	R08 HD2 TEACH 모드
P10828	BIT	R08 HD2 (Ot25)
P10839	BIT	R08 HD2 (Ot42) 그리퍼1 클램프 잠김요구
P1082D	BIT	R08 HD2 (Ot30)
P10840	BIT	R08 HD2 (Ot49) 그리퍼2 핀 전진요구
P10837	BIT	R08 HD2 (Ot40) OK 마스타 언로딩 완료
P1083F	BIT	R08 HD2 (Ot48) 그리퍼2 클램프 풀림요구
P1083B	BIT	R08 HD2 (Ot44) 그리퍼1 핀 전진요구
P1082F	BIT	R08 HD2 (Ot32) 비상정지
P10818	BIT	R08 HD2 (Ot09) W400 언로딩 완료 _RG3
P10829	BIT	R08 HD2 (Ot26)
P1080A	BIT	R08 HD2 HOME Position
P10814	BIT	R08 HD2 (Ot05) PLT "A"  간섭무
P10815	BIT	R08 HD2 (Ot06) PLT "B"  간섭무
P10816	BIT	R08 HD2 (Ot07) NG 대차 간섭무
P1081E	BIT	R08 HD2 (Ot15) W700 로딩 완료 _RG3
P1081F	BIT	R08 HD2 (Ot16) W700 언로딩 완료 _RG3
P10821	BIT	R08 HD2 (Ot18) OUT PLT-A FULL
P10822	BIT	R08 HD2 (Ot19) OUT PLT-A 카운터 클리어
P10824	BIT	R08 HD2 (Ot21) OUT PLT-B FULL
P10825	BIT	R08 HD2 (Ot22) OUT PLT-B 카운터 클리어
P10827	BIT	R08 HD2 (Ot24)
P1082A	BIT	R08 HD2 (Ot27)
P1082B	BIT	R08 HD2 (Ot28)
P1082C	BIT	R08 HD2 (Ot29)
P10831	BIT	R08 HD4 (Ot34) 인터록
P10832	BIT	R08 HD2 (Ot35) 인터록
P10833	BIT	R08 HD2 (Ot36) 
P10834	BIT	R08 HD2 (Ot37) 비젼 마스타 로딩 완료
P10835	BIT	R08 HD2 (Ot38) 비젼 마스타 언로딩 완료
P1083A	BIT	R08 HD2 (Ot43) 그리퍼1 클램프 풀림요구
P1083C	BIT	R08 HD2 (Ot45) 그리퍼1 핀 후진요구
P1083E	BIT	R08 HD2 (Ot47) 그리퍼2 클램프 잠김요구
P10843	BIT	R08 HD2 (Ot52)
P1087D	BIT	R08 HD2 그리퍼1 클램프 잠김2
P1087E	BIT	R08 HD2 그리퍼1 클램프 풀림2
P1081C	BIT	R08 HD2 (Ot13) W600 로딩 완료 _RG3
P1081D	BIT	R08 HD2 (Ot14) W600 언로딩 완료 _RG3
P1081A	BIT	R08 HD2 (Ot11) W500 로딩 완료 _RG3
P1081B	BIT	R08 HD2 (Ot12) W500 언로딩 완료 _RG3
P10875	BIT	R08 HD2 그리퍼 클램프 잠김1
P10877	BIT	R08 HD2 그리퍼 클램프 잠김2
P10879	BIT	R08 HD2 그리퍼 클램프 잠김3
P10876	BIT	R08 HD2 그리퍼 클램프 풀림1
P10878	BIT	R08 HD2 그리퍼 클램프 풀림2
P1087A	BIT	R08 HD2 그리퍼 클램프 풀림3
P10872	BIT	R08 HD2 그리퍼 핀 전진1
P10874	BIT	R08 HD2 그리퍼 핀 전진2
P10871	BIT	R08 HD2 그리퍼 핀 후진1
P10873	BIT	R08 HD2 그리퍼 핀 후진2
P10870	BIT	R08 HD2 그리퍼 파트감지
P1088E	BIT	HD-2 H/D Robot Air Press S/W
P10810	BIT	R08 HD2 (Ot01) W400 간섭무
P10811	BIT	R08 HD2 (Ot02) W500 간섭무
P10812	BIT	R08 HD2 (Ot03) W600 간섭무
P10813	BIT	R08 HD2 (Ot03) W700 간섭무
P10817	BIT	R08 HD2 (Ot08) OK 마스타 간섭무
P10830	BIT	R08 HD2 (Ot33) 그리퍼1 No.2 탑너트 파트체크 요구
P1087B	BIT	R08 HD2 그리퍼1 No.2 너트감지 파트1
P1087C	BIT	R08 HD2 그리퍼1 No.2 너트감지 파트2
M10800	BIT	R08 HD2 External RUN
M10801	BIT	R08 HD2 Servo_ON
M10803	BIT	R08 HD2 Error Reset
M10805	BIT	R08 HD2 REMInE Selet
M10806	BIT	R08 HD2 PLAY Select
M10807	BIT	R08 HD2 TEACH Select
M1080A	BIT	OP2 RobIn WELD ON
M1081C	BIT	R08 HD2 (In13) W600 로딩가능 _RG3
M1081D	BIT	R08 HD2 (In14) W600 언로딩가능 _RG3
M1081E	BIT	R08 HD2 (In15) W700 로딩가능 _RG3
M1081F	BIT	R08 HD2 (In16) W700 언로딩가능 _RG3
M10820	BIT	R08 HD2 (In17) PLT-A 로딩 가능
M10822	BIT	R08 HD2 (In19) PLT-A FULL
M10823	BIT	R08 HD2 (In20) PLT-B 로딩 가능
M10825	BIT	R08 HD2 (In22) PLT-B FULL
M10826	BIT	R08 HD2 (In23) NG 대차 로딩 가능 _RG3
M10827	BIT	R08 HD2 (In24) Line 강제배출 Mode On
M1082A	BIT	R08 HD2 (In27)
M1082B	BIT	R08 HD2 (In28)
M1082C	BIT	R08 HD2 (In29)
M1082E	BIT	R08 HD2 (In31) 외부 비상정지
M1082F	BIT	R08 HD2 (In32) 외부 일시정지
M1081B	BIT	R08 HD2 (In12) W500 언로딩가능 _RG3
M10828	BIT	R08 HD2 (In25)
M10829	BIT	R08 HD2 (In26)
M1082D	BIT	R08 HD2 (In30)
M10838	BIT	R08 HD2 (In41) 그리퍼1 파트감지
M10840	BIT	R08 HD2 (In49) 그리퍼2 핀 전진
M1083C	BIT	R08 HD2 (In45) 그리퍼1 핀 후진
M10818	BIT	R08 HD2 (In09) W400 언로딩 가능 _RG3
M10819	BIT	R08 HD2 (In10) 비젼마스타 W400 로딩진입 _RG3
M1081A	BIT	R08 HD2 (In11) W500 로딩 가능 _RG3
M10831	BIT	R08 HD2 (In34)
M10839	BIT	R08 HD2 (In42) 그리퍼1 클램프 잠김
M1083A	BIT	R08 HD2 (In43) 그리퍼1 클램프 풀림
M1083B	BIT	R08 HD2 (In44) 그리퍼1 핀 전진
M1083E	BIT	R08 HD2 (In47) 그리퍼2 클램프 잠김
M1083F	BIT	R08 HD2 (In48) 그리퍼2 클램프 풀림
M10841	BIT	R08 HD2 (In50) 그리퍼2 핀 후진
M10844	BIT	R08 HD2 (In53) W500 사용가능
M10850	BIT	R08 HD2 (In65) OUT PLT-A LOAD COMP 카운터1
M10851	BIT	R08 HD2 (In66) OUT PLT-A LOAD COMP 카운터2
M10852	BIT	R08 HD2 (In67) OUT PLT-A LOAD COMP 카운터4
M10870	BIT	R08 HD2 그리퍼2 핀 전진 SOL
M10871	BIT	R08 HD2 그리퍼2 핀 후진 SOL
M10872	BIT	R08 HD2 그리퍼2 클램프 잠김 SOL
M10873	BIT	R08 HD2 그리퍼2 클램프 풀림 SOL
M10874	BIT	R08 HD2 그리퍼1 핀 전진 Sol
M10875	BIT	R08 HD2 그리퍼1 핀 후진 Sol
M10876	BIT	R08 HD2 그리퍼1 클램프 잠김 Sol
M10877	BIT	R08 HD2 그리퍼1 클램프 풀림 Sol
M10890	BIT	R08 HD2 그리퍼 파트감지 없음
M10842	BIT	R08 HD2 (In51)
M10843	BIT	R08 HD2 (In52)
M10830	BIT	R08 HD2 (In33) 그리퍼 No.2 탑너트 파트체크 OK
P10641	BIT	R06 (OT50)
P10642	BIT	R06 (OT51)
P10643	BIT	R06 (OT52)
P10646	BIT	R06 (OT55)
P10649	BIT	R06 (OT58)
P1064A	BIT	R06 (OT59)
P1064B	BIT	R06 (OT60)
P1064C	BIT	R06 (OT61)
P1064D	BIT	R06 (OT62)
P1064E	BIT	R06 (OT63)
P1064F	BIT	R06 (OT64)
M10641	BIT	R06 (IN50)
M10642	BIT	R06 (IN51)
M10648	BIT	R06 (IN57)
M10649	BIT	R06 (IN58)
M1064A	BIT	R06 (IN59)
M1064B	BIT	R06 (IN60)
M1064C	BIT	R06 (IN61)
M1064D	BIT	R06 (IN62)
M1064E	BIT	R06 (IN63)
M1064F	BIT	R06 (IN64)
M03500	BIT	PC Position 1
T0675	BIT/WORD	PC 측정 시작 지연
M04960	BIT	비젼 마스타 체크 On T/K
M04961	BIT	비젼 마스타 체크 Off T/K
M04962	BIT	비젼 마스타 체크요구 Lamp
M04963	BIT	비젼 마스타 파트있음 Lamp
M04964	BIT	비젼 마스타 예약기동
M04970	BIT	비젼 마스타 Start Lamp
P10836	BIT	R08 HD2 (Ot39) OK 마스타 로딩 완료
P10838	BIT	R08 HD2 (Ot41)
P10848	BIT	R08 HD2 (Ot57) W400 언로딩 완료 _RG3 EV
P10844	BIT	R08 HD2 (Ot53)
P10845	BIT	R08 HD2 (Ot54)
P10846	BIT	R08 HD2 (Ot55)
P10849	BIT	R08 HD2 (Ot58) 비젼마스타 W400 로딩완료 _RG3 EV
P10644	BIT	R06 (OT53)
M10836	BIT	R08 HD2 (In39) OK 마스타 로딩진입
M10837	BIT	R08 HD2 (In40) OK 마스타 언로딩진입
M10834	BIT	R08 HD2 (In37) 비젼 마스타 로딩진입
M10835	BIT	R08 HD2 (In38) 비젼 마스타 언로딩진입
M10845	BIT	R08 HD2 (In54)
M1084F	BIT	R08 HD2 (In64) W700 언로딩가능 _RG3 EV
M10853	BIT	R08 HD2 (In68) OUT PLT-A LOAD COMP 카운터8
M10854	BIT	R08 HD2 (In69)
M10855	BIT	R08 HD2 (In70)
M10856	BIT	R08 HD2 (In71)
M10857	BIT	R08 HD2 (In72)
M10858	BIT	R08 HD2 (In73) OUT PLT-B LOAD COMP 카운터1
M10859	BIT	R08 HD2 (In74) OUT PLT-B LOAD COMP 카운터2
M1085A	BIT	R08 HD2 (In75) OUT PLT-B LOAD COMP 카운터4
M1085B	BIT	R08 HD2 (In76) OUT PLT-B LOAD COMP 카운터8
M1085C	BIT	R08 HD2 (In77)
M1085D	BIT	R08 HD2 (In78)
M1085E	BIT	R08 HD2 (In79)
M1085F	BIT	R08 HD2 (In80)
M10860	BIT	R08 HD2 (In81)
M10861	BIT	R08 HD2 (In82)
M10862	BIT	R08 HD2 (In83)
M10863	BIT	R08 HD2 (In84)
M10864	BIT	R08 HD2 (In85)
M10865	BIT	R08 HD2 (In86)
M10866	BIT	R08 HD2 (In87)
M10867	BIT	R08 HD2 (In88)
M10868	BIT	R08 HD2 (In89)
M10869	BIT	R08 HD2 (In90)
M1086A	BIT	R08 HD2 (In91)
M1086B	BIT	R08 HD2 (In92)
M1086C	BIT	R08 HD2 (In93)
M1086D	BIT	R08 HD2 (In94)
M1086E	BIT	R08 HD2 (In95)
M1086F	BIT	R08 HD2 (In96)
P1084A	BIT	R08 HD2 (Ot59) W500 로딩 완료 _RG3 EV
P1084B	BIT	R08 HD2 (Ot60) W500 언로딩 완료 _RG3 EV
P1084C	BIT	R08 HD2 (Ot61) W600 로딩 완료 _RG3 EV
P1084D	BIT	R08 HD2 (Ot62) W600 언로딩 완료 _RG3 EV
P1084E	BIT	R08 HD2 (Ot63) W700 로딩 완료 _RG3 EV
P1084F	BIT	R08 HD2 (Ot64) W700 언로딩 완료 _RG3 EV
P10850	BIT	R08 HD2 (Ot65)
P10851	BIT	R08 HD2 (Ot66)
P10852	BIT	R08 HD2 (Ot67)
P10853	BIT	R08 HD2 (Ot68)
P10854	BIT	R08 HD2 (Ot69)
P10855	BIT	R08 HD2 (Ot70)
P10856	BIT	R08 HD2 (Ot71)
P10857	BIT	R08 HD2 (Ot72)
P10858	BIT	R08 HD2 (Ot73)
P10859	BIT	R08 HD2 (Ot74)
P1085A	BIT	R08 HD2 (Ot75)
P1085B	BIT	R08 HD2 (Ot76)
P1085C	BIT	R08 HD2 (Ot77)
P1085D	BIT	R08 HD2 (Ot78)
P1085E	BIT	R08 HD2 (Ot79)
P1085F	BIT	R08 HD2 (Ot80)
P10860	BIT	R08 HD2 (Ot81)
P10861	BIT	R08 HD2 (Ot82)
P10862	BIT	R08 HD2 (Ot83)
P10863	BIT	R08 HD2 (Ot84)
P10864	BIT	R08 HD2 (Ot85)
P10865	BIT	R08 HD2 (Ot86)
P10866	BIT	R08 HD2 (Ot87)
P10867	BIT	R08 HD2 (Ot88)
P10868	BIT	R08 HD2 (Ot89)
P10869	BIT	R08 HD2 (Ot90)
P1086A	BIT	R08 HD2 (Ot91)
P1086B	BIT	R08 HD2 (Ot92)
P1086C	BIT	R08 HD2 (Ot93)
P1086D	BIT	R08 HD2 (Ot94)
P1086E	BIT	R08 HD2 (Ot95)
P1086F	BIT	R08 HD2 (Ot96)
P10841	BIT	R08 HD2 (Ot50)
D17000	WORD	1번 비드 품질 정보
D17001	WORD	2번 비드 품질 정보
D17002	WORD	3번 비드 품질 정보
D17003	WORD	4번 비드 품질 정보
D17004	WORD	5번 비드 품질 정보
D17005	WORD	6번 비드 품질 정보
D17006	WORD	7번 비드 품질 정보
D17007	WORD	8번 비드 품질 정보
D17008	WORD	9번 비드 품질 정보
D17009	WORD	10번 비드 품질 정보
D17010	WORD	11번 비드 품질 정보
D17011	WORD	12번 비드 품질 정보
D17012	WORD	13번 비드 품질 정보
D17013	WORD	14번 비드 품질 정보
D17014	WORD	15번 비드 품질 정보
D17015	WORD	16번 비드 품질 정보
D17050	WORD	PC 검사 포인트 
D17050.1	BIT	PC 검사 포인트 2 
D17050.2	BIT	PC 검사 포인트 4
D17050.3	BIT	PC 검사 포인트 8 
D17050.4	BIT	PC 검사 포인트 16 
D17050.5	BIT	PC 검사 포인트 32
D17050.6	BIT	PC 검사 포인트 64
D17050.7	BIT	PC 검사 포인트 128
M10643	BIT	R06 (IN52)
M10645	BIT	R06 (IN54)
D17016	WORD	17번 비드 품질 정보
D17017	WORD	18번 비드 품질 정보
D17018	WORD	19번 비드 품질 정보
D17019	WORD	비젼 정도체크 품질 정보
D17051	WORD	모델번호
D17020.1	BIT	비젼 검사준비 완료
D17020.2	BIT	비드 검사완료 OK
D17020.0	BIT	비젼 초기 대기 
D17020.3	BIT	비드 검사완료 NG
K01851	BIT	비젼마스타 W400 로딩완료 HD2
M01850	BIT	비젼마스타 자동
K01850	BIT	비젼마스타 베이스 슬라이드 전진
K01852	BIT	비젼마스타 베이스 슬라이드 후진
K01853	BIT	비젼마스타 W400 언로딩완료 HD1
K01854	BIT	비젼마스타 W300 언로딩완료 HD1
K01855	BIT	비젼마스타 W400 로딩완료 HD1
K01856	BIT	비젼마스타 베이스 슬라이드 전진
K01857	BIT	비젼마스타 W400 언로딩완료 HD2
K01858	BIT	비젼마스타 작업완료 HD2
P10819	BIT	R08 HD2 (Ot09) 비젼마스타 W400 로딩완료 _RG3
K01896	BIT	비젼 마스타 로딩 완료 지연
K01895	BIT	비젼 마스타 로딩 완료 RST 지연
P10645	BIT	R06 (OT54)
D00560	WORD	W300 비젼정도 P0 측정 1:OK 2:NG
K0185F	BIT	비젼 임시체크 신호
D17061.0	BIT	마스터 체크 신호
M00059	BIT	W50 내부 안전센서 이상
D10000	WORD	라인상태
D10001	WORD	예약
D10005	WORD	현재품번의생산수량
D10006	WORD	예약
D10012	WORD	품번 1의 생산량
D10013	WORD	품번 1의 예약정보
D10014	WORD	품번
D10015	WORD	품번 2의 생산량
D10016	WORD	품번 2의 예약정보
D10017	WORD	품번
D10018	WORD	품번 3의 생산량
D10019	WORD	품번 3의 예약정보
D10020	WORD	품번
D10021	WORD	품번 4의 생산량
D10022	WORD	품번 4의 예약정보
D10023	WORD	품번
D10024	WORD	품번 5의 생산량
D10025	WORD	품번 5의 예약정보
D10026	WORD	품번
D10027	WORD	품번 6의 생산량
D10028	WORD	품번 6의 예약정보
D10029	WORD	품번
D10030	WORD	품번 7의 생산량
D10031	WORD	품번 7의 예약정보
D10032	WORD	품번
D10033	WORD	품번 8의 생산량
D10034	WORD	품번 8의 예약정보
D10035	WORD	품번
D10036	WORD	품번 9의 생산량
D10037	WORD	품번 9의 예약정보
D10038	WORD	품번
D10039	WORD	품번 10의 생산량
D10040	WORD	품번 10의 예약정보
D10041	WORD	품번
D10042	WORD	품번 11의 생산량
D10043	WORD	품번 11의 예약정보
D10044	WORD	품번
D10045	WORD	품번 12의 생산량
D10046	WORD	품번 12의 예약정보
D10047	WORD	품번
D10048	WORD	품번 13의 생산량
D10049	WORD	품번 13의 예약정보
D10050	WORD	품번
D10051	WORD	품번 14의 생산량
D10052	WORD	품번 14의 예약정보
D10053	WORD	품번
D10054	WORD	품번 15의 생산량
D10055	WORD	품번 15의 예약정보
D10056	WORD	품번
D10057	WORD	품번 16의 생산량
D10058	WORD	품번 16의 예약정보
D10059	WORD	품번
D10060	WORD	품번 17의 생산량
D10061	WORD	품번 17의 예약정보
D10062	WORD	품번
D10063	WORD	품번 18의 생산량
D10064	WORD	품번 18의 예약정보
D10065	WORD	품번
D10066	WORD	품번 19의 생산량
D10067	WORD	품번 19의 예약정보
D10068	WORD	품번
D10069	WORD	품번 20의 생산량
D10070	WORD	품번 20의 예약정보
D10071	WORD	품번
D10072	WORD	품번 21의 생산량
D10073	WORD	품번 21의 예약정보
D10074	WORD	품번
D10075	WORD	품번 22의 생산량
D10076	WORD	품번 22의 예약정보
D10077	WORD	품번
D10078	WORD	품번 23의 생산량
D10079	WORD	품번 23의 예약정보
D10080	WORD	품번
D10081	WORD	품번 24의 생산량
D10082	WORD	품번 24의 예약정보
D10083	WORD	품번
D10084	WORD	품번 25의 생산량
D10085	WORD	품번 25의 예약정보
D10086	WORD	품번
D10087	WORD	품번 26의 생산량
D10088	WORD	품번 26의 예약정보
D10089	WORD	품번
D10090	WORD	품번 27의 생산량
D10091	WORD	품번 27의 예약정보
D10092	WORD	품번
D10093	WORD	품번 28의 생산량
D10094	WORD	품번 28의 예약정보
D10095	WORD	품번
D10096	WORD	품번 29의 생산량
D10097	WORD	품번 29의 예약정보
D10098	WORD	품번
D10099	WORD	품번 30의 생산량
D10100	WORD	품번 30의 예약정보
D10101	WORD	품번
D10102	WORD	품번 31의 생산량
D10103	WORD	품번 31의 예약정보
D10104	WORD	품번
D10105	WORD	품번 32의 생산량
D10106	WORD	품번 32의 예약정보
D10107	WORD	품번
D10108	WORD	품번 33의 생산량
D10109	WORD	품번 33의 예약정보
D10110	WORD	품번
D10111	WORD	품번 34의 생산량
D10112	WORD	품번 34의 예약정보
D10113	WORD	품번
D10114	WORD	품번 35의 생산량
D10115	WORD	품번 35의 예약정보
D10116	WORD	품번
D10117	WORD	품번 36의 생산량
D10118	WORD	품번 36의 예약정보
D10119	WORD	품번
D10120	WORD	품번 37의 생산량
D10121	WORD	품번 37의 예약정보
D10122	WORD	품번
D10123	WORD	품번 38의 생산량
D10124	WORD	품번 38의 예약정보
D10125	WORD	품번
D10126	WORD	품번 39의 생산량
D10127	WORD	품번 39의 예약정보
D10128	WORD	품번
D10129	WORD	품번 40의 생산량
D10130	WORD	품번 40의 예약정보
K00002	BIT	차종,2 RG3 EV
P00402	BIT	W10 LH 서보모터 도그1
P00404	BIT	W10 LH 서보모터 도그3
P00403	BIT	W10 LH 서보모터 도그2
D00126	WORD	W50 파트램프 상태16
D00217	WORD	W100 파트램프 상태7
D00218	WORD	W100 파트램프 상태8
P00512	BIT	W10 RH 1차 클램프 잠김4
P00513	BIT	W10 RH 1차 클램프 풀림4
P00516	BIT	W10 RH 3차 클램프 잠김1
P0051A	BIT	W10 RH 3차 클램프 잠김3
P0051B	BIT	W10 RH 3차 클램프 풀림3
P00517	BIT	W10 RH 3차 클램프 풀림1
D00317	WORD	W150-2 파트램프 상태3
D00318	WORD	W150-2 파트램프 상태4
P00603	BIT	W10 RH 서보모터 도그2
P00602	BIT	W10 RH 서보모터 도그1
P00604	BIT	W10 RH 서보모터 도그3
P10780	BIT	R07 HD1 그리퍼2 핀 전진
P10781	BIT	R07 HD1 그리퍼2 핀 후진
P1077E	BIT	R07 HD1 그리퍼2 파트감지1
P1077F	BIT	R07 HD1 그리퍼2 파트감지2
M10811	BIT	R08 HD2 (In02) 차종2
M10810	BIT	R08 HD2 (In01) 차종1
P10782	BIT	R07 HD1 그리퍼2 클램프 잠김
P10783	BIT	R07 HD1 그리퍼2 클램프 풀림
D18507.0	BIT	W200 차종
D18509.0	BIT	W300 차종
M10710	BIT	R07 HD1 (In01) 차종1
M10711	BIT	R07 HD1 (In02) 차종2
D18502.0	BIT	W100 차종
P10746	BIT	R07 HD1 (Ot55) W100 언로딩 완료 _RG3 EV
P10747	BIT	R07 HD1 (Ot56) W150-1 로딩 완료 _RG3 EV
P10748	BIT	R07 HD1 (Ot57) W150-1 언로딩 완료 _RG3 EV
P10749	BIT	R07 HD1 (Ot58) W150-2 로딩 완료 _RG3 EV
P1074A	BIT	R07 HD1 (Ot59) W150-2 언로딩 완료 _RG3 EV
P1074B	BIT	R07 HD1 (Ot60) W200 로딩 완료 _RG3 EV
P1074C	BIT	R07 HD1 (Ot61) W200 언로딩 완료 _RG3 EV
P1074D	BIT	R07 HD1 (Ot62) W300 로딩 완료 _RG3 EV
P1074E	BIT	R07 HD1 (Ot63) W300 언로딩 완료 _RG3 EV
P1074F	BIT	R07 HD1 (Ot64) W400 로딩 완료 _RG3 EV
M10746	BIT	R07 HD1 (In55) W100 언로딩 가능 _RG3 EV
M10747	BIT	R07 HD1 (In56) W150-1 로딩 가능 _RG3 EV
M10748	BIT	R07 HD1 (In57) W150-1 언로딩가능 _RG3 EV
M10749	BIT	R07 HD1 (In58) W150-2 로딩가능 _RG3 EV
M1074A	BIT	R07 HD1 (In59) W150-2 언로딩가능 _RG3 EV
M1074B	BIT	R07 HD1 (In60) W200 로딩가능 _RG3 EV
M1074C	BIT	R07 HD1 (In61) W200 언로딩가능 _RG3 EV
M1074D	BIT	R07 HD1 (In62) W300 로딩가능 _RG3 EV
M1074E	BIT	R07 HD1 (In63) W300 언로딩가능 _RG3 EV
M1074F	BIT	R07 HD1 (In64) W400 로딩가능 _RG3 EV
M10848	BIT	R08 HD2 (In57) W400 언로딩 가능 _RG3 EV
M10849	BIT	R08 HD2 (In58) 비젼마스타 W400 로딩진입 _RG3 EV
M1084A	BIT	R08 HD2 (In59) W500 로딩 가능 _RG3 EV
M1084B	BIT	R08 HD2 (In60) W500 언로딩가능 _RG3 EV
M1084C	BIT	R08 HD2 (In61) W600 로딩가능 _RG3 EV
M1084D	BIT	R08 HD2 (In62) W600 언로딩가능 _RG3 EV
M1084E	BIT	R08 HD2 (In63) W700 로딩가능 _RG3 EV
P10842	BIT	R08 HD2 (Ot51) 에어클리너 On 요구
M10833	BIT	R08 HD2 (In36) W600 NG슈트 취출진입 EV
M10832	BIT	R08 HD2 (In35) W600 NG슈트 취출진입 RG3
K00071	BIT	차종변경 RG3 EV -> RG3
K00072	BIT	차종변경 RG3 -> RG3 EV
D36010	WORD	G1: CTR "L" REAL 스펙Data <RG3 EV>
D36012	WORD	G1: CTR "L" REAL 하한치 <RG3 EV>
D36017	WORD	G1: CTR "L" REAL 상한치 <RG3 EV>
D36020	WORD	G2:FRT LH "T" REAL 스펙Data <RG3 EV>
D36022	WORD	G2:FRT LH "T" REAL 하한치 <RG3 EV>
D36027	WORD	G2:FRT LH "T" REAL 상한치 <RG3 EV>
D36030	WORD	G3:FRT LH "L" REAL 스펙Data <RG3 EV>
D36032	WORD	G3:FRT LH "L" REAL 하한치 <RG3 EV>
D36037	WORD	G3:FRT LH "L" REAL 상한치 <RG3 EV>
D36040	WORD	G4:FRT LH "H" REAL 스펙Data <RG3 EV>
D36042	WORD	G4:FRT LH "H" REAL 하한치 <RG3 EV>
D36047	WORD	G4:FRT LH "H" REAL 상한치 <RG3 EV>
D36050	WORD	G5:FRT RH "T" REAL 스펙Data <RG3 EV>
D36052	WORD	G5:FRT RH "T" REAL 하한치 <RG3 EV>
D36057	WORD	G5:FRT RH "T" REAL 상한치 <RG3 EV>
D36060	WORD	G6:FRT RH "L" REAL 스펙Data <RG3 EV>
D36062	WORD	G6:FRT RH "L" REAL 하한치 <RG3 EV>
D36067	WORD	G6:FRT RH "L" REAL 상한치 <RG3 EV>
D36070	WORD	G7:FRT RH "H" REAL 스펙Data <RG3 EV>
D36072	WORD	G7:FRT RH "H" REAL 하한치 <RG3 EV>
D36077	WORD	G7:FRT RH "H" REAL 상한치 <RG3 EV>
D36080	WORD	G8:RR LH "T" REAL 스펙Data <RG3 EV>
D36082	WORD	G8:RR LH "T" REAL 하한치 <RG3 EV>
D36087	WORD	G8:RR LH "T" REAL 상한치 <RG3 EV>
D36090	WORD	G9:RR LH "L" REAL 스펙Data <RG3 EV>
D36092	WORD	G9:RR LH "L" REAL 하한치 <RG3 EV>
D36097	WORD	G9:RR LH "L" REAL 상한치 <RG3 EV>
D36100	WORD	G10:RR LH "H" REAL 스펙Data <RG3 EV>
D36102	WORD	G10:RR LH "H" REAL 하한치 <RG3 EV>
D36107	WORD	G10:RR LH "H" REAL 상한치 <RG3 EV>
D36110	WORD	G11:RR RH "T" REAL 스펙Data <RG3 EV>
D36112	WORD	G11:RR RH "T" REAL 하한치 <RG3 EV>
D36117	WORD	G11:RR RH "T" REAL 상한치 <RG3 EV>
D36120	WORD	G12:RR RH "L" REAL 스펙Data <RG3 EV>
D36122	WORD	G12:RR RH "L" REAL 하한치 <RG3 EV>
D36127	WORD	G12:RR RH "L" REAL 상한치 <RG3 EV>
D36130	WORD	G13:RR RH "H" REAL 스펙Data <RG3 EV>
D36132	WORD	G13:RR RH "H" REAL 하한치 <RG3 EV>
D36137	WORD	G13:RR RH "H" REAL 상한치 <RG3 EV>
D36150	WORD	W500 G1:CTR "L" REAL Data 차이 <RG3 EV>
D36152	WORD	OK/NG마스타 G1:CTR "L" REAL Data 차이 <RG3 EV>
D36155	WORD	W500 G2:FRT LH "T" REAL Data 차이 <RG3 EV>
D36157	WORD	OK/NG마스타 G2:FRT LH "T" REAL Data 차이 <RG3 EV>
D36160	WORD	W500 G3:FRT LH "L" REAL Data 차이 <RG3 EV>
D36162	WORD	OK/NG마스타 G3:FRT LH "L" REAL Data 차이 <RG3 EV>
D36165	WORD	W500 G4:FRT LH "H" REAL Data 차이 <RG3 EV>
D36167	WORD	OK/NG마스타 G4:FRT LH "H" REAL Data 차이 <RG3 EV>
D36170	WORD	W500 G5:FRT RH "T" REAL Data 차이 <RG3 EV>
D36172	WORD	OK/NG마스타 G5:FRT RH "T" REAL Data 차이 <RG3 EV>
D36175	WORD	W500 G6:FRT RH "L" REAL Data 차이 <RG3 EV>
D36177	WORD	OK/NG마스타 G6:FRT RH "L" REAL Data 차이 <RG3 EV>
D36180	WORD	W500 G7:FRT RH "H" REAL Data 차이 <RG3 EV>
D36182	WORD	OK/NG마스타 G7:FRT RH "H" REAL Data 차이 <RG3 EV>
D36185	WORD	W500 G8:RR LH "T" REAL Data 차이 <RG3 EV>
